// TIA Portal V17 export
// export: Created 2023-02-14T02:49:49.5801565Z, ExportSetting WithDefaults, DisplayName Totally Integrated Automation Portal, DisplayVersion V17, DisplayName TIA Portal Openness, DisplayVersion V17, DisplayName TIA Portal Teamcenter Gateway, DisplayVersion V17, DisplayName TIA Portal Version Control Interface, DisplayVersion V17, DisplayName SINAMICS Startdrive Advanced, DisplayVersion V17, DisplayName SINAMICS Startdrive G130, G150, S120, S150, SINAMICS MV, S210, DisplayVersion V17, DisplayName SINAMICS Startdrive G110M, G120, G120C, G120D, G120P, G115D, DisplayVersion V17, DisplayName STEP 7 Professional, DisplayVersion V17, DisplayName STEP 7 Safety, DisplayVersion V17, DisplayName WinCC Professional, DisplayVersion V17
FUNCTION "Preparation" : Void   // FC6, LAD
{ S7_Optimized_Access := 'TRUE' }
VERSION : 0.1
// stored: AutoNumber true, IsIECCheckEnabled false, SetENOAutomatically false, UDAEnableTagReadback false
   VAR_TEMP   // added for the SCL form of the ladder/FBD networks
      _w1 : Bool;
      _w2 : Bool;
      _w3 : Bool;
      _w4 : Bool;
      _w5 : Bool;
   END_VAR
BEGIN

REGION Network 1: Analog IO
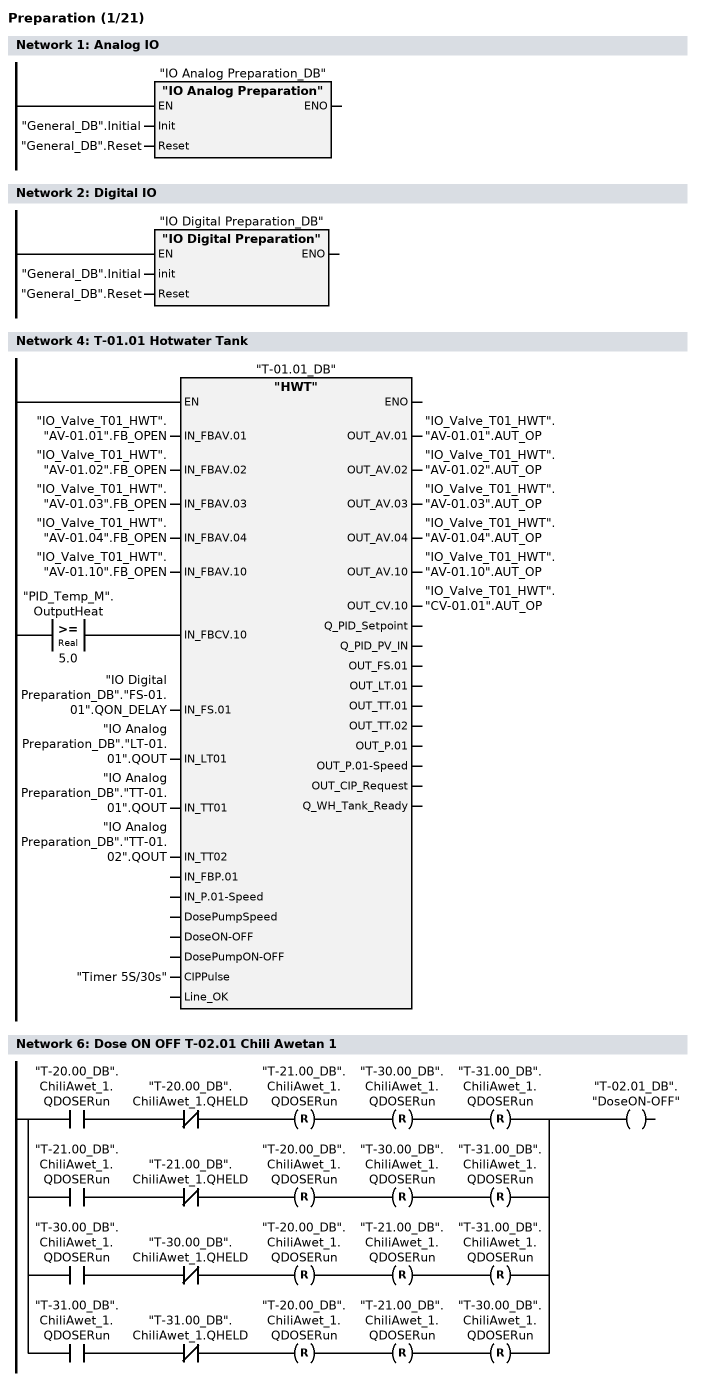
   RUNG wire#powerrail
      "IO Analog Preparation_DB"(Init := "General_DB".Initial, Reset := "General_DB".Reset)
   END_RUNG
   // the same network as SCL:
   "IO Analog Preparation_DB"(Init := "General_DB".Initial, Reset := "General_DB".Reset);   // "IO Analog Preparation"
END_REGION

REGION Network 2: Digital IO
   RUNG wire#powerrail
      "IO Digital Preparation_DB"(init := "General_DB".Initial, Reset := "General_DB".Reset)
   END_RUNG
   // the same network as SCL:
   "IO Digital Preparation_DB"(init := "General_DB".Initial, Reset := "General_DB".Reset);   // "IO Digital Preparation"
END_REGION

REGION Network 4: T-01.01 Hotwater Tank
   RUNG wire#powerrail
      "T-01.01_DB"("IN_FBCV.10" := wire#w1, "IN_FBAV.01" := "IO_Valve_T01_HWT"."AV-01.01".FB_OPEN, "IN_FBAV.02" := "IO_Valve_T01_HWT"."AV-01.02".FB_OPEN, "IN_FBAV.03" := "IO_Valve_T01_HWT"."AV-01.03".FB_OPEN, "IN_FBAV.04" := "IO_Valve_T01_HWT"."AV-01.04".FB_OPEN, "IN_FBAV.10" := "IO_Valve_T01_HWT"."AV-01.10".FB_OPEN, "IN_FS.01" := "IO Digital Preparation_DB"."FS-01.01".QON_DELAY, IN_LT01 := "IO Analog Preparation_DB"."LT-01.01".QOUT, IN_TT01 := "IO Analog Preparation_DB"."TT-01.01".QOUT, IN_TT02 := "IO Analog Preparation_DB"."TT-01.02".QOUT, "IN_FBP.01" :=, "IN_P.01-Speed" :=, DosePumpSpeed :=, "DoseON-OFF" :=, "DosePumpON-OFF" :=, CIPPulse := "Timer 5S/30s", Line_OK :=, "OUT_AV.01" => "IO_Valve_T01_HWT"."AV-01.01".AUT_OP, "OUT_AV.02" => "IO_Valve_T01_HWT"."AV-01.02".AUT_OP, "OUT_AV.03" => "IO_Valve_T01_HWT"."AV-01.03".AUT_OP, "OUT_AV.04" => "IO_Valve_T01_HWT"."AV-01.04".AUT_OP, "OUT_AV.10" => "IO_Valve_T01_HWT"."AV-01.10".AUT_OP, "OUT_CV.10" => "IO_Valve_T01_HWT"."CV-01.01".AUT_OP, Q_PID_Setpoint =>, Q_PID_PV_IN =>, "OUT_FS.01" =>, "OUT_LT.01" =>, "OUT_TT.01" =>, "OUT_TT.02" =>, "OUT_P.01" =>, "OUT_P.01-Speed" =>, OUT_CIP_Request =>, Q_WH_Tank_Ready =>)
   END_RUNG
   RUNG wire#powerrail
      { S7_Templates := "SrcType := Real" } GE_Contact(in1 := "PID_Temp_M".OutputHeat, in2 := 5.0)
   END_RUNG wire#w1
   // the same network as SCL:
   "T-01.01_DB"("IN_FBAV.01" := "IO_Valve_T01_HWT"."AV-01.01".FB_OPEN,   // "HWT"
                "IN_FBAV.02" := "IO_Valve_T01_HWT"."AV-01.02".FB_OPEN,
                "IN_FBAV.03" := "IO_Valve_T01_HWT"."AV-01.03".FB_OPEN,
                "IN_FBAV.04" := "IO_Valve_T01_HWT"."AV-01.04".FB_OPEN,
                "IN_FBAV.10" := "IO_Valve_T01_HWT"."AV-01.10".FB_OPEN,
                "IN_FBCV.10" := "PID_Temp_M".OutputHeat >= 5.0,
                "IN_FS.01" := "IO Digital Preparation_DB"."FS-01.01".QON_DELAY,
                IN_LT01 := "IO Analog Preparation_DB"."LT-01.01".QOUT,
                IN_TT01 := "IO Analog Preparation_DB"."TT-01.01".QOUT,
                IN_TT02 := "IO Analog Preparation_DB"."TT-01.02".QOUT,
                CIPPulse := "Timer 5S/30s",
                "OUT_AV.01" => "IO_Valve_T01_HWT"."AV-01.01".AUT_OP,
                "OUT_AV.02" => "IO_Valve_T01_HWT"."AV-01.02".AUT_OP,
                "OUT_AV.03" => "IO_Valve_T01_HWT"."AV-01.03".AUT_OP,
                "OUT_AV.04" => "IO_Valve_T01_HWT"."AV-01.04".AUT_OP,
                "OUT_AV.10" => "IO_Valve_T01_HWT"."AV-01.10".AUT_OP,
                "OUT_CV.10" => "IO_Valve_T01_HWT"."CV-01.01".AUT_OP);
END_REGION

REGION Network 6: Dose ON OFF T-02.01 Chili Awetan 1
   RUNG wire#powerrail
      Contact( "T-20.00_DB".ChiliAwet_1.QDOSERun )
      I_Contact( "T-20.00_DB".ChiliAwet_1.QHELD )
      R_Coil( "T-21.00_DB".ChiliAwet_1.QDOSERun )
      R_Coil( "T-30.00_DB".ChiliAwet_1.QDOSERun )
      R_Coil( "T-31.00_DB".ChiliAwet_1.QDOSERun )
      wire#w1
      Coil( "T-02.01_DB"."DoseON-OFF" )
   END_RUNG
   RUNG wire#powerrail
      Contact( "T-21.00_DB".ChiliAwet_1.QDOSERun )
      I_Contact( "T-21.00_DB".ChiliAwet_1.QHELD )
      R_Coil( "T-20.00_DB".ChiliAwet_1.QDOSERun )
      R_Coil( "T-30.00_DB".ChiliAwet_1.QDOSERun )
      R_Coil( "T-31.00_DB".ChiliAwet_1.QDOSERun )
   END_RUNG wire#w1
   RUNG wire#powerrail
      Contact( "T-30.00_DB".ChiliAwet_1.QDOSERun )
      I_Contact( "T-30.00_DB".ChiliAwet_1.QHELD )
      R_Coil( "T-20.00_DB".ChiliAwet_1.QDOSERun )
      R_Coil( "T-21.00_DB".ChiliAwet_1.QDOSERun )
      R_Coil( "T-31.00_DB".ChiliAwet_1.QDOSERun )
   END_RUNG wire#w1
   RUNG wire#powerrail
      Contact( "T-31.00_DB".ChiliAwet_1.QDOSERun )
      I_Contact( "T-31.00_DB".ChiliAwet_1.QHELD )
      R_Coil( "T-20.00_DB".ChiliAwet_1.QDOSERun )
      R_Coil( "T-21.00_DB".ChiliAwet_1.QDOSERun )
      R_Coil( "T-30.00_DB".ChiliAwet_1.QDOSERun )
   END_RUNG wire#w1
   // the same network as SCL:
   #_w1 := "T-20.00_DB".ChiliAwet_1.QDOSERun AND NOT "T-20.00_DB".ChiliAwet_1.QHELD;
   IF #_w1 THEN
       "T-21.00_DB".ChiliAwet_1.QDOSERun := FALSE;
       "T-30.00_DB".ChiliAwet_1.QDOSERun := FALSE;
       "T-31.00_DB".ChiliAwet_1.QDOSERun := FALSE;
   END_IF;
   #_w2 := "T-21.00_DB".ChiliAwet_1.QDOSERun AND NOT "T-21.00_DB".ChiliAwet_1.QHELD;
   IF #_w2 THEN
       "T-20.00_DB".ChiliAwet_1.QDOSERun := FALSE;
       "T-30.00_DB".ChiliAwet_1.QDOSERun := FALSE;
       "T-31.00_DB".ChiliAwet_1.QDOSERun := FALSE;
   END_IF;
   #_w3 := "T-30.00_DB".ChiliAwet_1.QDOSERun AND NOT "T-30.00_DB".ChiliAwet_1.QHELD;
   IF #_w3 THEN
       "T-20.00_DB".ChiliAwet_1.QDOSERun := FALSE;
       "T-21.00_DB".ChiliAwet_1.QDOSERun := FALSE;
       "T-31.00_DB".ChiliAwet_1.QDOSERun := FALSE;
   END_IF;
   #_w4 := "T-31.00_DB".ChiliAwet_1.QDOSERun AND NOT "T-31.00_DB".ChiliAwet_1.QHELD;
   IF #_w4 THEN
       "T-20.00_DB".ChiliAwet_1.QDOSERun := FALSE;
       "T-21.00_DB".ChiliAwet_1.QDOSERun := FALSE;
       "T-30.00_DB".ChiliAwet_1.QDOSERun := FALSE;
   END_IF;
   "T-02.01_DB"."DoseON-OFF" := #_w1 OR #_w2 OR #_w3 OR #_w4;
END_REGION

REGION Network 7: Dose Pump ON OFF T-02.01 Chili Awetan 1
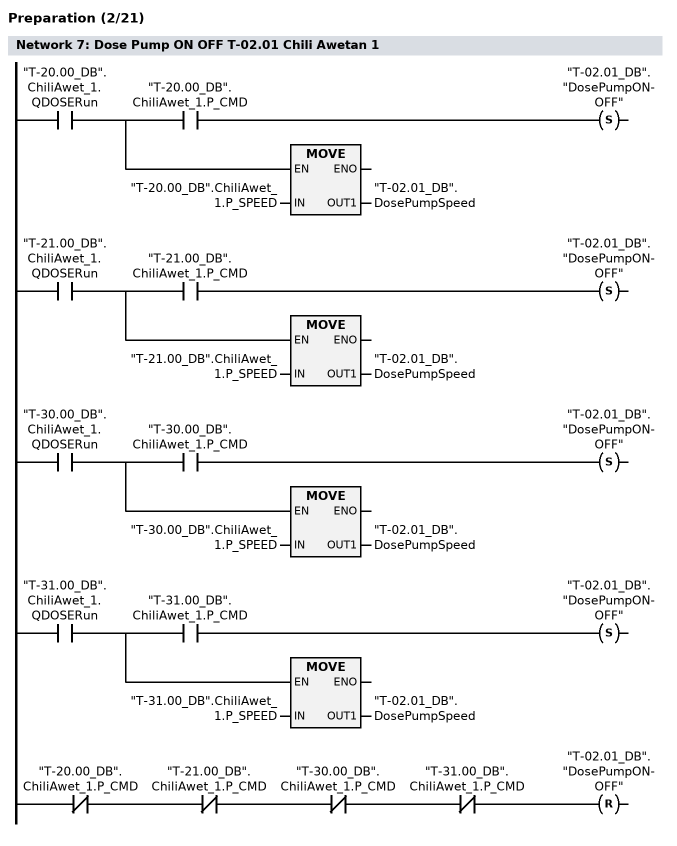
   RUNG wire#powerrail
      Contact( "T-20.00_DB".ChiliAwet_1.QDOSERun )
      wire#w1
      Contact( "T-20.00_DB".ChiliAwet_1.P_CMD )
      S_Coil( "T-02.01_DB"."DosePumpON-OFF" )
   END_RUNG
   RUNG wire#w1
      Move(in := "T-20.00_DB".ChiliAwet_1.P_SPEED, out1 => "T-02.01_DB".DosePumpSpeed)
   END_RUNG
   RUNG wire#powerrail
      Contact( "T-21.00_DB".ChiliAwet_1.QDOSERun )
      wire#w2
      Contact( "T-21.00_DB".ChiliAwet_1.P_CMD )
      S_Coil( "T-02.01_DB"."DosePumpON-OFF" )
   END_RUNG
   RUNG wire#w2
      Move(in := "T-21.00_DB".ChiliAwet_1.P_SPEED, out1 => "T-02.01_DB".DosePumpSpeed)
   END_RUNG
   RUNG wire#powerrail
      Contact( "T-30.00_DB".ChiliAwet_1.QDOSERun )
      wire#w3
      Contact( "T-30.00_DB".ChiliAwet_1.P_CMD )
      S_Coil( "T-02.01_DB"."DosePumpON-OFF" )
   END_RUNG
   RUNG wire#w3
      Move(in := "T-30.00_DB".ChiliAwet_1.P_SPEED, out1 => "T-02.01_DB".DosePumpSpeed)
   END_RUNG
   RUNG wire#powerrail
      Contact( "T-31.00_DB".ChiliAwet_1.QDOSERun )
      wire#w4
      Contact( "T-31.00_DB".ChiliAwet_1.P_CMD )
      S_Coil( "T-02.01_DB"."DosePumpON-OFF" )
   END_RUNG
   RUNG wire#w4
      Move(in := "T-31.00_DB".ChiliAwet_1.P_SPEED, out1 => "T-02.01_DB".DosePumpSpeed)
   END_RUNG
   RUNG wire#powerrail
      I_Contact( "T-20.00_DB".ChiliAwet_1.P_CMD )
      I_Contact( "T-21.00_DB".ChiliAwet_1.P_CMD )
      I_Contact( "T-30.00_DB".ChiliAwet_1.P_CMD )
      I_Contact( "T-31.00_DB".ChiliAwet_1.P_CMD )
      R_Coil( "T-02.01_DB"."DosePumpON-OFF" )
   END_RUNG
   // the same network as SCL:
   IF "T-20.00_DB".ChiliAwet_1.QDOSERun AND "T-20.00_DB".ChiliAwet_1.P_CMD THEN
       "T-02.01_DB"."DosePumpON-OFF" := TRUE;
   END_IF;
   IF "T-20.00_DB".ChiliAwet_1.QDOSERun THEN
       "T-02.01_DB".DosePumpSpeed := "T-20.00_DB".ChiliAwet_1.P_SPEED;
   END_IF;
   IF "T-21.00_DB".ChiliAwet_1.QDOSERun AND "T-21.00_DB".ChiliAwet_1.P_CMD THEN
       "T-02.01_DB"."DosePumpON-OFF" := TRUE;
   END_IF;
   IF "T-21.00_DB".ChiliAwet_1.QDOSERun THEN
       "T-02.01_DB".DosePumpSpeed := "T-21.00_DB".ChiliAwet_1.P_SPEED;
   END_IF;
   IF "T-30.00_DB".ChiliAwet_1.QDOSERun AND "T-30.00_DB".ChiliAwet_1.P_CMD THEN
       "T-02.01_DB"."DosePumpON-OFF" := TRUE;
   END_IF;
   IF "T-30.00_DB".ChiliAwet_1.QDOSERun THEN
       "T-02.01_DB".DosePumpSpeed := "T-30.00_DB".ChiliAwet_1.P_SPEED;
   END_IF;
   IF "T-31.00_DB".ChiliAwet_1.QDOSERun AND "T-31.00_DB".ChiliAwet_1.P_CMD THEN
       "T-02.01_DB"."DosePumpON-OFF" := TRUE;
   END_IF;
   IF "T-31.00_DB".ChiliAwet_1.QDOSERun THEN
       "T-02.01_DB".DosePumpSpeed := "T-31.00_DB".ChiliAwet_1.P_SPEED;
   END_IF;
   IF NOT "T-20.00_DB".ChiliAwet_1.P_CMD AND NOT "T-21.00_DB".ChiliAwet_1.P_CMD AND NOT "T-30.00_DB".ChiliAwet_1.P_CMD AND NOT "T-31.00_DB".ChiliAwet_1.P_CMD THEN
       "T-02.01_DB"."DosePumpON-OFF" := FALSE;
   END_IF;
END_REGION

REGION Network 8: T-02.01 Buffer Tank Chili Awetan
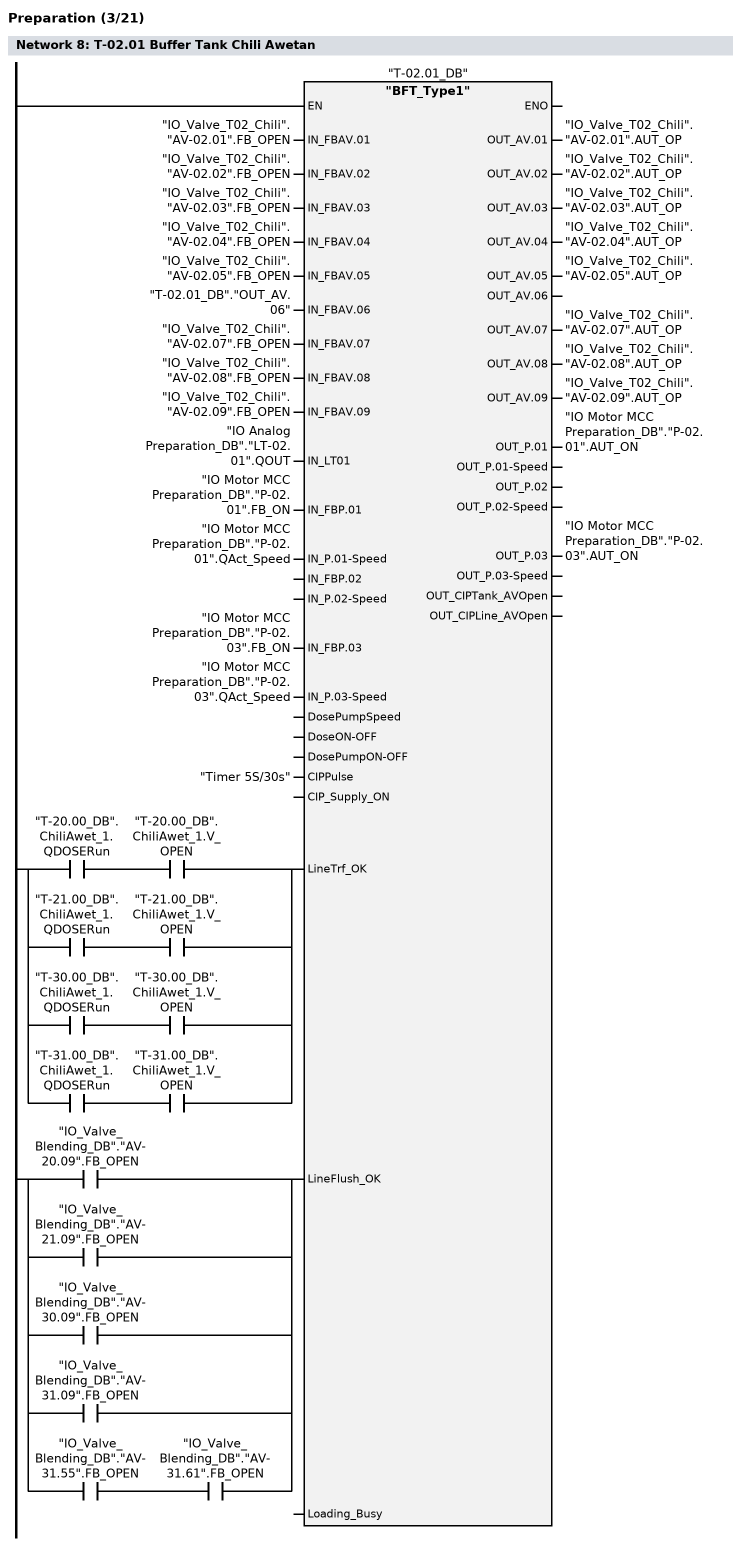
   RUNG wire#powerrail
      "T-02.01_DB"(LineTrf_OK := wire#w1, LineFlush_OK := wire#w2, "IN_FBAV.01" := "IO_Valve_T02_Chili"."AV-02.01".FB_OPEN, "IN_FBAV.02" := "IO_Valve_T02_Chili"."AV-02.02".FB_OPEN, "IN_FBAV.03" := "IO_Valve_T02_Chili"."AV-02.03".FB_OPEN, "IN_FBAV.04" := "IO_Valve_T02_Chili"."AV-02.04".FB_OPEN, "IN_FBAV.05" := "IO_Valve_T02_Chili"."AV-02.05".FB_OPEN, "IN_FBAV.06" := "T-02.01_DB"."OUT_AV.06", "IN_FBAV.07" := "IO_Valve_T02_Chili"."AV-02.07".FB_OPEN, "IN_FBAV.08" := "IO_Valve_T02_Chili"."AV-02.08".FB_OPEN, "IN_FBAV.09" := "IO_Valve_T02_Chili"."AV-02.09".FB_OPEN, IN_LT01 := "IO Analog Preparation_DB"."LT-02.01".QOUT, "IN_FBP.01" := "IO Motor MCC Preparation_DB"."P-02.01".FB_ON, "IN_P.01-Speed" := "IO Motor MCC Preparation_DB"."P-02.01".QAct_Speed, "IN_FBP.02" :=, "IN_P.02-Speed" :=, "IN_FBP.03" := "IO Motor MCC Preparation_DB"."P-02.03".FB_ON, "IN_P.03-Speed" := "IO Motor MCC Preparation_DB"."P-02.03".QAct_Speed, DosePumpSpeed :=, "DoseON-OFF" :=, "DosePumpON-OFF" :=, CIPPulse := "Timer 5S/30s", CIP_Supply_ON :=, Loading_Busy :=, "OUT_AV.01" => "IO_Valve_T02_Chili"."AV-02.01".AUT_OP, "OUT_AV.02" => "IO_Valve_T02_Chili"."AV-02.02".AUT_OP, "OUT_AV.03" => "IO_Valve_T02_Chili"."AV-02.03".AUT_OP, "OUT_AV.04" => "IO_Valve_T02_Chili"."AV-02.04".AUT_OP, "OUT_AV.05" => "IO_Valve_T02_Chili"."AV-02.05".AUT_OP, "OUT_AV.06" =>, "OUT_AV.07" => "IO_Valve_T02_Chili"."AV-02.07".AUT_OP, "OUT_AV.08" => "IO_Valve_T02_Chili"."AV-02.08".AUT_OP, "OUT_AV.09" => "IO_Valve_T02_Chili"."AV-02.09".AUT_OP, "OUT_P.01" => "IO Motor MCC Preparation_DB"."P-02.01".AUT_ON, "OUT_P.01-Speed" =>, "OUT_P.02" =>, "OUT_P.02-Speed" =>, "OUT_P.03" => "IO Motor MCC Preparation_DB"."P-02.03".AUT_ON, "OUT_P.03-Speed" =>, OUT_CIPTank_AVOpen =>, OUT_CIPLine_AVOpen =>)
   END_RUNG
   RUNG wire#powerrail
      Contact( "T-20.00_DB".ChiliAwet_1.QDOSERun )
      Contact( "T-20.00_DB".ChiliAwet_1.V_OPEN )
   END_RUNG wire#w1
   RUNG wire#powerrail
      Contact( "T-21.00_DB".ChiliAwet_1.QDOSERun )
      Contact( "T-21.00_DB".ChiliAwet_1.V_OPEN )
   END_RUNG wire#w1
   RUNG wire#powerrail
      Contact( "T-30.00_DB".ChiliAwet_1.QDOSERun )
      Contact( "T-30.00_DB".ChiliAwet_1.V_OPEN )
   END_RUNG wire#w1
   RUNG wire#powerrail
      Contact( "T-31.00_DB".ChiliAwet_1.QDOSERun )
      Contact( "T-31.00_DB".ChiliAwet_1.V_OPEN )
   END_RUNG wire#w1
   RUNG wire#powerrail
      Contact( "IO_Valve_Blending_DB"."AV-20.09".FB_OPEN )
   END_RUNG wire#w2
   RUNG wire#powerrail
      Contact( "IO_Valve_Blending_DB"."AV-21.09".FB_OPEN )
   END_RUNG wire#w2
   RUNG wire#powerrail
      Contact( "IO_Valve_Blending_DB"."AV-30.09".FB_OPEN )
   END_RUNG wire#w2
   RUNG wire#powerrail
      Contact( "IO_Valve_Blending_DB"."AV-31.09".FB_OPEN )
   END_RUNG wire#w2
   RUNG wire#powerrail
      Contact( "IO_Valve_Blending_DB"."AV-31.55".FB_OPEN )
      Contact( "IO_Valve_Blending_DB"."AV-31.61".FB_OPEN )
   END_RUNG wire#w2
   // the same network as SCL:
   "T-02.01_DB"("IN_FBAV.01" := "IO_Valve_T02_Chili"."AV-02.01".FB_OPEN,   // "BFT_Type1"
                "IN_FBAV.02" := "IO_Valve_T02_Chili"."AV-02.02".FB_OPEN,
                "IN_FBAV.03" := "IO_Valve_T02_Chili"."AV-02.03".FB_OPEN,
                "IN_FBAV.04" := "IO_Valve_T02_Chili"."AV-02.04".FB_OPEN,
                "IN_FBAV.05" := "IO_Valve_T02_Chili"."AV-02.05".FB_OPEN,
                "IN_FBAV.06" := "T-02.01_DB"."OUT_AV.06",
                "IN_FBAV.07" := "IO_Valve_T02_Chili"."AV-02.07".FB_OPEN,
                "IN_FBAV.08" := "IO_Valve_T02_Chili"."AV-02.08".FB_OPEN,
                "IN_FBAV.09" := "IO_Valve_T02_Chili"."AV-02.09".FB_OPEN,
                IN_LT01 := "IO Analog Preparation_DB"."LT-02.01".QOUT,
                "IN_FBP.01" := "IO Motor MCC Preparation_DB"."P-02.01".FB_ON,
                "IN_P.01-Speed" := "IO Motor MCC Preparation_DB"."P-02.01".QAct_Speed,
                "IN_FBP.03" := "IO Motor MCC Preparation_DB"."P-02.03".FB_ON,
                "IN_P.03-Speed" := "IO Motor MCC Preparation_DB"."P-02.03".QAct_Speed,
                CIPPulse := "Timer 5S/30s",
                LineTrf_OK := ("T-20.00_DB".ChiliAwet_1.QDOSERun AND "T-20.00_DB".ChiliAwet_1.V_OPEN) OR ("T-21.00_DB".ChiliAwet_1.QDOSERun AND "T-21.00_DB".ChiliAwet_1.V_OPEN) OR ("T-30.00_DB".ChiliAwet_1.QDOSERun AND "T-30.00_DB".ChiliAwet_1.V_OPEN) OR ("T-31.00_DB".ChiliAwet_1.QDOSERun AND "T-31.00_DB".ChiliAwet_1.V_OPEN),
                LineFlush_OK := "IO_Valve_Blending_DB"."AV-20.09".FB_OPEN OR "IO_Valve_Blending_DB"."AV-21.09".FB_OPEN OR "IO_Valve_Blending_DB"."AV-30.09".FB_OPEN OR "IO_Valve_Blending_DB"."AV-31.09".FB_OPEN OR ("IO_Valve_Blending_DB"."AV-31.55".FB_OPEN AND "IO_Valve_Blending_DB"."AV-31.61".FB_OPEN),
                "OUT_AV.01" => "IO_Valve_T02_Chili"."AV-02.01".AUT_OP,
                "OUT_AV.02" => "IO_Valve_T02_Chili"."AV-02.02".AUT_OP,
                "OUT_AV.03" => "IO_Valve_T02_Chili"."AV-02.03".AUT_OP,
                "OUT_AV.04" => "IO_Valve_T02_Chili"."AV-02.04".AUT_OP,
                "OUT_AV.05" => "IO_Valve_T02_Chili"."AV-02.05".AUT_OP,
                "OUT_AV.07" => "IO_Valve_T02_Chili"."AV-02.07".AUT_OP,
                "OUT_AV.08" => "IO_Valve_T02_Chili"."AV-02.08".AUT_OP,
                "OUT_AV.09" => "IO_Valve_T02_Chili"."AV-02.09".AUT_OP,
                "OUT_P.01" => "IO Motor MCC Preparation_DB"."P-02.01".AUT_ON,
                "OUT_P.03" => "IO Motor MCC Preparation_DB"."P-02.03".AUT_ON);
END_REGION

REGION Network 10: Dose ON OFF T-03.01 Chili Awetan 2
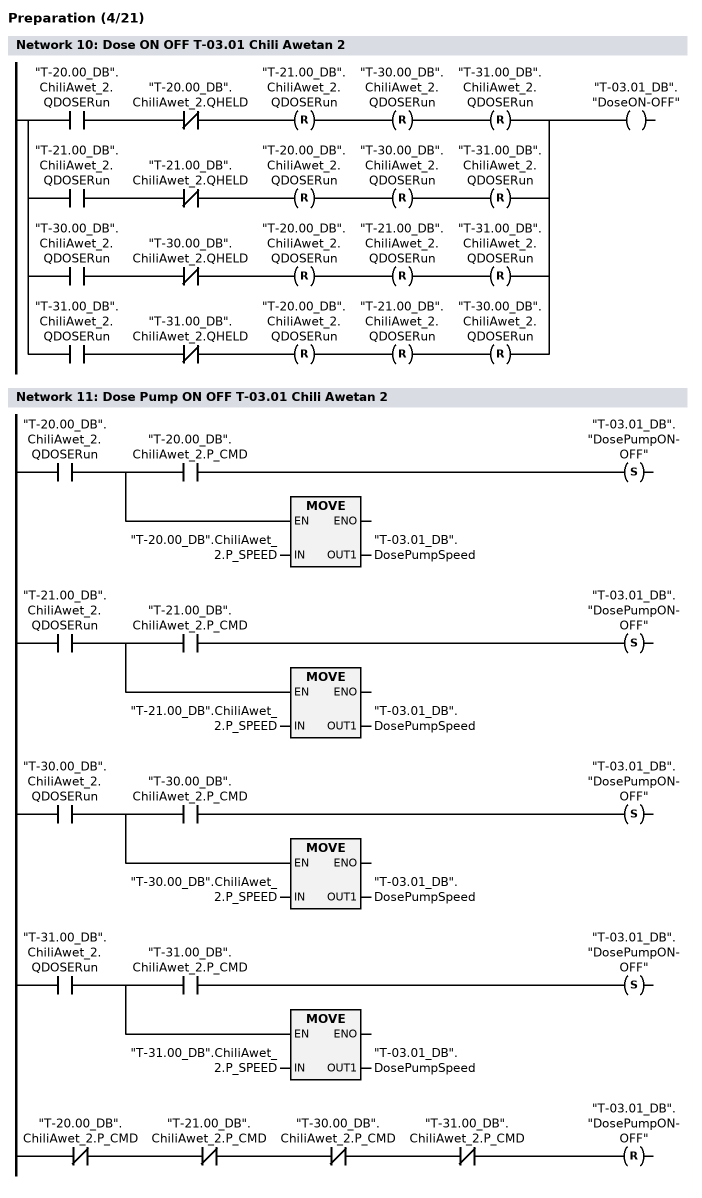
   RUNG wire#powerrail
      Contact( "T-20.00_DB".ChiliAwet_2.QDOSERun )
      I_Contact( "T-20.00_DB".ChiliAwet_2.QHELD )
      R_Coil( "T-21.00_DB".ChiliAwet_2.QDOSERun )
      R_Coil( "T-30.00_DB".ChiliAwet_2.QDOSERun )
      R_Coil( "T-31.00_DB".ChiliAwet_2.QDOSERun )
      wire#w1
      Coil( "T-03.01_DB"."DoseON-OFF" )
   END_RUNG
   RUNG wire#powerrail
      Contact( "T-21.00_DB".ChiliAwet_2.QDOSERun )
      I_Contact( "T-21.00_DB".ChiliAwet_2.QHELD )
      R_Coil( "T-20.00_DB".ChiliAwet_2.QDOSERun )
      R_Coil( "T-30.00_DB".ChiliAwet_2.QDOSERun )
      R_Coil( "T-31.00_DB".ChiliAwet_2.QDOSERun )
   END_RUNG wire#w1
   RUNG wire#powerrail
      Contact( "T-30.00_DB".ChiliAwet_2.QDOSERun )
      I_Contact( "T-30.00_DB".ChiliAwet_2.QHELD )
      R_Coil( "T-20.00_DB".ChiliAwet_2.QDOSERun )
      R_Coil( "T-21.00_DB".ChiliAwet_2.QDOSERun )
      R_Coil( "T-31.00_DB".ChiliAwet_2.QDOSERun )
   END_RUNG wire#w1
   RUNG wire#powerrail
      Contact( "T-31.00_DB".ChiliAwet_2.QDOSERun )
      I_Contact( "T-31.00_DB".ChiliAwet_2.QHELD )
      R_Coil( "T-20.00_DB".ChiliAwet_2.QDOSERun )
      R_Coil( "T-21.00_DB".ChiliAwet_2.QDOSERun )
      R_Coil( "T-30.00_DB".ChiliAwet_2.QDOSERun )
   END_RUNG wire#w1
   // the same network as SCL:
   #_w1 := "T-20.00_DB".ChiliAwet_2.QDOSERun AND NOT "T-20.00_DB".ChiliAwet_2.QHELD;
   IF #_w1 THEN
       "T-21.00_DB".ChiliAwet_2.QDOSERun := FALSE;
       "T-30.00_DB".ChiliAwet_2.QDOSERun := FALSE;
       "T-31.00_DB".ChiliAwet_2.QDOSERun := FALSE;
   END_IF;
   #_w2 := "T-21.00_DB".ChiliAwet_2.QDOSERun AND NOT "T-21.00_DB".ChiliAwet_2.QHELD;
   IF #_w2 THEN
       "T-20.00_DB".ChiliAwet_2.QDOSERun := FALSE;
       "T-30.00_DB".ChiliAwet_2.QDOSERun := FALSE;
       "T-31.00_DB".ChiliAwet_2.QDOSERun := FALSE;
   END_IF;
   #_w3 := "T-30.00_DB".ChiliAwet_2.QDOSERun AND NOT "T-30.00_DB".ChiliAwet_2.QHELD;
   IF #_w3 THEN
       "T-20.00_DB".ChiliAwet_2.QDOSERun := FALSE;
       "T-21.00_DB".ChiliAwet_2.QDOSERun := FALSE;
       "T-31.00_DB".ChiliAwet_2.QDOSERun := FALSE;
   END_IF;
   #_w4 := "T-31.00_DB".ChiliAwet_2.QDOSERun AND NOT "T-31.00_DB".ChiliAwet_2.QHELD;
   IF #_w4 THEN
       "T-20.00_DB".ChiliAwet_2.QDOSERun := FALSE;
       "T-21.00_DB".ChiliAwet_2.QDOSERun := FALSE;
       "T-30.00_DB".ChiliAwet_2.QDOSERun := FALSE;
   END_IF;
   "T-03.01_DB"."DoseON-OFF" := #_w1 OR #_w2 OR #_w3 OR #_w4;
END_REGION

REGION Network 11: Dose Pump ON OFF T-03.01 Chili Awetan 2
   RUNG wire#powerrail
      Contact( "T-20.00_DB".ChiliAwet_2.QDOSERun )
      wire#w1
      Contact( "T-20.00_DB".ChiliAwet_2.P_CMD )
      S_Coil( "T-03.01_DB"."DosePumpON-OFF" )
   END_RUNG
   RUNG wire#w1
      Move(in := "T-20.00_DB".ChiliAwet_2.P_SPEED, out1 => "T-03.01_DB".DosePumpSpeed)
   END_RUNG
   RUNG wire#powerrail
      Contact( "T-21.00_DB".ChiliAwet_2.QDOSERun )
      wire#w2
      Contact( "T-21.00_DB".ChiliAwet_2.P_CMD )
      S_Coil( "T-03.01_DB"."DosePumpON-OFF" )
   END_RUNG
   RUNG wire#w2
      Move(in := "T-21.00_DB".ChiliAwet_2.P_SPEED, out1 => "T-03.01_DB".DosePumpSpeed)
   END_RUNG
   RUNG wire#powerrail
      Contact( "T-30.00_DB".ChiliAwet_2.QDOSERun )
      wire#w3
      Contact( "T-30.00_DB".ChiliAwet_2.P_CMD )
      S_Coil( "T-03.01_DB"."DosePumpON-OFF" )
   END_RUNG
   RUNG wire#w3
      Move(in := "T-30.00_DB".ChiliAwet_2.P_SPEED, out1 => "T-03.01_DB".DosePumpSpeed)
   END_RUNG
   RUNG wire#powerrail
      Contact( "T-31.00_DB".ChiliAwet_2.QDOSERun )
      wire#w4
      Contact( "T-31.00_DB".ChiliAwet_2.P_CMD )
      S_Coil( "T-03.01_DB"."DosePumpON-OFF" )
   END_RUNG
   RUNG wire#w4
      Move(in := "T-31.00_DB".ChiliAwet_2.P_SPEED, out1 => "T-03.01_DB".DosePumpSpeed)
   END_RUNG
   RUNG wire#powerrail
      I_Contact( "T-20.00_DB".ChiliAwet_2.P_CMD )
      I_Contact( "T-21.00_DB".ChiliAwet_2.P_CMD )
      I_Contact( "T-30.00_DB".ChiliAwet_2.P_CMD )
      I_Contact( "T-31.00_DB".ChiliAwet_2.P_CMD )
      R_Coil( "T-03.01_DB"."DosePumpON-OFF" )
   END_RUNG
   // the same network as SCL:
   IF "T-20.00_DB".ChiliAwet_2.QDOSERun AND "T-20.00_DB".ChiliAwet_2.P_CMD THEN
       "T-03.01_DB"."DosePumpON-OFF" := TRUE;
   END_IF;
   IF "T-20.00_DB".ChiliAwet_2.QDOSERun THEN
       "T-03.01_DB".DosePumpSpeed := "T-20.00_DB".ChiliAwet_2.P_SPEED;
   END_IF;
   IF "T-21.00_DB".ChiliAwet_2.QDOSERun AND "T-21.00_DB".ChiliAwet_2.P_CMD THEN
       "T-03.01_DB"."DosePumpON-OFF" := TRUE;
   END_IF;
   IF "T-21.00_DB".ChiliAwet_2.QDOSERun THEN
       "T-03.01_DB".DosePumpSpeed := "T-21.00_DB".ChiliAwet_2.P_SPEED;
   END_IF;
   IF "T-30.00_DB".ChiliAwet_2.QDOSERun AND "T-30.00_DB".ChiliAwet_2.P_CMD THEN
       "T-03.01_DB"."DosePumpON-OFF" := TRUE;
   END_IF;
   IF "T-30.00_DB".ChiliAwet_2.QDOSERun THEN
       "T-03.01_DB".DosePumpSpeed := "T-30.00_DB".ChiliAwet_2.P_SPEED;
   END_IF;
   IF "T-31.00_DB".ChiliAwet_2.QDOSERun AND "T-31.00_DB".ChiliAwet_2.P_CMD THEN
       "T-03.01_DB"."DosePumpON-OFF" := TRUE;
   END_IF;
   IF "T-31.00_DB".ChiliAwet_2.QDOSERun THEN
       "T-03.01_DB".DosePumpSpeed := "T-31.00_DB".ChiliAwet_2.P_SPEED;
   END_IF;
   IF NOT "T-20.00_DB".ChiliAwet_2.P_CMD AND NOT "T-21.00_DB".ChiliAwet_2.P_CMD AND NOT "T-30.00_DB".ChiliAwet_2.P_CMD AND NOT "T-31.00_DB".ChiliAwet_2.P_CMD THEN
       "T-03.01_DB"."DosePumpON-OFF" := FALSE;
   END_IF;
END_REGION

REGION Network 12: T-03.01 Buffer Tank Chili Awetan
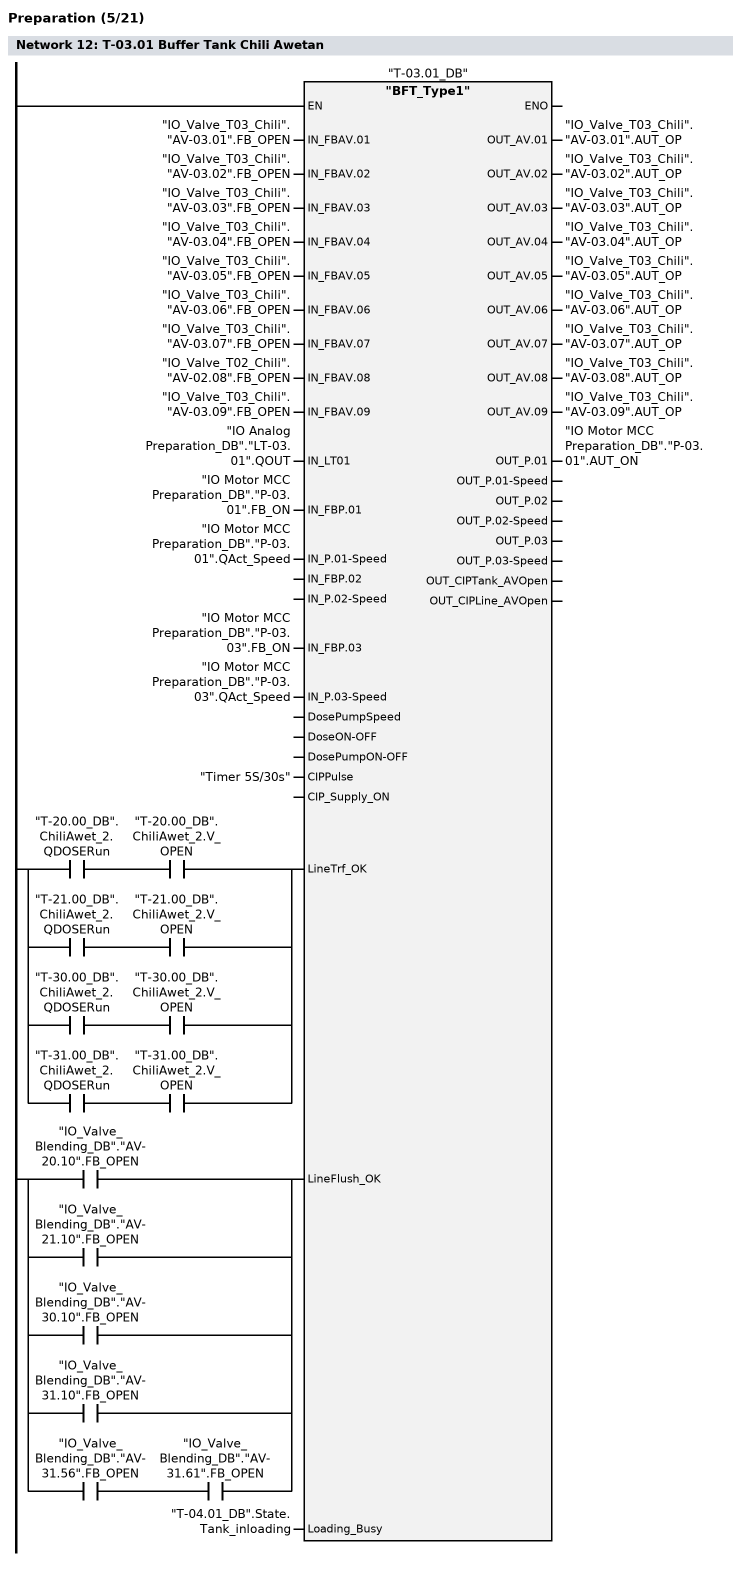
   RUNG wire#powerrail
      "T-03.01_DB"(LineTrf_OK := wire#w1, LineFlush_OK := wire#w2, "IN_FBAV.01" := "IO_Valve_T03_Chili"."AV-03.01".FB_OPEN, "IN_FBAV.02" := "IO_Valve_T03_Chili"."AV-03.02".FB_OPEN, "IN_FBAV.03" := "IO_Valve_T03_Chili"."AV-03.03".FB_OPEN, "IN_FBAV.04" := "IO_Valve_T03_Chili"."AV-03.04".FB_OPEN, "IN_FBAV.05" := "IO_Valve_T03_Chili"."AV-03.05".FB_OPEN, "IN_FBAV.06" := "IO_Valve_T03_Chili"."AV-03.06".FB_OPEN, "IN_FBAV.07" := "IO_Valve_T03_Chili"."AV-03.07".FB_OPEN, "IN_FBAV.08" := "IO_Valve_T02_Chili"."AV-02.08".FB_OPEN, "IN_FBAV.09" := "IO_Valve_T03_Chili"."AV-03.09".FB_OPEN, IN_LT01 := "IO Analog Preparation_DB"."LT-03.01".QOUT, "IN_FBP.01" := "IO Motor MCC Preparation_DB"."P-03.01".FB_ON, "IN_P.01-Speed" := "IO Motor MCC Preparation_DB"."P-03.01".QAct_Speed, "IN_FBP.02" :=, "IN_P.02-Speed" :=, "IN_FBP.03" := "IO Motor MCC Preparation_DB"."P-03.03".FB_ON, "IN_P.03-Speed" := "IO Motor MCC Preparation_DB"."P-03.03".QAct_Speed, DosePumpSpeed :=, "DoseON-OFF" :=, "DosePumpON-OFF" :=, CIPPulse := "Timer 5S/30s", CIP_Supply_ON :=, Loading_Busy := "T-04.01_DB".State.Tank_inloading, "OUT_AV.01" => "IO_Valve_T03_Chili"."AV-03.01".AUT_OP, "OUT_AV.02" => "IO_Valve_T03_Chili"."AV-03.02".AUT_OP, "OUT_AV.03" => "IO_Valve_T03_Chili"."AV-03.03".AUT_OP, "OUT_AV.04" => "IO_Valve_T03_Chili"."AV-03.04".AUT_OP, "OUT_AV.05" => "IO_Valve_T03_Chili"."AV-03.05".AUT_OP, "OUT_AV.06" => "IO_Valve_T03_Chili"."AV-03.06".AUT_OP, "OUT_AV.07" => "IO_Valve_T03_Chili"."AV-03.07".AUT_OP, "OUT_AV.08" => "IO_Valve_T03_Chili"."AV-03.08".AUT_OP, "OUT_AV.09" => "IO_Valve_T03_Chili"."AV-03.09".AUT_OP, "OUT_P.01" => "IO Motor MCC Preparation_DB"."P-03.01".AUT_ON, "OUT_P.01-Speed" =>, "OUT_P.02" =>, "OUT_P.02-Speed" =>, "OUT_P.03" =>, "OUT_P.03-Speed" =>, OUT_CIPTank_AVOpen =>, OUT_CIPLine_AVOpen =>)
   END_RUNG
   RUNG wire#powerrail
      Contact( "T-20.00_DB".ChiliAwet_2.QDOSERun )
      Contact( "T-20.00_DB".ChiliAwet_2.V_OPEN )
   END_RUNG wire#w1
   RUNG wire#powerrail
      Contact( "T-21.00_DB".ChiliAwet_2.QDOSERun )
      Contact( "T-21.00_DB".ChiliAwet_2.V_OPEN )
   END_RUNG wire#w1
   RUNG wire#powerrail
      Contact( "T-30.00_DB".ChiliAwet_2.QDOSERun )
      Contact( "T-30.00_DB".ChiliAwet_2.V_OPEN )
   END_RUNG wire#w1
   RUNG wire#powerrail
      Contact( "T-31.00_DB".ChiliAwet_2.QDOSERun )
      Contact( "T-31.00_DB".ChiliAwet_2.V_OPEN )
   END_RUNG wire#w1
   RUNG wire#powerrail
      Contact( "IO_Valve_Blending_DB"."AV-20.10".FB_OPEN )
   END_RUNG wire#w2
   RUNG wire#powerrail
      Contact( "IO_Valve_Blending_DB"."AV-21.10".FB_OPEN )
   END_RUNG wire#w2
   RUNG wire#powerrail
      Contact( "IO_Valve_Blending_DB"."AV-30.10".FB_OPEN )
   END_RUNG wire#w2
   RUNG wire#powerrail
      Contact( "IO_Valve_Blending_DB"."AV-31.10".FB_OPEN )
   END_RUNG wire#w2
   RUNG wire#powerrail
      Contact( "IO_Valve_Blending_DB"."AV-31.56".FB_OPEN )
      Contact( "IO_Valve_Blending_DB"."AV-31.61".FB_OPEN )
   END_RUNG wire#w2
   // the same network as SCL:
   "T-03.01_DB"("IN_FBAV.01" := "IO_Valve_T03_Chili"."AV-03.01".FB_OPEN,   // "BFT_Type1"
                "IN_FBAV.02" := "IO_Valve_T03_Chili"."AV-03.02".FB_OPEN,
                "IN_FBAV.03" := "IO_Valve_T03_Chili"."AV-03.03".FB_OPEN,
                "IN_FBAV.04" := "IO_Valve_T03_Chili"."AV-03.04".FB_OPEN,
                "IN_FBAV.05" := "IO_Valve_T03_Chili"."AV-03.05".FB_OPEN,
                "IN_FBAV.06" := "IO_Valve_T03_Chili"."AV-03.06".FB_OPEN,
                "IN_FBAV.07" := "IO_Valve_T03_Chili"."AV-03.07".FB_OPEN,
                "IN_FBAV.08" := "IO_Valve_T02_Chili"."AV-02.08".FB_OPEN,
                "IN_FBAV.09" := "IO_Valve_T03_Chili"."AV-03.09".FB_OPEN,
                IN_LT01 := "IO Analog Preparation_DB"."LT-03.01".QOUT,
                "IN_FBP.01" := "IO Motor MCC Preparation_DB"."P-03.01".FB_ON,
                "IN_P.01-Speed" := "IO Motor MCC Preparation_DB"."P-03.01".QAct_Speed,
                "IN_FBP.03" := "IO Motor MCC Preparation_DB"."P-03.03".FB_ON,
                "IN_P.03-Speed" := "IO Motor MCC Preparation_DB"."P-03.03".QAct_Speed,
                CIPPulse := "Timer 5S/30s",
                LineTrf_OK := ("T-20.00_DB".ChiliAwet_2.QDOSERun AND "T-20.00_DB".ChiliAwet_2.V_OPEN) OR ("T-21.00_DB".ChiliAwet_2.QDOSERun AND "T-21.00_DB".ChiliAwet_2.V_OPEN) OR ("T-30.00_DB".ChiliAwet_2.QDOSERun AND "T-30.00_DB".ChiliAwet_2.V_OPEN) OR ("T-31.00_DB".ChiliAwet_2.QDOSERun AND "T-31.00_DB".ChiliAwet_2.V_OPEN),
                LineFlush_OK := "IO_Valve_Blending_DB"."AV-20.10".FB_OPEN OR "IO_Valve_Blending_DB"."AV-21.10".FB_OPEN OR "IO_Valve_Blending_DB"."AV-30.10".FB_OPEN OR "IO_Valve_Blending_DB"."AV-31.10".FB_OPEN OR ("IO_Valve_Blending_DB"."AV-31.56".FB_OPEN AND "IO_Valve_Blending_DB"."AV-31.61".FB_OPEN),
                Loading_Busy := "T-04.01_DB".State.Tank_inloading,
                "OUT_AV.01" => "IO_Valve_T03_Chili"."AV-03.01".AUT_OP,
                "OUT_AV.02" => "IO_Valve_T03_Chili"."AV-03.02".AUT_OP,
                "OUT_AV.03" => "IO_Valve_T03_Chili"."AV-03.03".AUT_OP,
                "OUT_AV.04" => "IO_Valve_T03_Chili"."AV-03.04".AUT_OP,
                "OUT_AV.05" => "IO_Valve_T03_Chili"."AV-03.05".AUT_OP,
                "OUT_AV.06" => "IO_Valve_T03_Chili"."AV-03.06".AUT_OP,
                "OUT_AV.07" => "IO_Valve_T03_Chili"."AV-03.07".AUT_OP,
                "OUT_AV.08" => "IO_Valve_T03_Chili"."AV-03.08".AUT_OP,
                "OUT_AV.09" => "IO_Valve_T03_Chili"."AV-03.09".AUT_OP,
                "OUT_P.01" => "IO Motor MCC Preparation_DB"."P-03.01".AUT_ON);
END_REGION

REGION Network 14: Dose ON OFF T-04.01 Chili Awetan 3
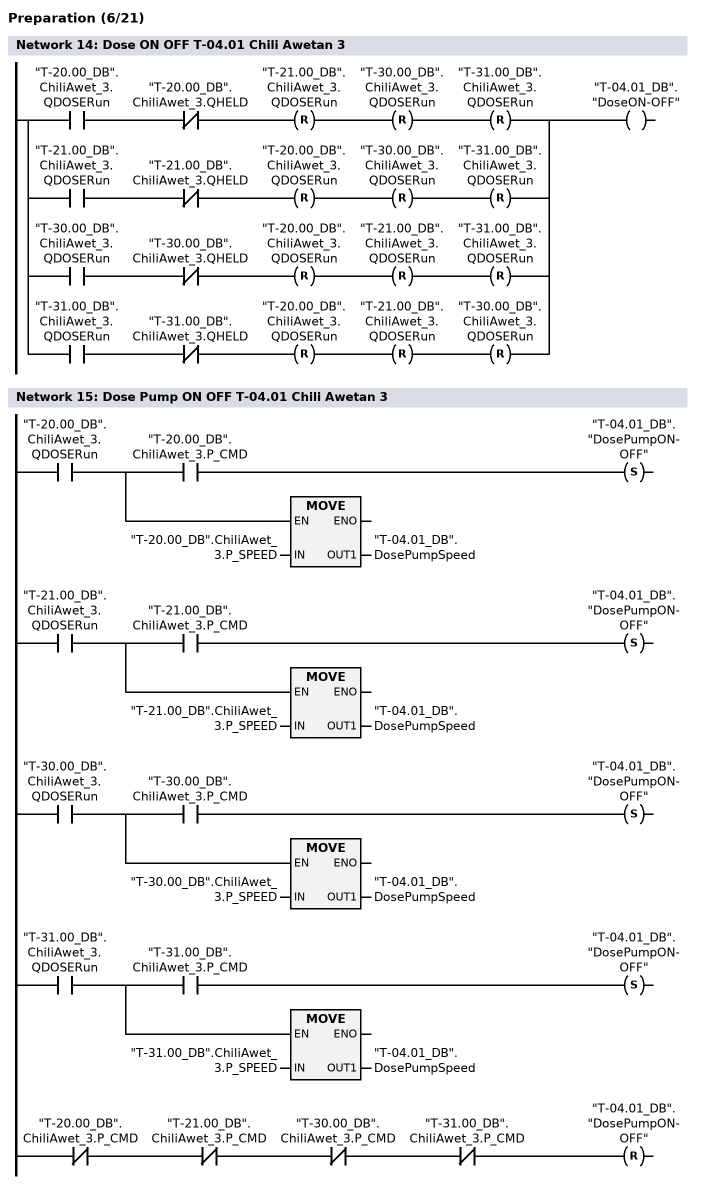
   RUNG wire#powerrail
      Contact( "T-20.00_DB".ChiliAwet_3.QDOSERun )
      I_Contact( "T-20.00_DB".ChiliAwet_3.QHELD )
      R_Coil( "T-21.00_DB".ChiliAwet_3.QDOSERun )
      R_Coil( "T-30.00_DB".ChiliAwet_3.QDOSERun )
      R_Coil( "T-31.00_DB".ChiliAwet_3.QDOSERun )
      wire#w1
      Coil( "T-04.01_DB"."DoseON-OFF" )
   END_RUNG
   RUNG wire#powerrail
      Contact( "T-21.00_DB".ChiliAwet_3.QDOSERun )
      I_Contact( "T-21.00_DB".ChiliAwet_3.QHELD )
      R_Coil( "T-20.00_DB".ChiliAwet_3.QDOSERun )
      R_Coil( "T-30.00_DB".ChiliAwet_3.QDOSERun )
      R_Coil( "T-31.00_DB".ChiliAwet_3.QDOSERun )
   END_RUNG wire#w1
   RUNG wire#powerrail
      Contact( "T-30.00_DB".ChiliAwet_3.QDOSERun )
      I_Contact( "T-30.00_DB".ChiliAwet_3.QHELD )
      R_Coil( "T-20.00_DB".ChiliAwet_3.QDOSERun )
      R_Coil( "T-21.00_DB".ChiliAwet_3.QDOSERun )
      R_Coil( "T-31.00_DB".ChiliAwet_3.QDOSERun )
   END_RUNG wire#w1
   RUNG wire#powerrail
      Contact( "T-31.00_DB".ChiliAwet_3.QDOSERun )
      I_Contact( "T-31.00_DB".ChiliAwet_3.QHELD )
      R_Coil( "T-20.00_DB".ChiliAwet_3.QDOSERun )
      R_Coil( "T-21.00_DB".ChiliAwet_3.QDOSERun )
      R_Coil( "T-30.00_DB".ChiliAwet_3.QDOSERun )
   END_RUNG wire#w1
   // the same network as SCL:
   #_w1 := "T-20.00_DB".ChiliAwet_3.QDOSERun AND NOT "T-20.00_DB".ChiliAwet_3.QHELD;
   IF #_w1 THEN
       "T-21.00_DB".ChiliAwet_3.QDOSERun := FALSE;
       "T-30.00_DB".ChiliAwet_3.QDOSERun := FALSE;
       "T-31.00_DB".ChiliAwet_3.QDOSERun := FALSE;
   END_IF;
   #_w2 := "T-21.00_DB".ChiliAwet_3.QDOSERun AND NOT "T-21.00_DB".ChiliAwet_3.QHELD;
   IF #_w2 THEN
       "T-20.00_DB".ChiliAwet_3.QDOSERun := FALSE;
       "T-30.00_DB".ChiliAwet_3.QDOSERun := FALSE;
       "T-31.00_DB".ChiliAwet_3.QDOSERun := FALSE;
   END_IF;
   #_w3 := "T-30.00_DB".ChiliAwet_3.QDOSERun AND NOT "T-30.00_DB".ChiliAwet_3.QHELD;
   IF #_w3 THEN
       "T-20.00_DB".ChiliAwet_3.QDOSERun := FALSE;
       "T-21.00_DB".ChiliAwet_3.QDOSERun := FALSE;
       "T-31.00_DB".ChiliAwet_3.QDOSERun := FALSE;
   END_IF;
   #_w4 := "T-31.00_DB".ChiliAwet_3.QDOSERun AND NOT "T-31.00_DB".ChiliAwet_3.QHELD;
   IF #_w4 THEN
       "T-20.00_DB".ChiliAwet_3.QDOSERun := FALSE;
       "T-21.00_DB".ChiliAwet_3.QDOSERun := FALSE;
       "T-30.00_DB".ChiliAwet_3.QDOSERun := FALSE;
   END_IF;
   "T-04.01_DB"."DoseON-OFF" := #_w1 OR #_w2 OR #_w3 OR #_w4;
END_REGION

REGION Network 15: Dose Pump ON OFF T-04.01 Chili Awetan 3
   RUNG wire#powerrail
      Contact( "T-20.00_DB".ChiliAwet_3.QDOSERun )
      wire#w1
      Contact( "T-20.00_DB".ChiliAwet_3.P_CMD )
      S_Coil( "T-04.01_DB"."DosePumpON-OFF" )
   END_RUNG
   RUNG wire#w1
      Move(in := "T-20.00_DB".ChiliAwet_3.P_SPEED, out1 => "T-04.01_DB".DosePumpSpeed)
   END_RUNG
   RUNG wire#powerrail
      Contact( "T-21.00_DB".ChiliAwet_3.QDOSERun )
      wire#w2
      Contact( "T-21.00_DB".ChiliAwet_3.P_CMD )
      S_Coil( "T-04.01_DB"."DosePumpON-OFF" )
   END_RUNG
   RUNG wire#w2
      Move(in := "T-21.00_DB".ChiliAwet_3.P_SPEED, out1 => "T-04.01_DB".DosePumpSpeed)
   END_RUNG
   RUNG wire#powerrail
      Contact( "T-30.00_DB".ChiliAwet_3.QDOSERun )
      wire#w3
      Contact( "T-30.00_DB".ChiliAwet_3.P_CMD )
      S_Coil( "T-04.01_DB"."DosePumpON-OFF" )
   END_RUNG
   RUNG wire#w3
      Move(in := "T-30.00_DB".ChiliAwet_3.P_SPEED, out1 => "T-04.01_DB".DosePumpSpeed)
   END_RUNG
   RUNG wire#powerrail
      Contact( "T-31.00_DB".ChiliAwet_3.QDOSERun )
      wire#w4
      Contact( "T-31.00_DB".ChiliAwet_3.P_CMD )
      S_Coil( "T-04.01_DB"."DosePumpON-OFF" )
   END_RUNG
   RUNG wire#w4
      Move(in := "T-31.00_DB".ChiliAwet_3.P_SPEED, out1 => "T-04.01_DB".DosePumpSpeed)
   END_RUNG
   RUNG wire#powerrail
      I_Contact( "T-20.00_DB".ChiliAwet_3.P_CMD )
      I_Contact( "T-21.00_DB".ChiliAwet_3.P_CMD )
      I_Contact( "T-30.00_DB".ChiliAwet_3.P_CMD )
      I_Contact( "T-31.00_DB".ChiliAwet_3.P_CMD )
      R_Coil( "T-04.01_DB"."DosePumpON-OFF" )
   END_RUNG
   // the same network as SCL:
   IF "T-20.00_DB".ChiliAwet_3.QDOSERun AND "T-20.00_DB".ChiliAwet_3.P_CMD THEN
       "T-04.01_DB"."DosePumpON-OFF" := TRUE;
   END_IF;
   IF "T-20.00_DB".ChiliAwet_3.QDOSERun THEN
       "T-04.01_DB".DosePumpSpeed := "T-20.00_DB".ChiliAwet_3.P_SPEED;
   END_IF;
   IF "T-21.00_DB".ChiliAwet_3.QDOSERun AND "T-21.00_DB".ChiliAwet_3.P_CMD THEN
       "T-04.01_DB"."DosePumpON-OFF" := TRUE;
   END_IF;
   IF "T-21.00_DB".ChiliAwet_3.QDOSERun THEN
       "T-04.01_DB".DosePumpSpeed := "T-21.00_DB".ChiliAwet_3.P_SPEED;
   END_IF;
   IF "T-30.00_DB".ChiliAwet_3.QDOSERun AND "T-30.00_DB".ChiliAwet_3.P_CMD THEN
       "T-04.01_DB"."DosePumpON-OFF" := TRUE;
   END_IF;
   IF "T-30.00_DB".ChiliAwet_3.QDOSERun THEN
       "T-04.01_DB".DosePumpSpeed := "T-30.00_DB".ChiliAwet_3.P_SPEED;
   END_IF;
   IF "T-31.00_DB".ChiliAwet_3.QDOSERun AND "T-31.00_DB".ChiliAwet_3.P_CMD THEN
       "T-04.01_DB"."DosePumpON-OFF" := TRUE;
   END_IF;
   IF "T-31.00_DB".ChiliAwet_3.QDOSERun THEN
       "T-04.01_DB".DosePumpSpeed := "T-31.00_DB".ChiliAwet_3.P_SPEED;
   END_IF;
   IF NOT "T-20.00_DB".ChiliAwet_3.P_CMD AND NOT "T-21.00_DB".ChiliAwet_3.P_CMD AND NOT "T-30.00_DB".ChiliAwet_3.P_CMD AND NOT "T-31.00_DB".ChiliAwet_3.P_CMD THEN
       "T-04.01_DB"."DosePumpON-OFF" := FALSE;
   END_IF;
END_REGION

REGION Network 16: T-04.01 Buffer Tank Chili Awetan
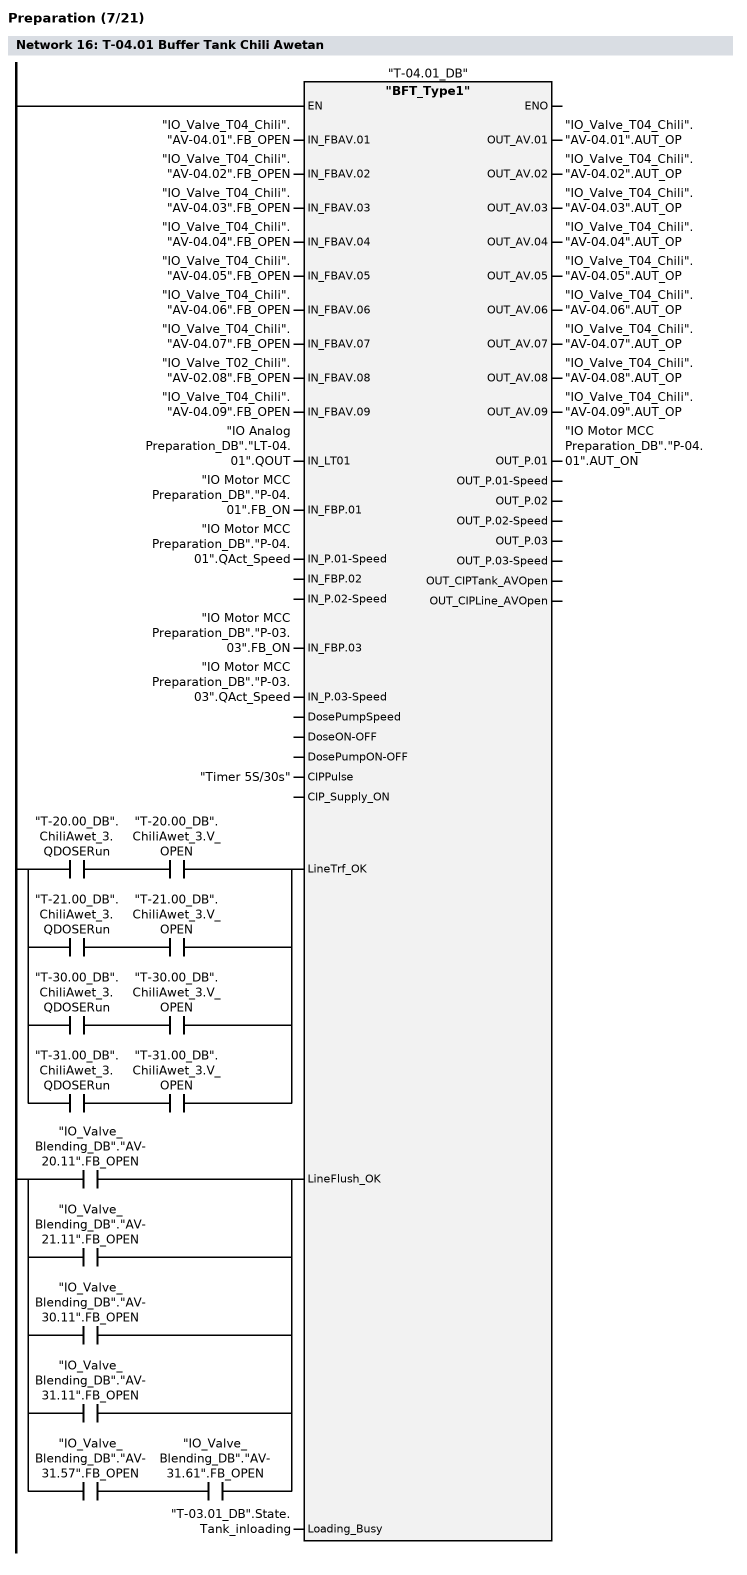
   RUNG wire#powerrail
      "T-04.01_DB"(LineTrf_OK := wire#w1, LineFlush_OK := wire#w2, "IN_FBAV.01" := "IO_Valve_T04_Chili"."AV-04.01".FB_OPEN, "IN_FBAV.02" := "IO_Valve_T04_Chili"."AV-04.02".FB_OPEN, "IN_FBAV.03" := "IO_Valve_T04_Chili"."AV-04.03".FB_OPEN, "IN_FBAV.04" := "IO_Valve_T04_Chili"."AV-04.04".FB_OPEN, "IN_FBAV.05" := "IO_Valve_T04_Chili"."AV-04.05".FB_OPEN, "IN_FBAV.06" := "IO_Valve_T04_Chili"."AV-04.06".FB_OPEN, "IN_FBAV.07" := "IO_Valve_T04_Chili"."AV-04.07".FB_OPEN, "IN_FBAV.08" := "IO_Valve_T02_Chili"."AV-02.08".FB_OPEN, "IN_FBAV.09" := "IO_Valve_T04_Chili"."AV-04.09".FB_OPEN, IN_LT01 := "IO Analog Preparation_DB"."LT-04.01".QOUT, "IN_FBP.01" := "IO Motor MCC Preparation_DB"."P-04.01".FB_ON, "IN_P.01-Speed" := "IO Motor MCC Preparation_DB"."P-04.01".QAct_Speed, "IN_FBP.02" :=, "IN_P.02-Speed" :=, "IN_FBP.03" := "IO Motor MCC Preparation_DB"."P-03.03".FB_ON, "IN_P.03-Speed" := "IO Motor MCC Preparation_DB"."P-03.03".QAct_Speed, DosePumpSpeed :=, "DoseON-OFF" :=, "DosePumpON-OFF" :=, CIPPulse := "Timer 5S/30s", CIP_Supply_ON :=, Loading_Busy := "T-03.01_DB".State.Tank_inloading, "OUT_AV.01" => "IO_Valve_T04_Chili"."AV-04.01".AUT_OP, "OUT_AV.02" => "IO_Valve_T04_Chili"."AV-04.02".AUT_OP, "OUT_AV.03" => "IO_Valve_T04_Chili"."AV-04.03".AUT_OP, "OUT_AV.04" => "IO_Valve_T04_Chili"."AV-04.04".AUT_OP, "OUT_AV.05" => "IO_Valve_T04_Chili"."AV-04.05".AUT_OP, "OUT_AV.06" => "IO_Valve_T04_Chili"."AV-04.06".AUT_OP, "OUT_AV.07" => "IO_Valve_T04_Chili"."AV-04.07".AUT_OP, "OUT_AV.08" => "IO_Valve_T04_Chili"."AV-04.08".AUT_OP, "OUT_AV.09" => "IO_Valve_T04_Chili"."AV-04.09".AUT_OP, "OUT_P.01" => "IO Motor MCC Preparation_DB"."P-04.01".AUT_ON, "OUT_P.01-Speed" =>, "OUT_P.02" =>, "OUT_P.02-Speed" =>, "OUT_P.03" =>, "OUT_P.03-Speed" =>, OUT_CIPTank_AVOpen =>, OUT_CIPLine_AVOpen =>)
   END_RUNG
   RUNG wire#powerrail
      Contact( "T-20.00_DB".ChiliAwet_3.QDOSERun )
      Contact( "T-20.00_DB".ChiliAwet_3.V_OPEN )
   END_RUNG wire#w1
   RUNG wire#powerrail
      Contact( "T-21.00_DB".ChiliAwet_3.QDOSERun )
      Contact( "T-21.00_DB".ChiliAwet_3.V_OPEN )
   END_RUNG wire#w1
   RUNG wire#powerrail
      Contact( "T-30.00_DB".ChiliAwet_3.QDOSERun )
      Contact( "T-30.00_DB".ChiliAwet_3.V_OPEN )
   END_RUNG wire#w1
   RUNG wire#powerrail
      Contact( "T-31.00_DB".ChiliAwet_3.QDOSERun )
      Contact( "T-31.00_DB".ChiliAwet_3.V_OPEN )
   END_RUNG wire#w1
   RUNG wire#powerrail
      Contact( "IO_Valve_Blending_DB"."AV-20.11".FB_OPEN )
   END_RUNG wire#w2
   RUNG wire#powerrail
      Contact( "IO_Valve_Blending_DB"."AV-21.11".FB_OPEN )
   END_RUNG wire#w2
   RUNG wire#powerrail
      Contact( "IO_Valve_Blending_DB"."AV-30.11".FB_OPEN )
   END_RUNG wire#w2
   RUNG wire#powerrail
      Contact( "IO_Valve_Blending_DB"."AV-31.11".FB_OPEN )
   END_RUNG wire#w2
   RUNG wire#powerrail
      Contact( "IO_Valve_Blending_DB"."AV-31.57".FB_OPEN )
      Contact( "IO_Valve_Blending_DB"."AV-31.61".FB_OPEN )
   END_RUNG wire#w2
   // the same network as SCL:
   "T-04.01_DB"("IN_FBAV.01" := "IO_Valve_T04_Chili"."AV-04.01".FB_OPEN,   // "BFT_Type1"
                "IN_FBAV.02" := "IO_Valve_T04_Chili"."AV-04.02".FB_OPEN,
                "IN_FBAV.03" := "IO_Valve_T04_Chili"."AV-04.03".FB_OPEN,
                "IN_FBAV.04" := "IO_Valve_T04_Chili"."AV-04.04".FB_OPEN,
                "IN_FBAV.05" := "IO_Valve_T04_Chili"."AV-04.05".FB_OPEN,
                "IN_FBAV.06" := "IO_Valve_T04_Chili"."AV-04.06".FB_OPEN,
                "IN_FBAV.07" := "IO_Valve_T04_Chili"."AV-04.07".FB_OPEN,
                "IN_FBAV.08" := "IO_Valve_T02_Chili"."AV-02.08".FB_OPEN,
                "IN_FBAV.09" := "IO_Valve_T04_Chili"."AV-04.09".FB_OPEN,
                IN_LT01 := "IO Analog Preparation_DB"."LT-04.01".QOUT,
                "IN_FBP.01" := "IO Motor MCC Preparation_DB"."P-04.01".FB_ON,
                "IN_P.01-Speed" := "IO Motor MCC Preparation_DB"."P-04.01".QAct_Speed,
                "IN_FBP.03" := "IO Motor MCC Preparation_DB"."P-03.03".FB_ON,
                "IN_P.03-Speed" := "IO Motor MCC Preparation_DB"."P-03.03".QAct_Speed,
                CIPPulse := "Timer 5S/30s",
                LineTrf_OK := ("T-20.00_DB".ChiliAwet_3.QDOSERun AND "T-20.00_DB".ChiliAwet_3.V_OPEN) OR ("T-21.00_DB".ChiliAwet_3.QDOSERun AND "T-21.00_DB".ChiliAwet_3.V_OPEN) OR ("T-30.00_DB".ChiliAwet_3.QDOSERun AND "T-30.00_DB".ChiliAwet_3.V_OPEN) OR ("T-31.00_DB".ChiliAwet_3.QDOSERun AND "T-31.00_DB".ChiliAwet_3.V_OPEN),
                LineFlush_OK := "IO_Valve_Blending_DB"."AV-20.11".FB_OPEN OR "IO_Valve_Blending_DB"."AV-21.11".FB_OPEN OR "IO_Valve_Blending_DB"."AV-30.11".FB_OPEN OR "IO_Valve_Blending_DB"."AV-31.11".FB_OPEN OR ("IO_Valve_Blending_DB"."AV-31.57".FB_OPEN AND "IO_Valve_Blending_DB"."AV-31.61".FB_OPEN),
                Loading_Busy := "T-03.01_DB".State.Tank_inloading,
                "OUT_AV.01" => "IO_Valve_T04_Chili"."AV-04.01".AUT_OP,
                "OUT_AV.02" => "IO_Valve_T04_Chili"."AV-04.02".AUT_OP,
                "OUT_AV.03" => "IO_Valve_T04_Chili"."AV-04.03".AUT_OP,
                "OUT_AV.04" => "IO_Valve_T04_Chili"."AV-04.04".AUT_OP,
                "OUT_AV.05" => "IO_Valve_T04_Chili"."AV-04.05".AUT_OP,
                "OUT_AV.06" => "IO_Valve_T04_Chili"."AV-04.06".AUT_OP,
                "OUT_AV.07" => "IO_Valve_T04_Chili"."AV-04.07".AUT_OP,
                "OUT_AV.08" => "IO_Valve_T04_Chili"."AV-04.08".AUT_OP,
                "OUT_AV.09" => "IO_Valve_T04_Chili"."AV-04.09".AUT_OP,
                "OUT_P.01" => "IO Motor MCC Preparation_DB"."P-04.01".AUT_ON);
END_REGION

REGION Network 17: Inload Pump T-03 and T-04 ( P-03.03 )
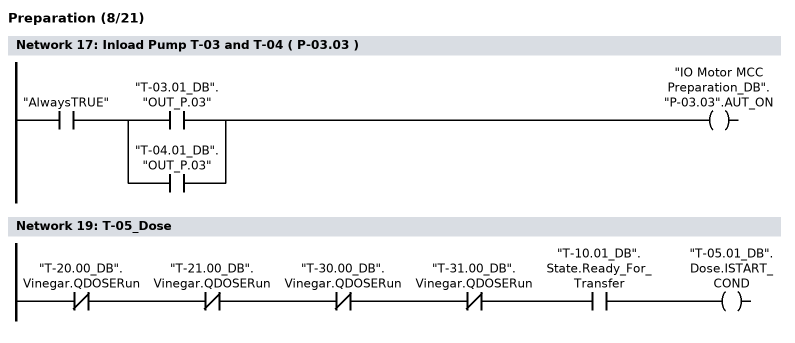
   RUNG wire#powerrail
      Contact( "AlwaysTRUE" )
      wire#w1
      Contact( "T-03.01_DB"."OUT_P.03" )
      wire#w2
      Coil( "IO Motor MCC Preparation_DB"."P-03.03".AUT_ON )
   END_RUNG
   RUNG wire#w1
      Contact( "T-04.01_DB"."OUT_P.03" )
   END_RUNG wire#w2
   // the same network as SCL:
   "IO Motor MCC Preparation_DB"."P-03.03".AUT_ON := "AlwaysTRUE" AND ("T-03.01_DB"."OUT_P.03" OR "T-04.01_DB"."OUT_P.03");
END_REGION

REGION Network 19: T-05_Dose
   RUNG wire#powerrail
      I_Contact( "T-20.00_DB".Vinegar.QDOSERun )
      I_Contact( "T-21.00_DB".Vinegar.QDOSERun )
      I_Contact( "T-30.00_DB".Vinegar.QDOSERun )
      I_Contact( "T-31.00_DB".Vinegar.QDOSERun )
      Contact( "T-10.01_DB".State.Ready_For_Transfer )
      Coil( "T-05.01_DB".Dose.ISTART_COND )
   END_RUNG
   // the same network as SCL:
   "T-05.01_DB".Dose.ISTART_COND := NOT "T-20.00_DB".Vinegar.QDOSERun AND NOT "T-21.00_DB".Vinegar.QDOSERun AND NOT "T-30.00_DB".Vinegar.QDOSERun AND NOT "T-31.00_DB".Vinegar.QDOSERun AND "T-10.01_DB".State.Ready_For_Transfer;
END_REGION

REGION Network 20: T-05.01 Buffer Tank Tomato
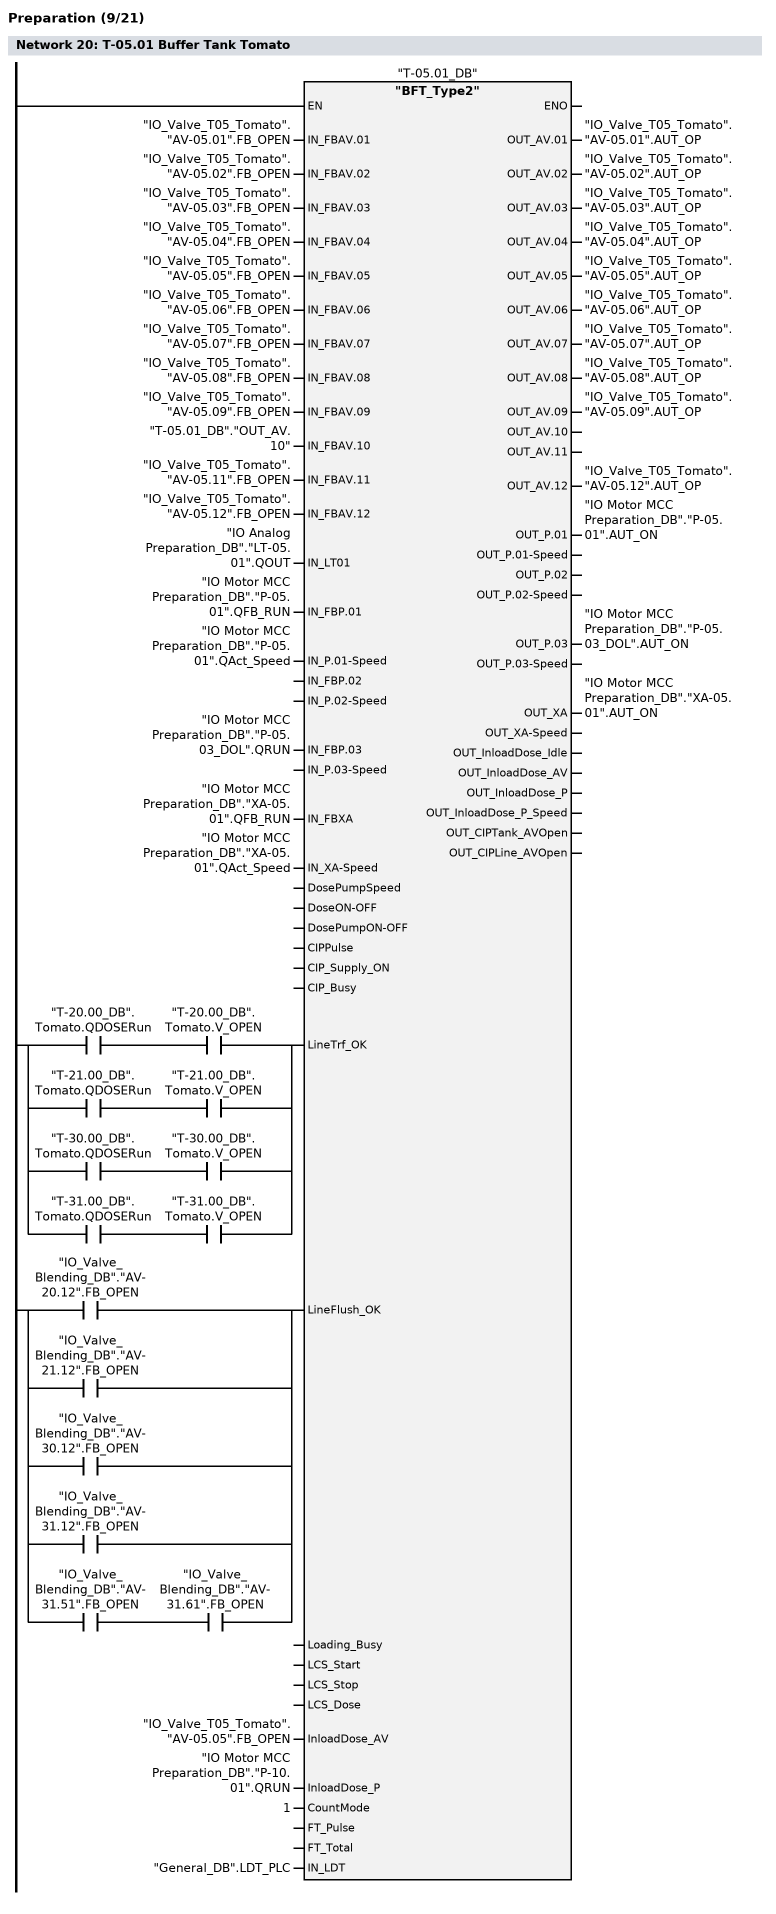
   RUNG wire#powerrail
      "T-05.01_DB"(LineTrf_OK := wire#w1, LineFlush_OK := wire#w2, "IN_FBAV.01" := "IO_Valve_T05_Tomato"."AV-05.01".FB_OPEN, "IN_FBAV.02" := "IO_Valve_T05_Tomato"."AV-05.02".FB_OPEN, "IN_FBAV.03" := "IO_Valve_T05_Tomato"."AV-05.03".FB_OPEN, "IN_FBAV.04" := "IO_Valve_T05_Tomato"."AV-05.04".FB_OPEN, "IN_FBAV.05" := "IO_Valve_T05_Tomato"."AV-05.05".FB_OPEN, "IN_FBAV.06" := "IO_Valve_T05_Tomato"."AV-05.06".FB_OPEN, "IN_FBAV.07" := "IO_Valve_T05_Tomato"."AV-05.07".FB_OPEN, "IN_FBAV.08" := "IO_Valve_T05_Tomato"."AV-05.08".FB_OPEN, "IN_FBAV.09" := "IO_Valve_T05_Tomato"."AV-05.09".FB_OPEN, "IN_FBAV.10" := "T-05.01_DB"."OUT_AV.10", "IN_FBAV.11" := "IO_Valve_T05_Tomato"."AV-05.11".FB_OPEN, "IN_FBAV.12" := "IO_Valve_T05_Tomato"."AV-05.12".FB_OPEN, IN_LT01 := "IO Analog Preparation_DB"."LT-05.01".QOUT, "IN_FBP.01" := "IO Motor MCC Preparation_DB"."P-05.01".QFB_RUN, "IN_P.01-Speed" := "IO Motor MCC Preparation_DB"."P-05.01".QAct_Speed, "IN_FBP.02" :=, "IN_P.02-Speed" :=, "IN_FBP.03" := "IO Motor MCC Preparation_DB"."P-05.03_DOL".QRUN, "IN_P.03-Speed" :=, IN_FBXA := "IO Motor MCC Preparation_DB"."XA-05.01".QFB_RUN, "IN_XA-Speed" := "IO Motor MCC Preparation_DB"."XA-05.01".QAct_Speed, DosePumpSpeed :=, "DoseON-OFF" :=, "DosePumpON-OFF" :=, CIPPulse :=, CIP_Supply_ON :=, CIP_Busy :=, Loading_Busy :=, LCS_Start :=, LCS_Stop :=, LCS_Dose :=, InloadDose_AV := "IO_Valve_T05_Tomato"."AV-05.05".FB_OPEN, InloadDose_P := "IO Motor MCC Preparation_DB"."P-10.01".QRUN, CountMode := 1, FT_Pulse :=, FT_Total :=, IN_LDT := "General_DB".LDT_PLC, "OUT_AV.01" => "IO_Valve_T05_Tomato"."AV-05.01".AUT_OP, "OUT_AV.02" => "IO_Valve_T05_Tomato"."AV-05.02".AUT_OP, "OUT_AV.03" => "IO_Valve_T05_Tomato"."AV-05.03".AUT_OP, "OUT_AV.04" => "IO_Valve_T05_Tomato"."AV-05.04".AUT_OP, "OUT_AV.05" => "IO_Valve_T05_Tomato"."AV-05.05".AUT_OP, "OUT_AV.06" => "IO_Valve_T05_Tomato"."AV-05.06".AUT_OP, "OUT_AV.07" => "IO_Valve_T05_Tomato"."AV-05.07".AUT_OP, "OUT_AV.08" => "IO_Valve_T05_Tomato"."AV-05.08".AUT_OP, "OUT_AV.09" => "IO_Valve_T05_Tomato"."AV-05.09".AUT_OP, "OUT_AV.10" =>, "OUT_AV.11" =>, "OUT_AV.12" => "IO_Valve_T05_Tomato"."AV-05.12".AUT_OP, "OUT_P.01" => "IO Motor MCC Preparation_DB"."P-05.01".AUT_ON, "OUT_P.01-Speed" =>, "OUT_P.02" =>, "OUT_P.02-Speed" =>, "OUT_P.03" => "IO Motor MCC Preparation_DB"."P-05.03_DOL".AUT_ON, "OUT_P.03-Speed" =>, OUT_XA => "IO Motor MCC Preparation_DB"."XA-05.01".AUT_ON, "OUT_XA-Speed" =>, OUT_InloadDose_Idle =>, OUT_InloadDose_AV =>, OUT_InloadDose_P =>, OUT_InloadDose_P_Speed =>, OUT_CIPTank_AVOpen =>, OUT_CIPLine_AVOpen =>)
   END_RUNG
   RUNG wire#powerrail
      Contact( "T-20.00_DB".Tomato.QDOSERun )
      Contact( "T-20.00_DB".Tomato.V_OPEN )
   END_RUNG wire#w1
   RUNG wire#powerrail
      Contact( "T-21.00_DB".Tomato.QDOSERun )
      Contact( "T-21.00_DB".Tomato.V_OPEN )
   END_RUNG wire#w1
   RUNG wire#powerrail
      Contact( "T-30.00_DB".Tomato.QDOSERun )
      Contact( "T-30.00_DB".Tomato.V_OPEN )
   END_RUNG wire#w1
   RUNG wire#powerrail
      Contact( "T-31.00_DB".Tomato.QDOSERun )
      Contact( "T-31.00_DB".Tomato.V_OPEN )
   END_RUNG wire#w1
   RUNG wire#powerrail
      Contact( "IO_Valve_Blending_DB"."AV-20.12".FB_OPEN )
   END_RUNG wire#w2
   RUNG wire#powerrail
      Contact( "IO_Valve_Blending_DB"."AV-21.12".FB_OPEN )
   END_RUNG wire#w2
   RUNG wire#powerrail
      Contact( "IO_Valve_Blending_DB"."AV-30.12".FB_OPEN )
   END_RUNG wire#w2
   RUNG wire#powerrail
      Contact( "IO_Valve_Blending_DB"."AV-31.12".FB_OPEN )
   END_RUNG wire#w2
   RUNG wire#powerrail
      Contact( "IO_Valve_Blending_DB"."AV-31.51".FB_OPEN )
      Contact( "IO_Valve_Blending_DB"."AV-31.61".FB_OPEN )
   END_RUNG wire#w2
   // the same network as SCL:
   "T-05.01_DB"("IN_FBAV.01" := "IO_Valve_T05_Tomato"."AV-05.01".FB_OPEN,   // "BFT_Type2"
                "IN_FBAV.02" := "IO_Valve_T05_Tomato"."AV-05.02".FB_OPEN,
                "IN_FBAV.03" := "IO_Valve_T05_Tomato"."AV-05.03".FB_OPEN,
                "IN_FBAV.04" := "IO_Valve_T05_Tomato"."AV-05.04".FB_OPEN,
                "IN_FBAV.05" := "IO_Valve_T05_Tomato"."AV-05.05".FB_OPEN,
                "IN_FBAV.06" := "IO_Valve_T05_Tomato"."AV-05.06".FB_OPEN,
                "IN_FBAV.07" := "IO_Valve_T05_Tomato"."AV-05.07".FB_OPEN,
                "IN_FBAV.08" := "IO_Valve_T05_Tomato"."AV-05.08".FB_OPEN,
                "IN_FBAV.09" := "IO_Valve_T05_Tomato"."AV-05.09".FB_OPEN,
                "IN_FBAV.10" := "T-05.01_DB"."OUT_AV.10",
                "IN_FBAV.11" := "IO_Valve_T05_Tomato"."AV-05.11".FB_OPEN,
                "IN_FBAV.12" := "IO_Valve_T05_Tomato"."AV-05.12".FB_OPEN,
                IN_LT01 := "IO Analog Preparation_DB"."LT-05.01".QOUT,
                "IN_FBP.01" := "IO Motor MCC Preparation_DB"."P-05.01".QFB_RUN,
                "IN_P.01-Speed" := "IO Motor MCC Preparation_DB"."P-05.01".QAct_Speed,
                "IN_FBP.03" := "IO Motor MCC Preparation_DB"."P-05.03_DOL".QRUN,
                IN_FBXA := "IO Motor MCC Preparation_DB"."XA-05.01".QFB_RUN,
                "IN_XA-Speed" := "IO Motor MCC Preparation_DB"."XA-05.01".QAct_Speed,
                LineTrf_OK := ("T-20.00_DB".Tomato.QDOSERun AND "T-20.00_DB".Tomato.V_OPEN) OR ("T-21.00_DB".Tomato.QDOSERun AND "T-21.00_DB".Tomato.V_OPEN) OR ("T-30.00_DB".Tomato.QDOSERun AND "T-30.00_DB".Tomato.V_OPEN) OR ("T-31.00_DB".Tomato.QDOSERun AND "T-31.00_DB".Tomato.V_OPEN),
                LineFlush_OK := "IO_Valve_Blending_DB"."AV-20.12".FB_OPEN OR "IO_Valve_Blending_DB"."AV-21.12".FB_OPEN OR "IO_Valve_Blending_DB"."AV-30.12".FB_OPEN OR "IO_Valve_Blending_DB"."AV-31.12".FB_OPEN OR ("IO_Valve_Blending_DB"."AV-31.51".FB_OPEN AND "IO_Valve_Blending_DB"."AV-31.61".FB_OPEN),
                InloadDose_AV := "IO_Valve_T05_Tomato"."AV-05.05".FB_OPEN,
                InloadDose_P := "IO Motor MCC Preparation_DB"."P-10.01".QRUN,
                CountMode := 1,
                IN_LDT := "General_DB".LDT_PLC,
                "OUT_AV.01" => "IO_Valve_T05_Tomato"."AV-05.01".AUT_OP,
                "OUT_AV.02" => "IO_Valve_T05_Tomato"."AV-05.02".AUT_OP,
                "OUT_AV.03" => "IO_Valve_T05_Tomato"."AV-05.03".AUT_OP,
                "OUT_AV.04" => "IO_Valve_T05_Tomato"."AV-05.04".AUT_OP,
                "OUT_AV.05" => "IO_Valve_T05_Tomato"."AV-05.05".AUT_OP,
                "OUT_AV.06" => "IO_Valve_T05_Tomato"."AV-05.06".AUT_OP,
                "OUT_AV.07" => "IO_Valve_T05_Tomato"."AV-05.07".AUT_OP,
                "OUT_AV.08" => "IO_Valve_T05_Tomato"."AV-05.08".AUT_OP,
                "OUT_AV.09" => "IO_Valve_T05_Tomato"."AV-05.09".AUT_OP,
                "OUT_AV.12" => "IO_Valve_T05_Tomato"."AV-05.12".AUT_OP,
                "OUT_P.01" => "IO Motor MCC Preparation_DB"."P-05.01".AUT_ON,
                "OUT_P.03" => "IO Motor MCC Preparation_DB"."P-05.03_DOL".AUT_ON,
                OUT_XA => "IO Motor MCC Preparation_DB"."XA-05.01".AUT_ON);
END_REGION

REGION Network 22: Dose ON OFF T-06.01 Chili Fresh 1
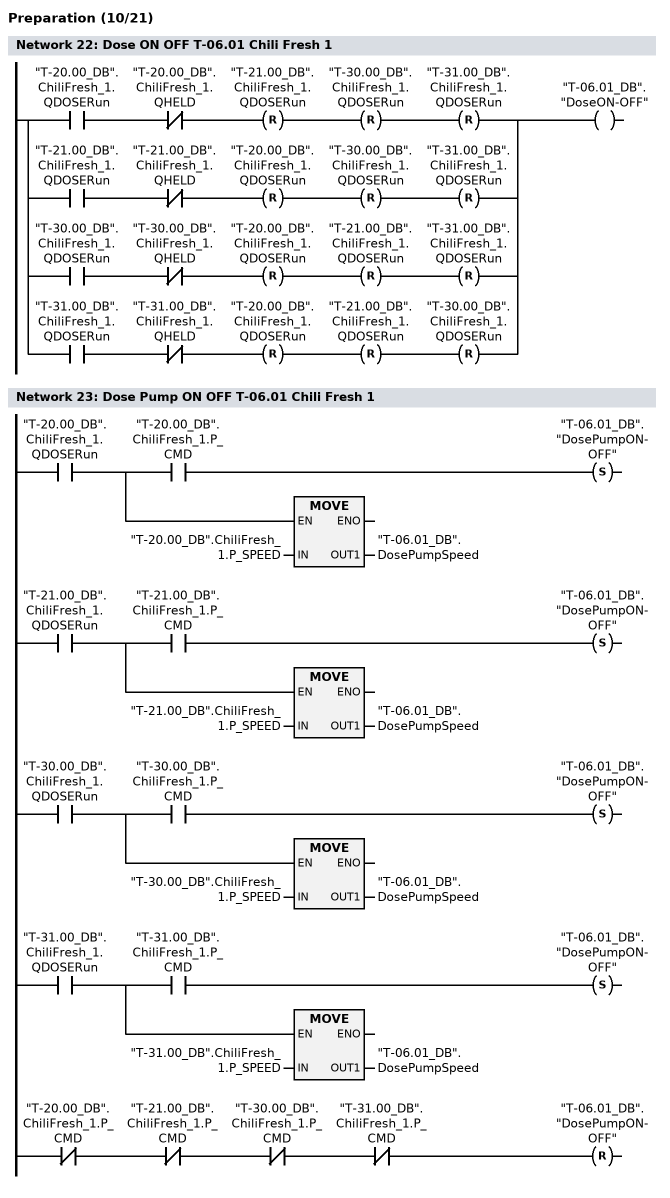
   RUNG wire#powerrail
      Contact( "T-20.00_DB".ChiliFresh_1.QDOSERun )
      I_Contact( "T-20.00_DB".ChiliFresh_1.QHELD )
      R_Coil( "T-21.00_DB".ChiliFresh_1.QDOSERun )
      R_Coil( "T-30.00_DB".ChiliFresh_1.QDOSERun )
      R_Coil( "T-31.00_DB".ChiliFresh_1.QDOSERun )
      wire#w1
      Coil( "T-06.01_DB"."DoseON-OFF" )
   END_RUNG
   RUNG wire#powerrail
      Contact( "T-21.00_DB".ChiliFresh_1.QDOSERun )
      I_Contact( "T-21.00_DB".ChiliFresh_1.QHELD )
      R_Coil( "T-20.00_DB".ChiliFresh_1.QDOSERun )
      R_Coil( "T-30.00_DB".ChiliFresh_1.QDOSERun )
      R_Coil( "T-31.00_DB".ChiliFresh_1.QDOSERun )
   END_RUNG wire#w1
   RUNG wire#powerrail
      Contact( "T-30.00_DB".ChiliFresh_1.QDOSERun )
      I_Contact( "T-30.00_DB".ChiliFresh_1.QHELD )
      R_Coil( "T-20.00_DB".ChiliFresh_1.QDOSERun )
      R_Coil( "T-21.00_DB".ChiliFresh_1.QDOSERun )
      R_Coil( "T-31.00_DB".ChiliFresh_1.QDOSERun )
   END_RUNG wire#w1
   RUNG wire#powerrail
      Contact( "T-31.00_DB".ChiliFresh_1.QDOSERun )
      I_Contact( "T-31.00_DB".ChiliFresh_1.QHELD )
      R_Coil( "T-20.00_DB".ChiliFresh_1.QDOSERun )
      R_Coil( "T-21.00_DB".ChiliFresh_1.QDOSERun )
      R_Coil( "T-30.00_DB".ChiliFresh_1.QDOSERun )
   END_RUNG wire#w1
   // the same network as SCL:
   #_w1 := "T-20.00_DB".ChiliFresh_1.QDOSERun AND NOT "T-20.00_DB".ChiliFresh_1.QHELD;
   IF #_w1 THEN
       "T-21.00_DB".ChiliFresh_1.QDOSERun := FALSE;
       "T-30.00_DB".ChiliFresh_1.QDOSERun := FALSE;
       "T-31.00_DB".ChiliFresh_1.QDOSERun := FALSE;
   END_IF;
   #_w2 := "T-21.00_DB".ChiliFresh_1.QDOSERun AND NOT "T-21.00_DB".ChiliFresh_1.QHELD;
   IF #_w2 THEN
       "T-20.00_DB".ChiliFresh_1.QDOSERun := FALSE;
       "T-30.00_DB".ChiliFresh_1.QDOSERun := FALSE;
       "T-31.00_DB".ChiliFresh_1.QDOSERun := FALSE;
   END_IF;
   #_w3 := "T-30.00_DB".ChiliFresh_1.QDOSERun AND NOT "T-30.00_DB".ChiliFresh_1.QHELD;
   IF #_w3 THEN
       "T-20.00_DB".ChiliFresh_1.QDOSERun := FALSE;
       "T-21.00_DB".ChiliFresh_1.QDOSERun := FALSE;
       "T-31.00_DB".ChiliFresh_1.QDOSERun := FALSE;
   END_IF;
   #_w4 := "T-31.00_DB".ChiliFresh_1.QDOSERun AND NOT "T-31.00_DB".ChiliFresh_1.QHELD;
   IF #_w4 THEN
       "T-20.00_DB".ChiliFresh_1.QDOSERun := FALSE;
       "T-21.00_DB".ChiliFresh_1.QDOSERun := FALSE;
       "T-30.00_DB".ChiliFresh_1.QDOSERun := FALSE;
   END_IF;
   "T-06.01_DB"."DoseON-OFF" := #_w1 OR #_w2 OR #_w3 OR #_w4;
END_REGION

REGION Network 23: Dose Pump ON OFF T-06.01 Chili Fresh 1
   RUNG wire#powerrail
      Contact( "T-20.00_DB".ChiliFresh_1.QDOSERun )
      wire#w1
      Contact( "T-20.00_DB".ChiliFresh_1.P_CMD )
      S_Coil( "T-06.01_DB"."DosePumpON-OFF" )
   END_RUNG
   RUNG wire#w1
      Move(in := "T-20.00_DB".ChiliFresh_1.P_SPEED, out1 => "T-06.01_DB".DosePumpSpeed)
   END_RUNG
   RUNG wire#powerrail
      Contact( "T-21.00_DB".ChiliFresh_1.QDOSERun )
      wire#w2
      Contact( "T-21.00_DB".ChiliFresh_1.P_CMD )
      S_Coil( "T-06.01_DB"."DosePumpON-OFF" )
   END_RUNG
   RUNG wire#w2
      Move(in := "T-21.00_DB".ChiliFresh_1.P_SPEED, out1 => "T-06.01_DB".DosePumpSpeed)
   END_RUNG
   RUNG wire#powerrail
      Contact( "T-30.00_DB".ChiliFresh_1.QDOSERun )
      wire#w3
      Contact( "T-30.00_DB".ChiliFresh_1.P_CMD )
      S_Coil( "T-06.01_DB"."DosePumpON-OFF" )
   END_RUNG
   RUNG wire#w3
      Move(in := "T-30.00_DB".ChiliFresh_1.P_SPEED, out1 => "T-06.01_DB".DosePumpSpeed)
   END_RUNG
   RUNG wire#powerrail
      Contact( "T-31.00_DB".ChiliFresh_1.QDOSERun )
      wire#w4
      Contact( "T-31.00_DB".ChiliFresh_1.P_CMD )
      S_Coil( "T-06.01_DB"."DosePumpON-OFF" )
   END_RUNG
   RUNG wire#w4
      Move(in := "T-31.00_DB".ChiliFresh_1.P_SPEED, out1 => "T-06.01_DB".DosePumpSpeed)
   END_RUNG
   RUNG wire#powerrail
      I_Contact( "T-20.00_DB".ChiliFresh_1.P_CMD )
      I_Contact( "T-21.00_DB".ChiliFresh_1.P_CMD )
      I_Contact( "T-30.00_DB".ChiliFresh_1.P_CMD )
      I_Contact( "T-31.00_DB".ChiliFresh_1.P_CMD )
      R_Coil( "T-06.01_DB"."DosePumpON-OFF" )
   END_RUNG
   // the same network as SCL:
   IF "T-20.00_DB".ChiliFresh_1.QDOSERun AND "T-20.00_DB".ChiliFresh_1.P_CMD THEN
       "T-06.01_DB"."DosePumpON-OFF" := TRUE;
   END_IF;
   IF "T-20.00_DB".ChiliFresh_1.QDOSERun THEN
       "T-06.01_DB".DosePumpSpeed := "T-20.00_DB".ChiliFresh_1.P_SPEED;
   END_IF;
   IF "T-21.00_DB".ChiliFresh_1.QDOSERun AND "T-21.00_DB".ChiliFresh_1.P_CMD THEN
       "T-06.01_DB"."DosePumpON-OFF" := TRUE;
   END_IF;
   IF "T-21.00_DB".ChiliFresh_1.QDOSERun THEN
       "T-06.01_DB".DosePumpSpeed := "T-21.00_DB".ChiliFresh_1.P_SPEED;
   END_IF;
   IF "T-30.00_DB".ChiliFresh_1.QDOSERun AND "T-30.00_DB".ChiliFresh_1.P_CMD THEN
       "T-06.01_DB"."DosePumpON-OFF" := TRUE;
   END_IF;
   IF "T-30.00_DB".ChiliFresh_1.QDOSERun THEN
       "T-06.01_DB".DosePumpSpeed := "T-30.00_DB".ChiliFresh_1.P_SPEED;
   END_IF;
   IF "T-31.00_DB".ChiliFresh_1.QDOSERun AND "T-31.00_DB".ChiliFresh_1.P_CMD THEN
       "T-06.01_DB"."DosePumpON-OFF" := TRUE;
   END_IF;
   IF "T-31.00_DB".ChiliFresh_1.QDOSERun THEN
       "T-06.01_DB".DosePumpSpeed := "T-31.00_DB".ChiliFresh_1.P_SPEED;
   END_IF;
   IF NOT "T-20.00_DB".ChiliFresh_1.P_CMD AND NOT "T-21.00_DB".ChiliFresh_1.P_CMD AND NOT "T-30.00_DB".ChiliFresh_1.P_CMD AND NOT "T-31.00_DB".ChiliFresh_1.P_CMD THEN
       "T-06.01_DB"."DosePumpON-OFF" := FALSE;
   END_IF;
END_REGION

REGION Network 24: T-06.01 Buffer Tank Chili Fresh
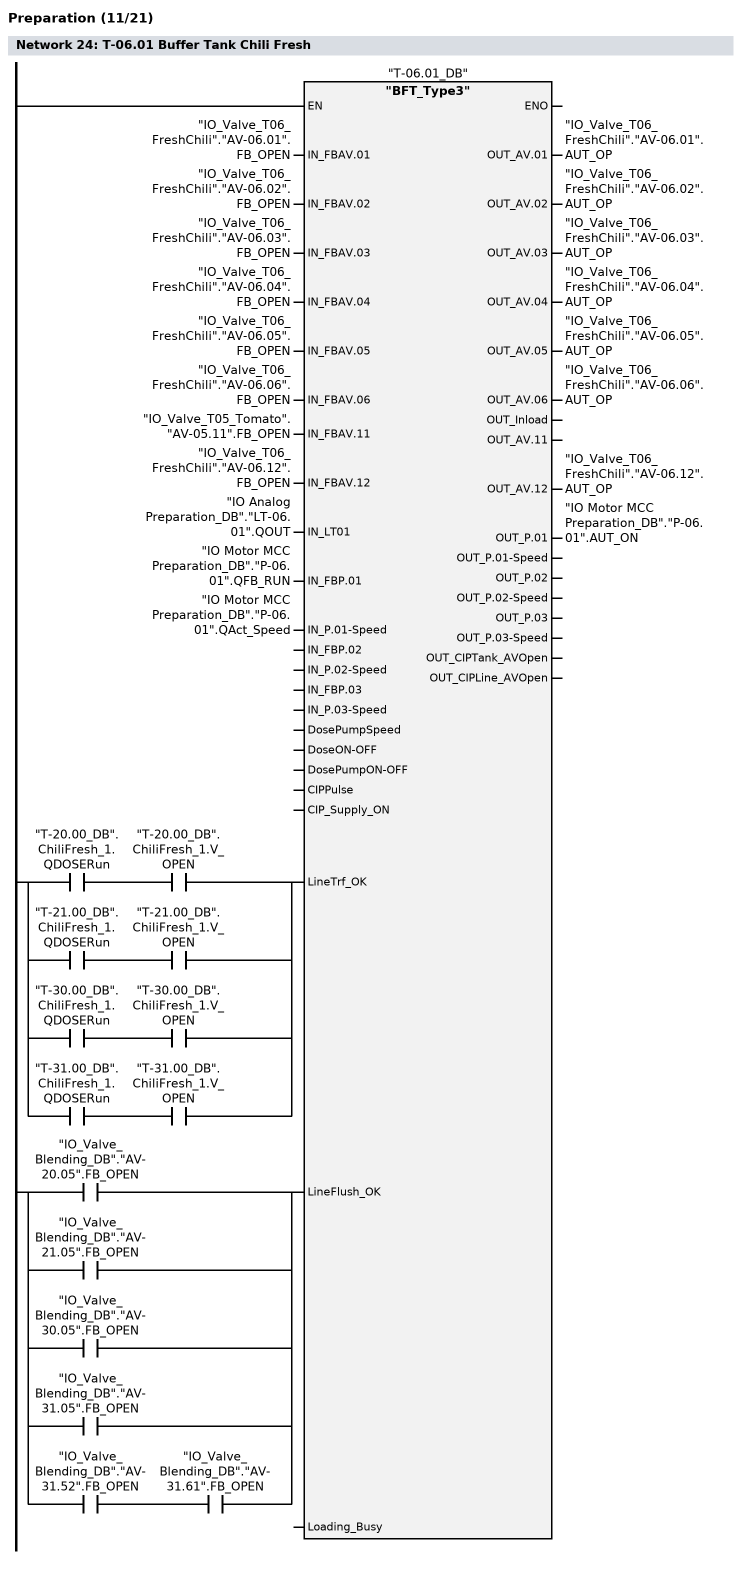
   RUNG wire#powerrail
      "T-06.01_DB"(LineTrf_OK := wire#w1, LineFlush_OK := wire#w2, "IN_FBAV.01" := "IO_Valve_T06_FreshChili"."AV-06.01".FB_OPEN, "IN_FBAV.02" := "IO_Valve_T06_FreshChili"."AV-06.02".FB_OPEN, "IN_FBAV.03" := "IO_Valve_T06_FreshChili"."AV-06.03".FB_OPEN, "IN_FBAV.04" := "IO_Valve_T06_FreshChili"."AV-06.04".FB_OPEN, "IN_FBAV.05" := "IO_Valve_T06_FreshChili"."AV-06.05".FB_OPEN, "IN_FBAV.06" := "IO_Valve_T06_FreshChili"."AV-06.06".FB_OPEN, "IN_FBAV.11" := "IO_Valve_T05_Tomato"."AV-05.11".FB_OPEN, "IN_FBAV.12" := "IO_Valve_T06_FreshChili"."AV-06.12".FB_OPEN, IN_LT01 := "IO Analog Preparation_DB"."LT-06.01".QOUT, "IN_FBP.01" := "IO Motor MCC Preparation_DB"."P-06.01".QFB_RUN, "IN_P.01-Speed" := "IO Motor MCC Preparation_DB"."P-06.01".QAct_Speed, "IN_FBP.02" :=, "IN_P.02-Speed" :=, "IN_FBP.03" :=, "IN_P.03-Speed" :=, DosePumpSpeed :=, "DoseON-OFF" :=, "DosePumpON-OFF" :=, CIPPulse :=, CIP_Supply_ON :=, Loading_Busy :=, "OUT_AV.01" => "IO_Valve_T06_FreshChili"."AV-06.01".AUT_OP, "OUT_AV.02" => "IO_Valve_T06_FreshChili"."AV-06.02".AUT_OP, "OUT_AV.03" => "IO_Valve_T06_FreshChili"."AV-06.03".AUT_OP, "OUT_AV.04" => "IO_Valve_T06_FreshChili"."AV-06.04".AUT_OP, "OUT_AV.05" => "IO_Valve_T06_FreshChili"."AV-06.05".AUT_OP, "OUT_AV.06" => "IO_Valve_T06_FreshChili"."AV-06.06".AUT_OP, OUT_Inload =>, "OUT_AV.11" =>, "OUT_AV.12" => "IO_Valve_T06_FreshChili"."AV-06.12".AUT_OP, "OUT_P.01" => "IO Motor MCC Preparation_DB"."P-06.01".AUT_ON, "OUT_P.01-Speed" =>, "OUT_P.02" =>, "OUT_P.02-Speed" =>, "OUT_P.03" =>, "OUT_P.03-Speed" =>, OUT_CIPTank_AVOpen =>, OUT_CIPLine_AVOpen =>)
   END_RUNG
   RUNG wire#powerrail
      Contact( "T-20.00_DB".ChiliFresh_1.QDOSERun )
      Contact( "T-20.00_DB".ChiliFresh_1.V_OPEN )
   END_RUNG wire#w1
   RUNG wire#powerrail
      Contact( "T-21.00_DB".ChiliFresh_1.QDOSERun )
      Contact( "T-21.00_DB".ChiliFresh_1.V_OPEN )
   END_RUNG wire#w1
   RUNG wire#powerrail
      Contact( "T-30.00_DB".ChiliFresh_1.QDOSERun )
      Contact( "T-30.00_DB".ChiliFresh_1.V_OPEN )
   END_RUNG wire#w1
   RUNG wire#powerrail
      Contact( "T-31.00_DB".ChiliFresh_1.QDOSERun )
      Contact( "T-31.00_DB".ChiliFresh_1.V_OPEN )
   END_RUNG wire#w1
   RUNG wire#powerrail
      Contact( "IO_Valve_Blending_DB"."AV-20.05".FB_OPEN )
   END_RUNG wire#w2
   RUNG wire#powerrail
      Contact( "IO_Valve_Blending_DB"."AV-21.05".FB_OPEN )
   END_RUNG wire#w2
   RUNG wire#powerrail
      Contact( "IO_Valve_Blending_DB"."AV-30.05".FB_OPEN )
   END_RUNG wire#w2
   RUNG wire#powerrail
      Contact( "IO_Valve_Blending_DB"."AV-31.05".FB_OPEN )
   END_RUNG wire#w2
   RUNG wire#powerrail
      Contact( "IO_Valve_Blending_DB"."AV-31.52".FB_OPEN )
      Contact( "IO_Valve_Blending_DB"."AV-31.61".FB_OPEN )
   END_RUNG wire#w2
   // the same network as SCL:
   "T-06.01_DB"("IN_FBAV.01" := "IO_Valve_T06_FreshChili"."AV-06.01".FB_OPEN,   // "BFT_Type3"
                "IN_FBAV.02" := "IO_Valve_T06_FreshChili"."AV-06.02".FB_OPEN,
                "IN_FBAV.03" := "IO_Valve_T06_FreshChili"."AV-06.03".FB_OPEN,
                "IN_FBAV.04" := "IO_Valve_T06_FreshChili"."AV-06.04".FB_OPEN,
                "IN_FBAV.05" := "IO_Valve_T06_FreshChili"."AV-06.05".FB_OPEN,
                "IN_FBAV.06" := "IO_Valve_T06_FreshChili"."AV-06.06".FB_OPEN,
                "IN_FBAV.11" := "IO_Valve_T05_Tomato"."AV-05.11".FB_OPEN,
                "IN_FBAV.12" := "IO_Valve_T06_FreshChili"."AV-06.12".FB_OPEN,
                IN_LT01 := "IO Analog Preparation_DB"."LT-06.01".QOUT,
                "IN_FBP.01" := "IO Motor MCC Preparation_DB"."P-06.01".QFB_RUN,
                "IN_P.01-Speed" := "IO Motor MCC Preparation_DB"."P-06.01".QAct_Speed,
                LineTrf_OK := ("T-20.00_DB".ChiliFresh_1.QDOSERun AND "T-20.00_DB".ChiliFresh_1.V_OPEN) OR ("T-21.00_DB".ChiliFresh_1.QDOSERun AND "T-21.00_DB".ChiliFresh_1.V_OPEN) OR ("T-30.00_DB".ChiliFresh_1.QDOSERun AND "T-30.00_DB".ChiliFresh_1.V_OPEN) OR ("T-31.00_DB".ChiliFresh_1.QDOSERun AND "T-31.00_DB".ChiliFresh_1.V_OPEN),
                LineFlush_OK := "IO_Valve_Blending_DB"."AV-20.05".FB_OPEN OR "IO_Valve_Blending_DB"."AV-21.05".FB_OPEN OR "IO_Valve_Blending_DB"."AV-30.05".FB_OPEN OR "IO_Valve_Blending_DB"."AV-31.05".FB_OPEN OR ("IO_Valve_Blending_DB"."AV-31.52".FB_OPEN AND "IO_Valve_Blending_DB"."AV-31.61".FB_OPEN),
                "OUT_AV.01" => "IO_Valve_T06_FreshChili"."AV-06.01".AUT_OP,
                "OUT_AV.02" => "IO_Valve_T06_FreshChili"."AV-06.02".AUT_OP,
                "OUT_AV.03" => "IO_Valve_T06_FreshChili"."AV-06.03".AUT_OP,
                "OUT_AV.04" => "IO_Valve_T06_FreshChili"."AV-06.04".AUT_OP,
                "OUT_AV.05" => "IO_Valve_T06_FreshChili"."AV-06.05".AUT_OP,
                "OUT_AV.06" => "IO_Valve_T06_FreshChili"."AV-06.06".AUT_OP,
                "OUT_AV.12" => "IO_Valve_T06_FreshChili"."AV-06.12".AUT_OP,
                "OUT_P.01" => "IO Motor MCC Preparation_DB"."P-06.01".AUT_ON);
END_REGION

REGION Network 26: Dose ON OFF T-07.01 Chili Fresh 2
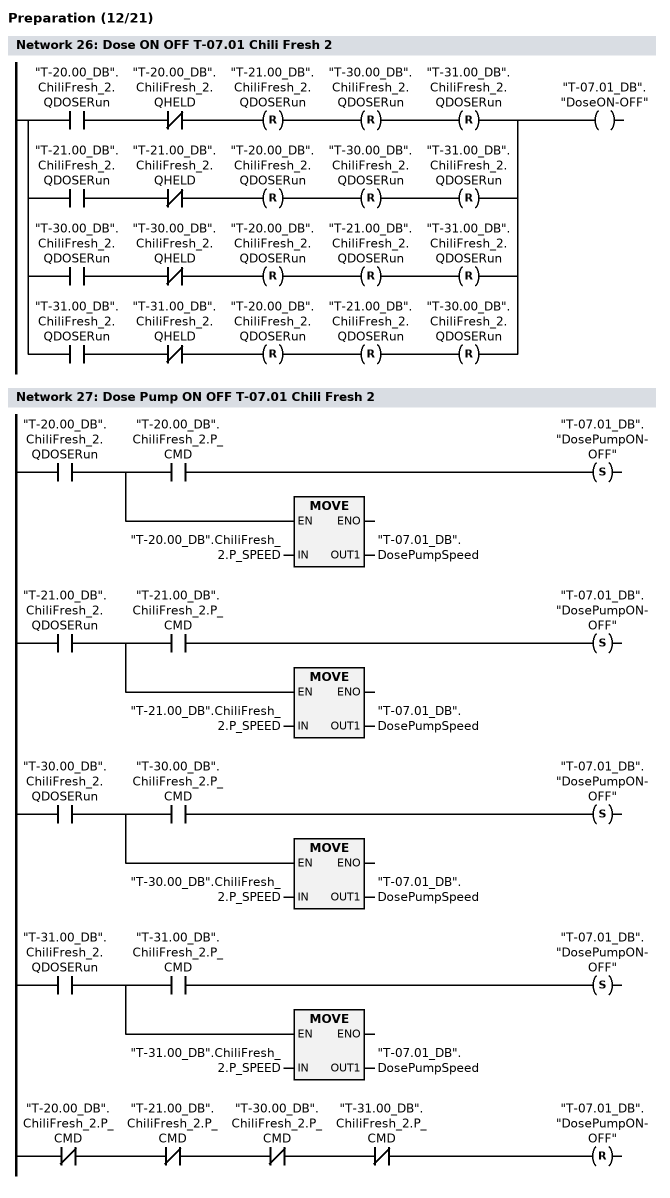
   RUNG wire#powerrail
      Contact( "T-20.00_DB".ChiliFresh_2.QDOSERun )
      I_Contact( "T-20.00_DB".ChiliFresh_2.QHELD )
      R_Coil( "T-21.00_DB".ChiliFresh_2.QDOSERun )
      R_Coil( "T-30.00_DB".ChiliFresh_2.QDOSERun )
      R_Coil( "T-31.00_DB".ChiliFresh_2.QDOSERun )
      wire#w1
      Coil( "T-07.01_DB"."DoseON-OFF" )
   END_RUNG
   RUNG wire#powerrail
      Contact( "T-21.00_DB".ChiliFresh_2.QDOSERun )
      I_Contact( "T-21.00_DB".ChiliFresh_2.QHELD )
      R_Coil( "T-20.00_DB".ChiliFresh_2.QDOSERun )
      R_Coil( "T-30.00_DB".ChiliFresh_2.QDOSERun )
      R_Coil( "T-31.00_DB".ChiliFresh_2.QDOSERun )
   END_RUNG wire#w1
   RUNG wire#powerrail
      Contact( "T-30.00_DB".ChiliFresh_2.QDOSERun )
      I_Contact( "T-30.00_DB".ChiliFresh_2.QHELD )
      R_Coil( "T-20.00_DB".ChiliFresh_2.QDOSERun )
      R_Coil( "T-21.00_DB".ChiliFresh_2.QDOSERun )
      R_Coil( "T-31.00_DB".ChiliFresh_2.QDOSERun )
   END_RUNG wire#w1
   RUNG wire#powerrail
      Contact( "T-31.00_DB".ChiliFresh_2.QDOSERun )
      I_Contact( "T-31.00_DB".ChiliFresh_2.QHELD )
      R_Coil( "T-20.00_DB".ChiliFresh_2.QDOSERun )
      R_Coil( "T-21.00_DB".ChiliFresh_2.QDOSERun )
      R_Coil( "T-30.00_DB".ChiliFresh_2.QDOSERun )
   END_RUNG wire#w1
   // the same network as SCL:
   #_w1 := "T-20.00_DB".ChiliFresh_2.QDOSERun AND NOT "T-20.00_DB".ChiliFresh_2.QHELD;
   IF #_w1 THEN
       "T-21.00_DB".ChiliFresh_2.QDOSERun := FALSE;
       "T-30.00_DB".ChiliFresh_2.QDOSERun := FALSE;
       "T-31.00_DB".ChiliFresh_2.QDOSERun := FALSE;
   END_IF;
   #_w2 := "T-21.00_DB".ChiliFresh_2.QDOSERun AND NOT "T-21.00_DB".ChiliFresh_2.QHELD;
   IF #_w2 THEN
       "T-20.00_DB".ChiliFresh_2.QDOSERun := FALSE;
       "T-30.00_DB".ChiliFresh_2.QDOSERun := FALSE;
       "T-31.00_DB".ChiliFresh_2.QDOSERun := FALSE;
   END_IF;
   #_w3 := "T-30.00_DB".ChiliFresh_2.QDOSERun AND NOT "T-30.00_DB".ChiliFresh_2.QHELD;
   IF #_w3 THEN
       "T-20.00_DB".ChiliFresh_2.QDOSERun := FALSE;
       "T-21.00_DB".ChiliFresh_2.QDOSERun := FALSE;
       "T-31.00_DB".ChiliFresh_2.QDOSERun := FALSE;
   END_IF;
   #_w4 := "T-31.00_DB".ChiliFresh_2.QDOSERun AND NOT "T-31.00_DB".ChiliFresh_2.QHELD;
   IF #_w4 THEN
       "T-20.00_DB".ChiliFresh_2.QDOSERun := FALSE;
       "T-21.00_DB".ChiliFresh_2.QDOSERun := FALSE;
       "T-30.00_DB".ChiliFresh_2.QDOSERun := FALSE;
   END_IF;
   "T-07.01_DB"."DoseON-OFF" := #_w1 OR #_w2 OR #_w3 OR #_w4;
END_REGION

REGION Network 27: Dose Pump ON OFF T-07.01 Chili Fresh 2
   RUNG wire#powerrail
      Contact( "T-20.00_DB".ChiliFresh_2.QDOSERun )
      wire#w1
      Contact( "T-20.00_DB".ChiliFresh_2.P_CMD )
      S_Coil( "T-07.01_DB"."DosePumpON-OFF" )
   END_RUNG
   RUNG wire#w1
      Move(in := "T-20.00_DB".ChiliFresh_2.P_SPEED, out1 => "T-07.01_DB".DosePumpSpeed)
   END_RUNG
   RUNG wire#powerrail
      Contact( "T-21.00_DB".ChiliFresh_2.QDOSERun )
      wire#w2
      Contact( "T-21.00_DB".ChiliFresh_2.P_CMD )
      S_Coil( "T-07.01_DB"."DosePumpON-OFF" )
   END_RUNG
   RUNG wire#w2
      Move(in := "T-21.00_DB".ChiliFresh_2.P_SPEED, out1 => "T-07.01_DB".DosePumpSpeed)
   END_RUNG
   RUNG wire#powerrail
      Contact( "T-30.00_DB".ChiliFresh_2.QDOSERun )
      wire#w3
      Contact( "T-30.00_DB".ChiliFresh_2.P_CMD )
      S_Coil( "T-07.01_DB"."DosePumpON-OFF" )
   END_RUNG
   RUNG wire#w3
      Move(in := "T-30.00_DB".ChiliFresh_2.P_SPEED, out1 => "T-07.01_DB".DosePumpSpeed)
   END_RUNG
   RUNG wire#powerrail
      Contact( "T-31.00_DB".ChiliFresh_2.QDOSERun )
      wire#w4
      Contact( "T-31.00_DB".ChiliFresh_2.P_CMD )
      S_Coil( "T-07.01_DB"."DosePumpON-OFF" )
   END_RUNG
   RUNG wire#w4
      Move(in := "T-31.00_DB".ChiliFresh_2.P_SPEED, out1 => "T-07.01_DB".DosePumpSpeed)
   END_RUNG
   RUNG wire#powerrail
      I_Contact( "T-20.00_DB".ChiliFresh_2.P_CMD )
      I_Contact( "T-21.00_DB".ChiliFresh_2.P_CMD )
      I_Contact( "T-30.00_DB".ChiliFresh_2.P_CMD )
      I_Contact( "T-31.00_DB".ChiliFresh_2.P_CMD )
      R_Coil( "T-07.01_DB"."DosePumpON-OFF" )
   END_RUNG
   // the same network as SCL:
   IF "T-20.00_DB".ChiliFresh_2.QDOSERun AND "T-20.00_DB".ChiliFresh_2.P_CMD THEN
       "T-07.01_DB"."DosePumpON-OFF" := TRUE;
   END_IF;
   IF "T-20.00_DB".ChiliFresh_2.QDOSERun THEN
       "T-07.01_DB".DosePumpSpeed := "T-20.00_DB".ChiliFresh_2.P_SPEED;
   END_IF;
   IF "T-21.00_DB".ChiliFresh_2.QDOSERun AND "T-21.00_DB".ChiliFresh_2.P_CMD THEN
       "T-07.01_DB"."DosePumpON-OFF" := TRUE;
   END_IF;
   IF "T-21.00_DB".ChiliFresh_2.QDOSERun THEN
       "T-07.01_DB".DosePumpSpeed := "T-21.00_DB".ChiliFresh_2.P_SPEED;
   END_IF;
   IF "T-30.00_DB".ChiliFresh_2.QDOSERun AND "T-30.00_DB".ChiliFresh_2.P_CMD THEN
       "T-07.01_DB"."DosePumpON-OFF" := TRUE;
   END_IF;
   IF "T-30.00_DB".ChiliFresh_2.QDOSERun THEN
       "T-07.01_DB".DosePumpSpeed := "T-30.00_DB".ChiliFresh_2.P_SPEED;
   END_IF;
   IF "T-31.00_DB".ChiliFresh_2.QDOSERun AND "T-31.00_DB".ChiliFresh_2.P_CMD THEN
       "T-07.01_DB"."DosePumpON-OFF" := TRUE;
   END_IF;
   IF "T-31.00_DB".ChiliFresh_2.QDOSERun THEN
       "T-07.01_DB".DosePumpSpeed := "T-31.00_DB".ChiliFresh_2.P_SPEED;
   END_IF;
   IF NOT "T-20.00_DB".ChiliFresh_2.P_CMD AND NOT "T-21.00_DB".ChiliFresh_2.P_CMD AND NOT "T-30.00_DB".ChiliFresh_2.P_CMD AND NOT "T-31.00_DB".ChiliFresh_2.P_CMD THEN
       "T-07.01_DB"."DosePumpON-OFF" := FALSE;
   END_IF;
END_REGION

REGION Network 28: T-07.01 Buffer Tank Chili Fresh
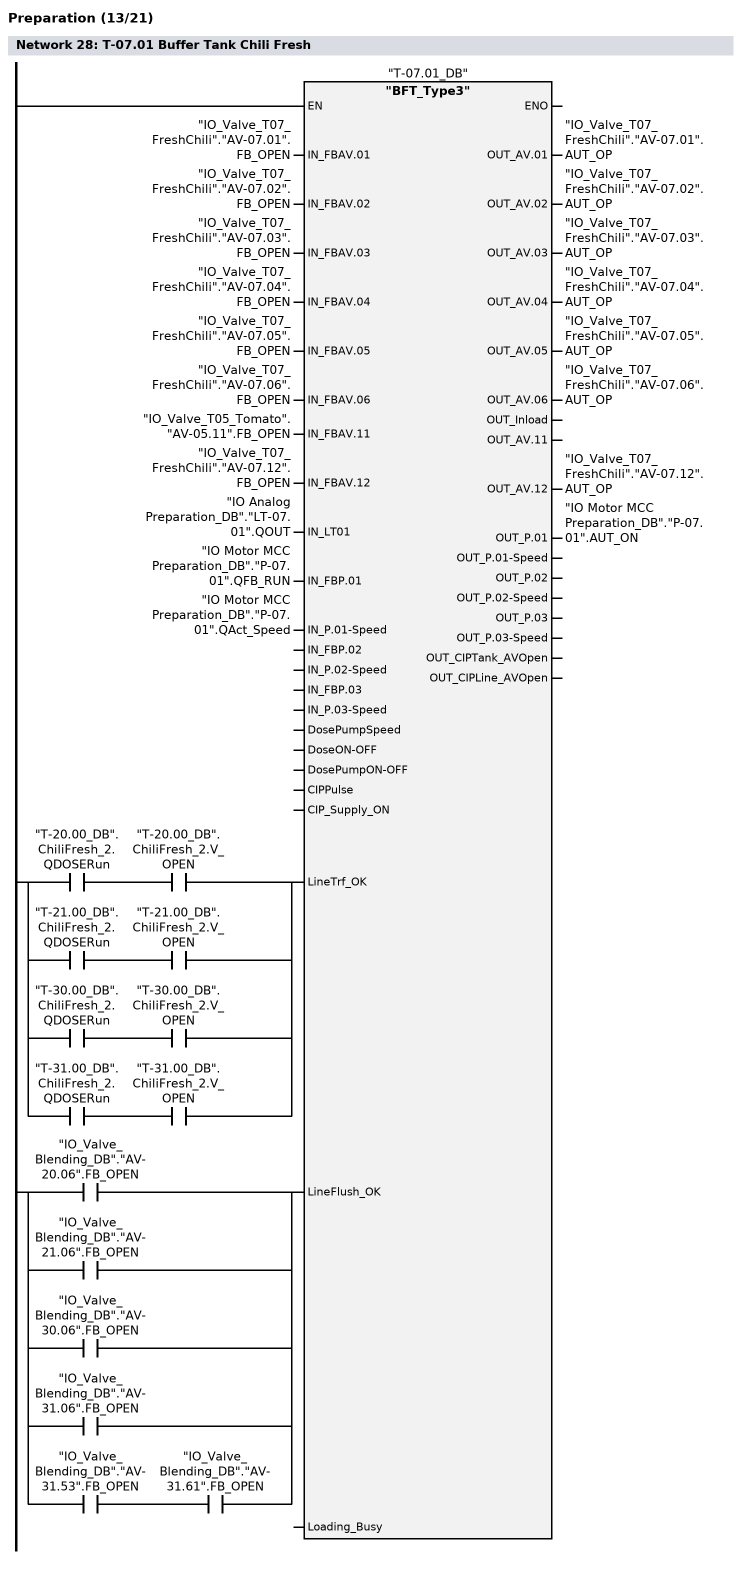
   RUNG wire#powerrail
      "T-07.01_DB"(LineTrf_OK := wire#w1, LineFlush_OK := wire#w2, "IN_FBAV.01" := "IO_Valve_T07_FreshChili"."AV-07.01".FB_OPEN, "IN_FBAV.02" := "IO_Valve_T07_FreshChili"."AV-07.02".FB_OPEN, "IN_FBAV.03" := "IO_Valve_T07_FreshChili"."AV-07.03".FB_OPEN, "IN_FBAV.04" := "IO_Valve_T07_FreshChili"."AV-07.04".FB_OPEN, "IN_FBAV.05" := "IO_Valve_T07_FreshChili"."AV-07.05".FB_OPEN, "IN_FBAV.06" := "IO_Valve_T07_FreshChili"."AV-07.06".FB_OPEN, "IN_FBAV.11" := "IO_Valve_T05_Tomato"."AV-05.11".FB_OPEN, "IN_FBAV.12" := "IO_Valve_T07_FreshChili"."AV-07.12".FB_OPEN, IN_LT01 := "IO Analog Preparation_DB"."LT-07.01".QOUT, "IN_FBP.01" := "IO Motor MCC Preparation_DB"."P-07.01".QFB_RUN, "IN_P.01-Speed" := "IO Motor MCC Preparation_DB"."P-07.01".QAct_Speed, "IN_FBP.02" :=, "IN_P.02-Speed" :=, "IN_FBP.03" :=, "IN_P.03-Speed" :=, DosePumpSpeed :=, "DoseON-OFF" :=, "DosePumpON-OFF" :=, CIPPulse :=, CIP_Supply_ON :=, Loading_Busy :=, "OUT_AV.01" => "IO_Valve_T07_FreshChili"."AV-07.01".AUT_OP, "OUT_AV.02" => "IO_Valve_T07_FreshChili"."AV-07.02".AUT_OP, "OUT_AV.03" => "IO_Valve_T07_FreshChili"."AV-07.03".AUT_OP, "OUT_AV.04" => "IO_Valve_T07_FreshChili"."AV-07.04".AUT_OP, "OUT_AV.05" => "IO_Valve_T07_FreshChili"."AV-07.05".AUT_OP, "OUT_AV.06" => "IO_Valve_T07_FreshChili"."AV-07.06".AUT_OP, OUT_Inload =>, "OUT_AV.11" =>, "OUT_AV.12" => "IO_Valve_T07_FreshChili"."AV-07.12".AUT_OP, "OUT_P.01" => "IO Motor MCC Preparation_DB"."P-07.01".AUT_ON, "OUT_P.01-Speed" =>, "OUT_P.02" =>, "OUT_P.02-Speed" =>, "OUT_P.03" =>, "OUT_P.03-Speed" =>, OUT_CIPTank_AVOpen =>, OUT_CIPLine_AVOpen =>)
   END_RUNG
   RUNG wire#powerrail
      Contact( "T-20.00_DB".ChiliFresh_2.QDOSERun )
      Contact( "T-20.00_DB".ChiliFresh_2.V_OPEN )
   END_RUNG wire#w1
   RUNG wire#powerrail
      Contact( "T-21.00_DB".ChiliFresh_2.QDOSERun )
      Contact( "T-21.00_DB".ChiliFresh_2.V_OPEN )
   END_RUNG wire#w1
   RUNG wire#powerrail
      Contact( "T-30.00_DB".ChiliFresh_2.QDOSERun )
      Contact( "T-30.00_DB".ChiliFresh_2.V_OPEN )
   END_RUNG wire#w1
   RUNG wire#powerrail
      Contact( "T-31.00_DB".ChiliFresh_2.QDOSERun )
      Contact( "T-31.00_DB".ChiliFresh_2.V_OPEN )
   END_RUNG wire#w1
   RUNG wire#powerrail
      Contact( "IO_Valve_Blending_DB"."AV-20.06".FB_OPEN )
   END_RUNG wire#w2
   RUNG wire#powerrail
      Contact( "IO_Valve_Blending_DB"."AV-21.06".FB_OPEN )
   END_RUNG wire#w2
   RUNG wire#powerrail
      Contact( "IO_Valve_Blending_DB"."AV-30.06".FB_OPEN )
   END_RUNG wire#w2
   RUNG wire#powerrail
      Contact( "IO_Valve_Blending_DB"."AV-31.06".FB_OPEN )
   END_RUNG wire#w2
   RUNG wire#powerrail
      Contact( "IO_Valve_Blending_DB"."AV-31.53".FB_OPEN )
      Contact( "IO_Valve_Blending_DB"."AV-31.61".FB_OPEN )
   END_RUNG wire#w2
   // the same network as SCL:
   "T-07.01_DB"("IN_FBAV.01" := "IO_Valve_T07_FreshChili"."AV-07.01".FB_OPEN,   // "BFT_Type3"
                "IN_FBAV.02" := "IO_Valve_T07_FreshChili"."AV-07.02".FB_OPEN,
                "IN_FBAV.03" := "IO_Valve_T07_FreshChili"."AV-07.03".FB_OPEN,
                "IN_FBAV.04" := "IO_Valve_T07_FreshChili"."AV-07.04".FB_OPEN,
                "IN_FBAV.05" := "IO_Valve_T07_FreshChili"."AV-07.05".FB_OPEN,
                "IN_FBAV.06" := "IO_Valve_T07_FreshChili"."AV-07.06".FB_OPEN,
                "IN_FBAV.11" := "IO_Valve_T05_Tomato"."AV-05.11".FB_OPEN,
                "IN_FBAV.12" := "IO_Valve_T07_FreshChili"."AV-07.12".FB_OPEN,
                IN_LT01 := "IO Analog Preparation_DB"."LT-07.01".QOUT,
                "IN_FBP.01" := "IO Motor MCC Preparation_DB"."P-07.01".QFB_RUN,
                "IN_P.01-Speed" := "IO Motor MCC Preparation_DB"."P-07.01".QAct_Speed,
                LineTrf_OK := ("T-20.00_DB".ChiliFresh_2.QDOSERun AND "T-20.00_DB".ChiliFresh_2.V_OPEN) OR ("T-21.00_DB".ChiliFresh_2.QDOSERun AND "T-21.00_DB".ChiliFresh_2.V_OPEN) OR ("T-30.00_DB".ChiliFresh_2.QDOSERun AND "T-30.00_DB".ChiliFresh_2.V_OPEN) OR ("T-31.00_DB".ChiliFresh_2.QDOSERun AND "T-31.00_DB".ChiliFresh_2.V_OPEN),
                LineFlush_OK := "IO_Valve_Blending_DB"."AV-20.06".FB_OPEN OR "IO_Valve_Blending_DB"."AV-21.06".FB_OPEN OR "IO_Valve_Blending_DB"."AV-30.06".FB_OPEN OR "IO_Valve_Blending_DB"."AV-31.06".FB_OPEN OR ("IO_Valve_Blending_DB"."AV-31.53".FB_OPEN AND "IO_Valve_Blending_DB"."AV-31.61".FB_OPEN),
                "OUT_AV.01" => "IO_Valve_T07_FreshChili"."AV-07.01".AUT_OP,
                "OUT_AV.02" => "IO_Valve_T07_FreshChili"."AV-07.02".AUT_OP,
                "OUT_AV.03" => "IO_Valve_T07_FreshChili"."AV-07.03".AUT_OP,
                "OUT_AV.04" => "IO_Valve_T07_FreshChili"."AV-07.04".AUT_OP,
                "OUT_AV.05" => "IO_Valve_T07_FreshChili"."AV-07.05".AUT_OP,
                "OUT_AV.06" => "IO_Valve_T07_FreshChili"."AV-07.06".AUT_OP,
                "OUT_AV.12" => "IO_Valve_T07_FreshChili"."AV-07.12".AUT_OP,
                "OUT_P.01" => "IO Motor MCC Preparation_DB"."P-07.01".AUT_ON);
END_REGION

REGION Network 30: Dose ON OFF T-08.01 Chili Fresh 3
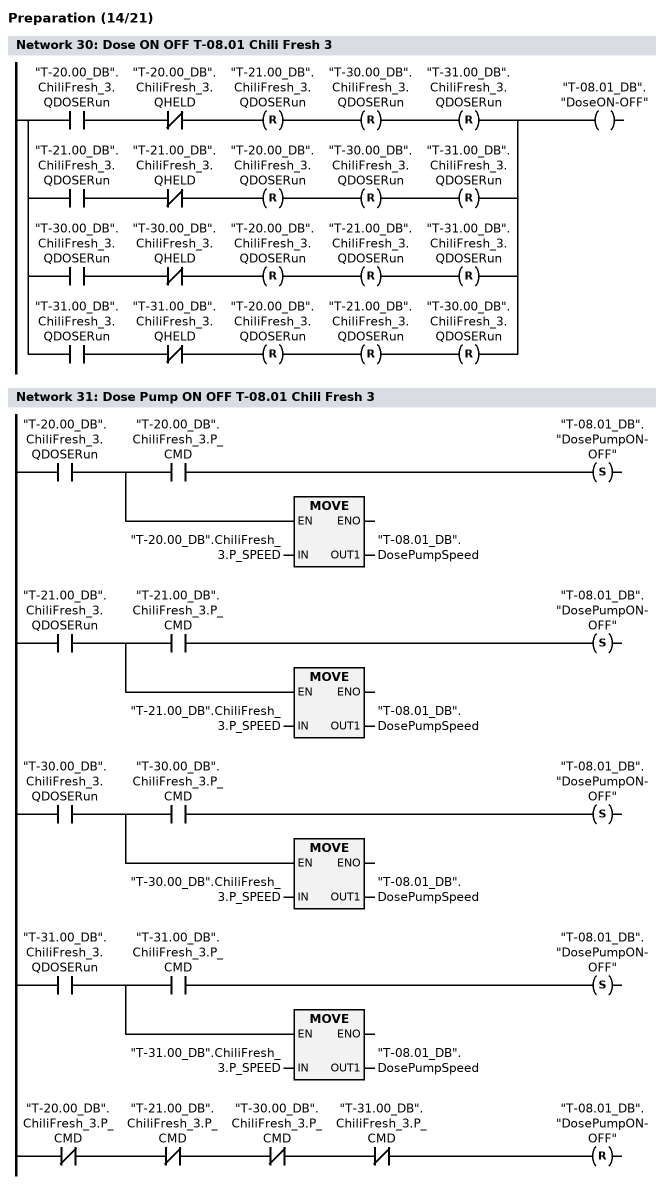
   RUNG wire#powerrail
      Contact( "T-20.00_DB".ChiliFresh_3.QDOSERun )
      I_Contact( "T-20.00_DB".ChiliFresh_3.QHELD )
      R_Coil( "T-21.00_DB".ChiliFresh_3.QDOSERun )
      R_Coil( "T-30.00_DB".ChiliFresh_3.QDOSERun )
      R_Coil( "T-31.00_DB".ChiliFresh_3.QDOSERun )
      wire#w1
      Coil( "T-08.01_DB"."DoseON-OFF" )
   END_RUNG
   RUNG wire#powerrail
      Contact( "T-21.00_DB".ChiliFresh_3.QDOSERun )
      I_Contact( "T-21.00_DB".ChiliFresh_3.QHELD )
      R_Coil( "T-20.00_DB".ChiliFresh_3.QDOSERun )
      R_Coil( "T-30.00_DB".ChiliFresh_3.QDOSERun )
      R_Coil( "T-31.00_DB".ChiliFresh_3.QDOSERun )
   END_RUNG wire#w1
   RUNG wire#powerrail
      Contact( "T-30.00_DB".ChiliFresh_3.QDOSERun )
      I_Contact( "T-30.00_DB".ChiliFresh_3.QHELD )
      R_Coil( "T-20.00_DB".ChiliFresh_3.QDOSERun )
      R_Coil( "T-21.00_DB".ChiliFresh_3.QDOSERun )
      R_Coil( "T-31.00_DB".ChiliFresh_3.QDOSERun )
   END_RUNG wire#w1
   RUNG wire#powerrail
      Contact( "T-31.00_DB".ChiliFresh_3.QDOSERun )
      I_Contact( "T-31.00_DB".ChiliFresh_3.QHELD )
      R_Coil( "T-20.00_DB".ChiliFresh_3.QDOSERun )
      R_Coil( "T-21.00_DB".ChiliFresh_3.QDOSERun )
      R_Coil( "T-30.00_DB".ChiliFresh_3.QDOSERun )
   END_RUNG wire#w1
   // the same network as SCL:
   #_w1 := "T-20.00_DB".ChiliFresh_3.QDOSERun AND NOT "T-20.00_DB".ChiliFresh_3.QHELD;
   IF #_w1 THEN
       "T-21.00_DB".ChiliFresh_3.QDOSERun := FALSE;
       "T-30.00_DB".ChiliFresh_3.QDOSERun := FALSE;
       "T-31.00_DB".ChiliFresh_3.QDOSERun := FALSE;
   END_IF;
   #_w2 := "T-21.00_DB".ChiliFresh_3.QDOSERun AND NOT "T-21.00_DB".ChiliFresh_3.QHELD;
   IF #_w2 THEN
       "T-20.00_DB".ChiliFresh_3.QDOSERun := FALSE;
       "T-30.00_DB".ChiliFresh_3.QDOSERun := FALSE;
       "T-31.00_DB".ChiliFresh_3.QDOSERun := FALSE;
   END_IF;
   #_w3 := "T-30.00_DB".ChiliFresh_3.QDOSERun AND NOT "T-30.00_DB".ChiliFresh_3.QHELD;
   IF #_w3 THEN
       "T-20.00_DB".ChiliFresh_3.QDOSERun := FALSE;
       "T-21.00_DB".ChiliFresh_3.QDOSERun := FALSE;
       "T-31.00_DB".ChiliFresh_3.QDOSERun := FALSE;
   END_IF;
   #_w4 := "T-31.00_DB".ChiliFresh_3.QDOSERun AND NOT "T-31.00_DB".ChiliFresh_3.QHELD;
   IF #_w4 THEN
       "T-20.00_DB".ChiliFresh_3.QDOSERun := FALSE;
       "T-21.00_DB".ChiliFresh_3.QDOSERun := FALSE;
       "T-30.00_DB".ChiliFresh_3.QDOSERun := FALSE;
   END_IF;
   "T-08.01_DB"."DoseON-OFF" := #_w1 OR #_w2 OR #_w3 OR #_w4;
END_REGION

REGION Network 31: Dose Pump ON OFF T-08.01 Chili Fresh 3
   RUNG wire#powerrail
      Contact( "T-20.00_DB".ChiliFresh_3.QDOSERun )
      wire#w1
      Contact( "T-20.00_DB".ChiliFresh_3.P_CMD )
      S_Coil( "T-08.01_DB"."DosePumpON-OFF" )
   END_RUNG
   RUNG wire#w1
      Move(in := "T-20.00_DB".ChiliFresh_3.P_SPEED, out1 => "T-08.01_DB".DosePumpSpeed)
   END_RUNG
   RUNG wire#powerrail
      Contact( "T-21.00_DB".ChiliFresh_3.QDOSERun )
      wire#w2
      Contact( "T-21.00_DB".ChiliFresh_3.P_CMD )
      S_Coil( "T-08.01_DB"."DosePumpON-OFF" )
   END_RUNG
   RUNG wire#w2
      Move(in := "T-21.00_DB".ChiliFresh_3.P_SPEED, out1 => "T-08.01_DB".DosePumpSpeed)
   END_RUNG
   RUNG wire#powerrail
      Contact( "T-30.00_DB".ChiliFresh_3.QDOSERun )
      wire#w3
      Contact( "T-30.00_DB".ChiliFresh_3.P_CMD )
      S_Coil( "T-08.01_DB"."DosePumpON-OFF" )
   END_RUNG
   RUNG wire#w3
      Move(in := "T-30.00_DB".ChiliFresh_3.P_SPEED, out1 => "T-08.01_DB".DosePumpSpeed)
   END_RUNG
   RUNG wire#powerrail
      Contact( "T-31.00_DB".ChiliFresh_3.QDOSERun )
      wire#w4
      Contact( "T-31.00_DB".ChiliFresh_3.P_CMD )
      S_Coil( "T-08.01_DB"."DosePumpON-OFF" )
   END_RUNG
   RUNG wire#w4
      Move(in := "T-31.00_DB".ChiliFresh_3.P_SPEED, out1 => "T-08.01_DB".DosePumpSpeed)
   END_RUNG
   RUNG wire#powerrail
      I_Contact( "T-20.00_DB".ChiliFresh_3.P_CMD )
      I_Contact( "T-21.00_DB".ChiliFresh_3.P_CMD )
      I_Contact( "T-30.00_DB".ChiliFresh_3.P_CMD )
      I_Contact( "T-31.00_DB".ChiliFresh_3.P_CMD )
      R_Coil( "T-08.01_DB"."DosePumpON-OFF" )
   END_RUNG
   // the same network as SCL:
   IF "T-20.00_DB".ChiliFresh_3.QDOSERun AND "T-20.00_DB".ChiliFresh_3.P_CMD THEN
       "T-08.01_DB"."DosePumpON-OFF" := TRUE;
   END_IF;
   IF "T-20.00_DB".ChiliFresh_3.QDOSERun THEN
       "T-08.01_DB".DosePumpSpeed := "T-20.00_DB".ChiliFresh_3.P_SPEED;
   END_IF;
   IF "T-21.00_DB".ChiliFresh_3.QDOSERun AND "T-21.00_DB".ChiliFresh_3.P_CMD THEN
       "T-08.01_DB"."DosePumpON-OFF" := TRUE;
   END_IF;
   IF "T-21.00_DB".ChiliFresh_3.QDOSERun THEN
       "T-08.01_DB".DosePumpSpeed := "T-21.00_DB".ChiliFresh_3.P_SPEED;
   END_IF;
   IF "T-30.00_DB".ChiliFresh_3.QDOSERun AND "T-30.00_DB".ChiliFresh_3.P_CMD THEN
       "T-08.01_DB"."DosePumpON-OFF" := TRUE;
   END_IF;
   IF "T-30.00_DB".ChiliFresh_3.QDOSERun THEN
       "T-08.01_DB".DosePumpSpeed := "T-30.00_DB".ChiliFresh_3.P_SPEED;
   END_IF;
   IF "T-31.00_DB".ChiliFresh_3.QDOSERun AND "T-31.00_DB".ChiliFresh_3.P_CMD THEN
       "T-08.01_DB"."DosePumpON-OFF" := TRUE;
   END_IF;
   IF "T-31.00_DB".ChiliFresh_3.QDOSERun THEN
       "T-08.01_DB".DosePumpSpeed := "T-31.00_DB".ChiliFresh_3.P_SPEED;
   END_IF;
   IF NOT "T-20.00_DB".ChiliFresh_3.P_CMD AND NOT "T-21.00_DB".ChiliFresh_3.P_CMD AND NOT "T-30.00_DB".ChiliFresh_3.P_CMD AND NOT "T-31.00_DB".ChiliFresh_3.P_CMD THEN
       "T-08.01_DB"."DosePumpON-OFF" := FALSE;
   END_IF;
END_REGION

REGION Network 32: T-08.01 Buffer Tank Chili Fresh
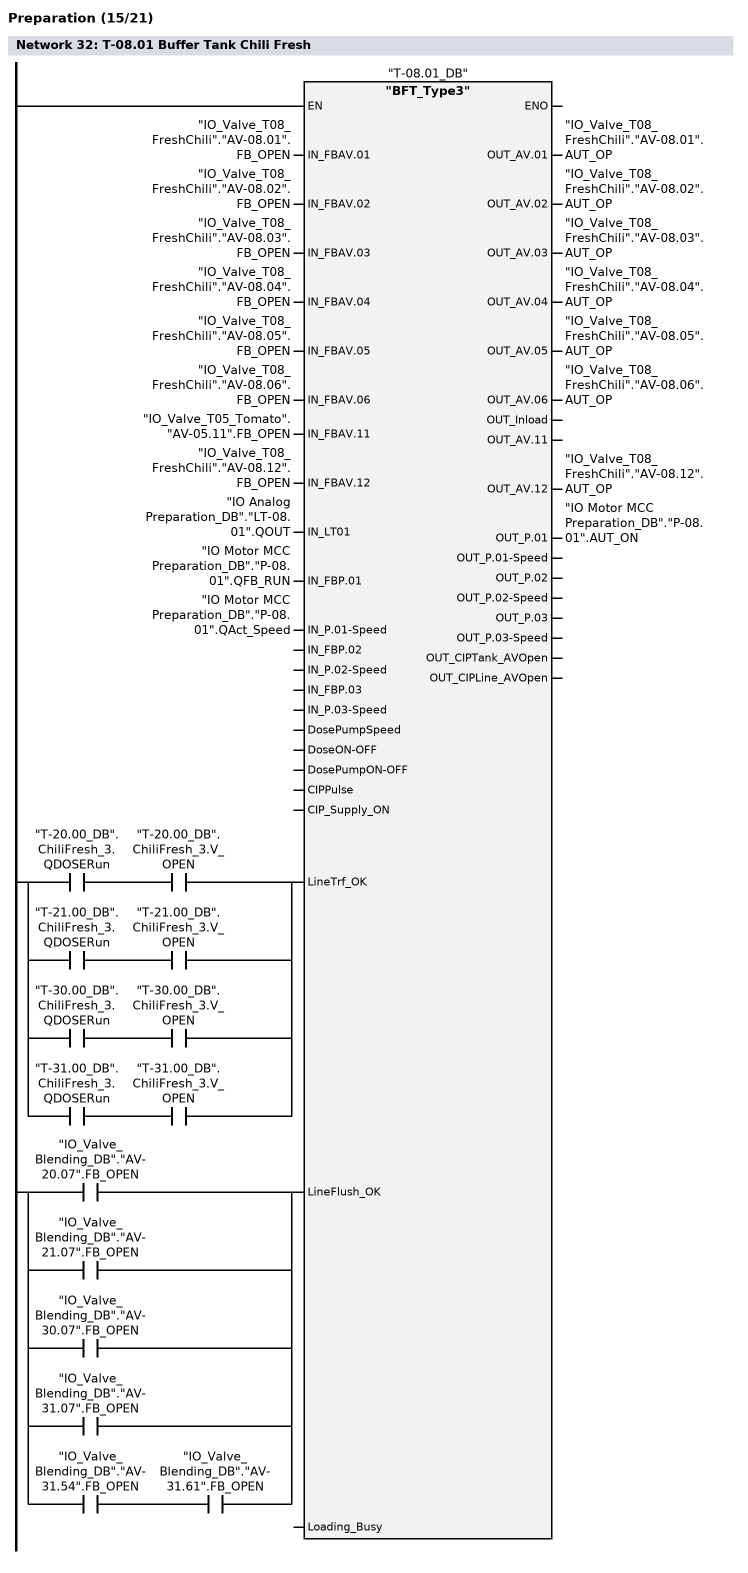
   RUNG wire#powerrail
      "T-08.01_DB"(LineTrf_OK := wire#w1, LineFlush_OK := wire#w2, "IN_FBAV.01" := "IO_Valve_T08_FreshChili"."AV-08.01".FB_OPEN, "IN_FBAV.02" := "IO_Valve_T08_FreshChili"."AV-08.02".FB_OPEN, "IN_FBAV.03" := "IO_Valve_T08_FreshChili"."AV-08.03".FB_OPEN, "IN_FBAV.04" := "IO_Valve_T08_FreshChili"."AV-08.04".FB_OPEN, "IN_FBAV.05" := "IO_Valve_T08_FreshChili"."AV-08.05".FB_OPEN, "IN_FBAV.06" := "IO_Valve_T08_FreshChili"."AV-08.06".FB_OPEN, "IN_FBAV.11" := "IO_Valve_T05_Tomato"."AV-05.11".FB_OPEN, "IN_FBAV.12" := "IO_Valve_T08_FreshChili"."AV-08.12".FB_OPEN, IN_LT01 := "IO Analog Preparation_DB"."LT-08.01".QOUT, "IN_FBP.01" := "IO Motor MCC Preparation_DB"."P-08.01".QFB_RUN, "IN_P.01-Speed" := "IO Motor MCC Preparation_DB"."P-08.01".QAct_Speed, "IN_FBP.02" :=, "IN_P.02-Speed" :=, "IN_FBP.03" :=, "IN_P.03-Speed" :=, DosePumpSpeed :=, "DoseON-OFF" :=, "DosePumpON-OFF" :=, CIPPulse :=, CIP_Supply_ON :=, Loading_Busy :=, "OUT_AV.01" => "IO_Valve_T08_FreshChili"."AV-08.01".AUT_OP, "OUT_AV.02" => "IO_Valve_T08_FreshChili"."AV-08.02".AUT_OP, "OUT_AV.03" => "IO_Valve_T08_FreshChili"."AV-08.03".AUT_OP, "OUT_AV.04" => "IO_Valve_T08_FreshChili"."AV-08.04".AUT_OP, "OUT_AV.05" => "IO_Valve_T08_FreshChili"."AV-08.05".AUT_OP, "OUT_AV.06" => "IO_Valve_T08_FreshChili"."AV-08.06".AUT_OP, OUT_Inload =>, "OUT_AV.11" =>, "OUT_AV.12" => "IO_Valve_T08_FreshChili"."AV-08.12".AUT_OP, "OUT_P.01" => "IO Motor MCC Preparation_DB"."P-08.01".AUT_ON, "OUT_P.01-Speed" =>, "OUT_P.02" =>, "OUT_P.02-Speed" =>, "OUT_P.03" =>, "OUT_P.03-Speed" =>, OUT_CIPTank_AVOpen =>, OUT_CIPLine_AVOpen =>)
   END_RUNG
   RUNG wire#powerrail
      Contact( "T-20.00_DB".ChiliFresh_3.QDOSERun )
      Contact( "T-20.00_DB".ChiliFresh_3.V_OPEN )
   END_RUNG wire#w1
   RUNG wire#powerrail
      Contact( "T-21.00_DB".ChiliFresh_3.QDOSERun )
      Contact( "T-21.00_DB".ChiliFresh_3.V_OPEN )
   END_RUNG wire#w1
   RUNG wire#powerrail
      Contact( "T-30.00_DB".ChiliFresh_3.QDOSERun )
      Contact( "T-30.00_DB".ChiliFresh_3.V_OPEN )
   END_RUNG wire#w1
   RUNG wire#powerrail
      Contact( "T-31.00_DB".ChiliFresh_3.QDOSERun )
      Contact( "T-31.00_DB".ChiliFresh_3.V_OPEN )
   END_RUNG wire#w1
   RUNG wire#powerrail
      Contact( "IO_Valve_Blending_DB"."AV-20.07".FB_OPEN )
   END_RUNG wire#w2
   RUNG wire#powerrail
      Contact( "IO_Valve_Blending_DB"."AV-21.07".FB_OPEN )
   END_RUNG wire#w2
   RUNG wire#powerrail
      Contact( "IO_Valve_Blending_DB"."AV-30.07".FB_OPEN )
   END_RUNG wire#w2
   RUNG wire#powerrail
      Contact( "IO_Valve_Blending_DB"."AV-31.07".FB_OPEN )
   END_RUNG wire#w2
   RUNG wire#powerrail
      Contact( "IO_Valve_Blending_DB"."AV-31.54".FB_OPEN )
      Contact( "IO_Valve_Blending_DB"."AV-31.61".FB_OPEN )
   END_RUNG wire#w2
   // the same network as SCL:
   "T-08.01_DB"("IN_FBAV.01" := "IO_Valve_T08_FreshChili"."AV-08.01".FB_OPEN,   // "BFT_Type3"
                "IN_FBAV.02" := "IO_Valve_T08_FreshChili"."AV-08.02".FB_OPEN,
                "IN_FBAV.03" := "IO_Valve_T08_FreshChili"."AV-08.03".FB_OPEN,
                "IN_FBAV.04" := "IO_Valve_T08_FreshChili"."AV-08.04".FB_OPEN,
                "IN_FBAV.05" := "IO_Valve_T08_FreshChili"."AV-08.05".FB_OPEN,
                "IN_FBAV.06" := "IO_Valve_T08_FreshChili"."AV-08.06".FB_OPEN,
                "IN_FBAV.11" := "IO_Valve_T05_Tomato"."AV-05.11".FB_OPEN,
                "IN_FBAV.12" := "IO_Valve_T08_FreshChili"."AV-08.12".FB_OPEN,
                IN_LT01 := "IO Analog Preparation_DB"."LT-08.01".QOUT,
                "IN_FBP.01" := "IO Motor MCC Preparation_DB"."P-08.01".QFB_RUN,
                "IN_P.01-Speed" := "IO Motor MCC Preparation_DB"."P-08.01".QAct_Speed,
                LineTrf_OK := ("T-20.00_DB".ChiliFresh_3.QDOSERun AND "T-20.00_DB".ChiliFresh_3.V_OPEN) OR ("T-21.00_DB".ChiliFresh_3.QDOSERun AND "T-21.00_DB".ChiliFresh_3.V_OPEN) OR ("T-30.00_DB".ChiliFresh_3.QDOSERun AND "T-30.00_DB".ChiliFresh_3.V_OPEN) OR ("T-31.00_DB".ChiliFresh_3.QDOSERun AND "T-31.00_DB".ChiliFresh_3.V_OPEN),
                LineFlush_OK := "IO_Valve_Blending_DB"."AV-20.07".FB_OPEN OR "IO_Valve_Blending_DB"."AV-21.07".FB_OPEN OR "IO_Valve_Blending_DB"."AV-30.07".FB_OPEN OR "IO_Valve_Blending_DB"."AV-31.07".FB_OPEN OR ("IO_Valve_Blending_DB"."AV-31.54".FB_OPEN AND "IO_Valve_Blending_DB"."AV-31.61".FB_OPEN),
                "OUT_AV.01" => "IO_Valve_T08_FreshChili"."AV-08.01".AUT_OP,
                "OUT_AV.02" => "IO_Valve_T08_FreshChili"."AV-08.02".AUT_OP,
                "OUT_AV.03" => "IO_Valve_T08_FreshChili"."AV-08.03".AUT_OP,
                "OUT_AV.04" => "IO_Valve_T08_FreshChili"."AV-08.04".AUT_OP,
                "OUT_AV.05" => "IO_Valve_T08_FreshChili"."AV-08.05".AUT_OP,
                "OUT_AV.06" => "IO_Valve_T08_FreshChili"."AV-08.06".AUT_OP,
                "OUT_AV.12" => "IO_Valve_T08_FreshChili"."AV-08.12".AUT_OP,
                "OUT_P.01" => "IO Motor MCC Preparation_DB"."P-08.01".AUT_ON);
END_REGION

REGION Network 34: Dose ON OFF T-09.01 Garlic
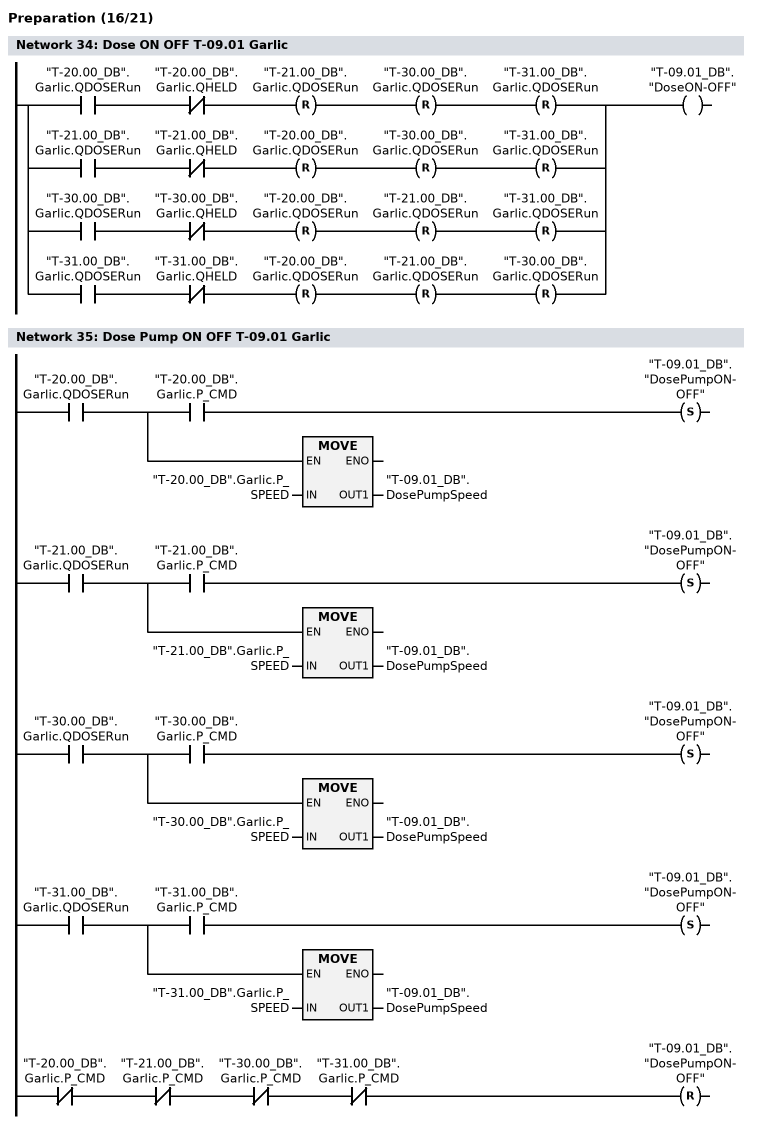
   RUNG wire#powerrail
      Contact( "T-20.00_DB".Garlic.QDOSERun )
      I_Contact( "T-20.00_DB".Garlic.QHELD )
      R_Coil( "T-21.00_DB".Garlic.QDOSERun )
      R_Coil( "T-30.00_DB".Garlic.QDOSERun )
      R_Coil( "T-31.00_DB".Garlic.QDOSERun )
      wire#w1
      Coil( "T-09.01_DB"."DoseON-OFF" )
   END_RUNG
   RUNG wire#powerrail
      Contact( "T-21.00_DB".Garlic.QDOSERun )
      I_Contact( "T-21.00_DB".Garlic.QHELD )
      R_Coil( "T-20.00_DB".Garlic.QDOSERun )
      R_Coil( "T-30.00_DB".Garlic.QDOSERun )
      R_Coil( "T-31.00_DB".Garlic.QDOSERun )
   END_RUNG wire#w1
   RUNG wire#powerrail
      Contact( "T-30.00_DB".Garlic.QDOSERun )
      I_Contact( "T-30.00_DB".Garlic.QHELD )
      R_Coil( "T-20.00_DB".Garlic.QDOSERun )
      R_Coil( "T-21.00_DB".Garlic.QDOSERun )
      R_Coil( "T-31.00_DB".Garlic.QDOSERun )
   END_RUNG wire#w1
   RUNG wire#powerrail
      Contact( "T-31.00_DB".Garlic.QDOSERun )
      I_Contact( "T-31.00_DB".Garlic.QHELD )
      R_Coil( "T-20.00_DB".Garlic.QDOSERun )
      R_Coil( "T-21.00_DB".Garlic.QDOSERun )
      R_Coil( "T-30.00_DB".Garlic.QDOSERun )
   END_RUNG wire#w1
   // the same network as SCL:
   #_w1 := "T-20.00_DB".Garlic.QDOSERun AND NOT "T-20.00_DB".Garlic.QHELD;
   IF #_w1 THEN
       "T-21.00_DB".Garlic.QDOSERun := FALSE;
       "T-30.00_DB".Garlic.QDOSERun := FALSE;
       "T-31.00_DB".Garlic.QDOSERun := FALSE;
   END_IF;
   #_w2 := "T-21.00_DB".Garlic.QDOSERun AND NOT "T-21.00_DB".Garlic.QHELD;
   IF #_w2 THEN
       "T-20.00_DB".Garlic.QDOSERun := FALSE;
       "T-30.00_DB".Garlic.QDOSERun := FALSE;
       "T-31.00_DB".Garlic.QDOSERun := FALSE;
   END_IF;
   #_w3 := "T-30.00_DB".Garlic.QDOSERun AND NOT "T-30.00_DB".Garlic.QHELD;
   IF #_w3 THEN
       "T-20.00_DB".Garlic.QDOSERun := FALSE;
       "T-21.00_DB".Garlic.QDOSERun := FALSE;
       "T-31.00_DB".Garlic.QDOSERun := FALSE;
   END_IF;
   #_w4 := "T-31.00_DB".Garlic.QDOSERun AND NOT "T-31.00_DB".Garlic.QHELD;
   IF #_w4 THEN
       "T-20.00_DB".Garlic.QDOSERun := FALSE;
       "T-21.00_DB".Garlic.QDOSERun := FALSE;
       "T-30.00_DB".Garlic.QDOSERun := FALSE;
   END_IF;
   "T-09.01_DB"."DoseON-OFF" := #_w1 OR #_w2 OR #_w3 OR #_w4;
END_REGION

REGION Network 35: Dose Pump ON OFF T-09.01 Garlic
   RUNG wire#powerrail
      Contact( "T-20.00_DB".Garlic.QDOSERun )
      wire#w1
      Contact( "T-20.00_DB".Garlic.P_CMD )
      S_Coil( "T-09.01_DB"."DosePumpON-OFF" )
   END_RUNG
   RUNG wire#w1
      Move(in := "T-20.00_DB".Garlic.P_SPEED, out1 => "T-09.01_DB".DosePumpSpeed)
   END_RUNG
   RUNG wire#powerrail
      Contact( "T-21.00_DB".Garlic.QDOSERun )
      wire#w2
      Contact( "T-21.00_DB".Garlic.P_CMD )
      S_Coil( "T-09.01_DB"."DosePumpON-OFF" )
   END_RUNG
   RUNG wire#w2
      Move(in := "T-21.00_DB".Garlic.P_SPEED, out1 => "T-09.01_DB".DosePumpSpeed)
   END_RUNG
   RUNG wire#powerrail
      Contact( "T-30.00_DB".Garlic.QDOSERun )
      wire#w3
      Contact( "T-30.00_DB".Garlic.P_CMD )
      S_Coil( "T-09.01_DB"."DosePumpON-OFF" )
   END_RUNG
   RUNG wire#w3
      Move(in := "T-30.00_DB".Garlic.P_SPEED, out1 => "T-09.01_DB".DosePumpSpeed)
   END_RUNG
   RUNG wire#powerrail
      Contact( "T-31.00_DB".Garlic.QDOSERun )
      wire#w4
      Contact( "T-31.00_DB".Garlic.P_CMD )
      S_Coil( "T-09.01_DB"."DosePumpON-OFF" )
   END_RUNG
   RUNG wire#w4
      Move(in := "T-31.00_DB".Garlic.P_SPEED, out1 => "T-09.01_DB".DosePumpSpeed)
   END_RUNG
   RUNG wire#powerrail
      I_Contact( "T-20.00_DB".Garlic.P_CMD )
      I_Contact( "T-21.00_DB".Garlic.P_CMD )
      I_Contact( "T-30.00_DB".Garlic.P_CMD )
      I_Contact( "T-31.00_DB".Garlic.P_CMD )
      R_Coil( "T-09.01_DB"."DosePumpON-OFF" )
   END_RUNG
   // the same network as SCL:
   IF "T-20.00_DB".Garlic.QDOSERun AND "T-20.00_DB".Garlic.P_CMD THEN
       "T-09.01_DB"."DosePumpON-OFF" := TRUE;
   END_IF;
   IF "T-20.00_DB".Garlic.QDOSERun THEN "T-09.01_DB".DosePumpSpeed := "T-20.00_DB".Garlic.P_SPEED; END_IF;
   IF "T-21.00_DB".Garlic.QDOSERun AND "T-21.00_DB".Garlic.P_CMD THEN
       "T-09.01_DB"."DosePumpON-OFF" := TRUE;
   END_IF;
   IF "T-21.00_DB".Garlic.QDOSERun THEN "T-09.01_DB".DosePumpSpeed := "T-21.00_DB".Garlic.P_SPEED; END_IF;
   IF "T-30.00_DB".Garlic.QDOSERun AND "T-30.00_DB".Garlic.P_CMD THEN
       "T-09.01_DB"."DosePumpON-OFF" := TRUE;
   END_IF;
   IF "T-30.00_DB".Garlic.QDOSERun THEN "T-09.01_DB".DosePumpSpeed := "T-30.00_DB".Garlic.P_SPEED; END_IF;
   IF "T-31.00_DB".Garlic.QDOSERun AND "T-31.00_DB".Garlic.P_CMD THEN
       "T-09.01_DB"."DosePumpON-OFF" := TRUE;
   END_IF;
   IF "T-31.00_DB".Garlic.QDOSERun THEN "T-09.01_DB".DosePumpSpeed := "T-31.00_DB".Garlic.P_SPEED; END_IF;
   IF NOT "T-20.00_DB".Garlic.P_CMD AND NOT "T-21.00_DB".Garlic.P_CMD AND NOT "T-30.00_DB".Garlic.P_CMD AND NOT "T-31.00_DB".Garlic.P_CMD THEN
       "T-09.01_DB"."DosePumpON-OFF" := FALSE;
   END_IF;
END_REGION

REGION Network 36: T-09.01 Buffer Tank Garlic
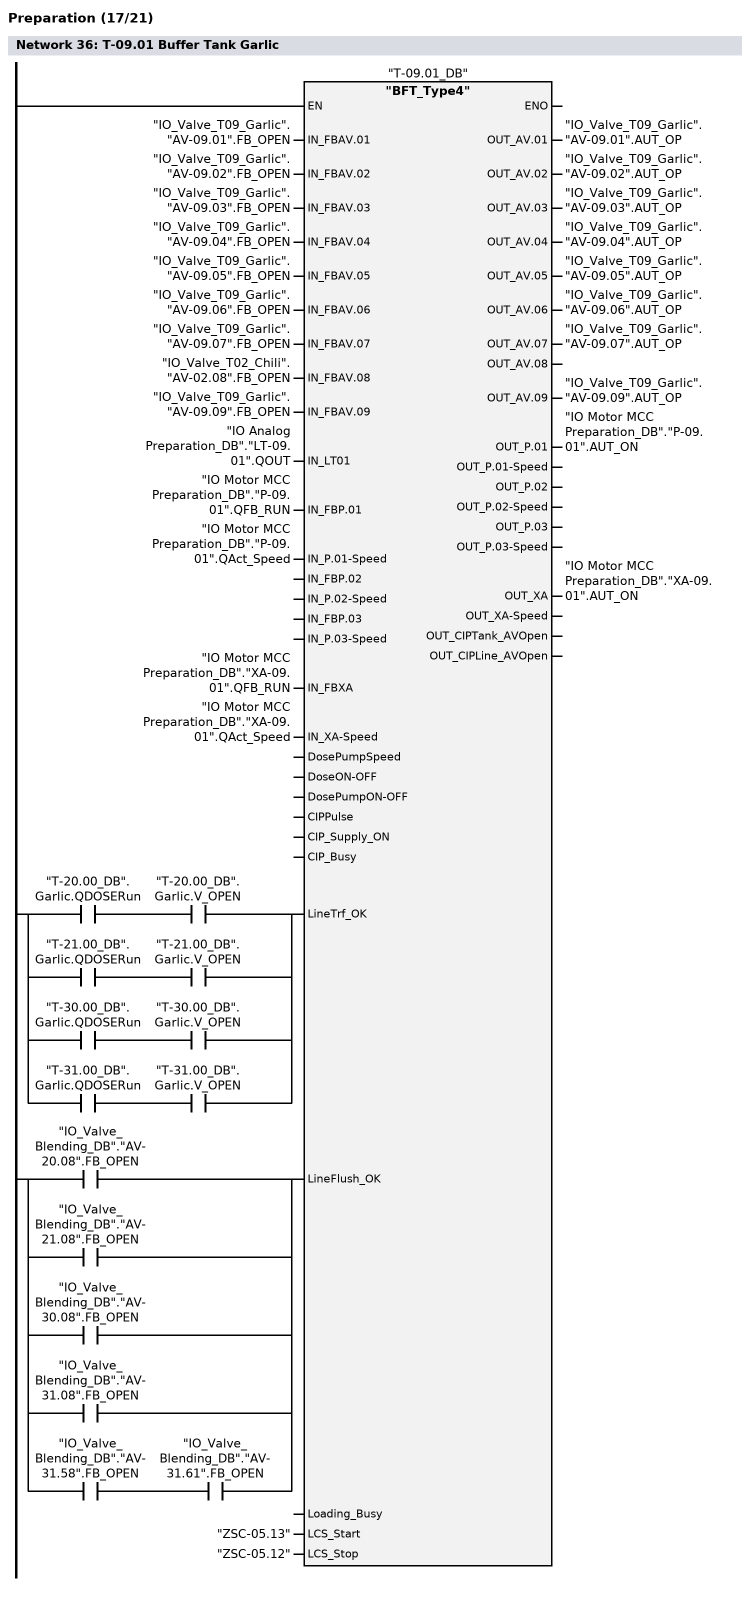
   RUNG wire#powerrail
      "T-09.01_DB"(LineTrf_OK := wire#w1, LineFlush_OK := wire#w2, "IN_FBAV.01" := "IO_Valve_T09_Garlic"."AV-09.01".FB_OPEN, "IN_FBAV.02" := "IO_Valve_T09_Garlic"."AV-09.02".FB_OPEN, "IN_FBAV.03" := "IO_Valve_T09_Garlic"."AV-09.03".FB_OPEN, "IN_FBAV.04" := "IO_Valve_T09_Garlic"."AV-09.04".FB_OPEN, "IN_FBAV.05" := "IO_Valve_T09_Garlic"."AV-09.05".FB_OPEN, "IN_FBAV.06" := "IO_Valve_T09_Garlic"."AV-09.06".FB_OPEN, "IN_FBAV.07" := "IO_Valve_T09_Garlic"."AV-09.07".FB_OPEN, "IN_FBAV.08" := "IO_Valve_T02_Chili"."AV-02.08".FB_OPEN, "IN_FBAV.09" := "IO_Valve_T09_Garlic"."AV-09.09".FB_OPEN, IN_LT01 := "IO Analog Preparation_DB"."LT-09.01".QOUT, "IN_FBP.01" := "IO Motor MCC Preparation_DB"."P-09.01".QFB_RUN, "IN_P.01-Speed" := "IO Motor MCC Preparation_DB"."P-09.01".QAct_Speed, "IN_FBP.02" :=, "IN_P.02-Speed" :=, "IN_FBP.03" :=, "IN_P.03-Speed" :=, IN_FBXA := "IO Motor MCC Preparation_DB"."XA-09.01".QFB_RUN, "IN_XA-Speed" := "IO Motor MCC Preparation_DB"."XA-09.01".QAct_Speed, DosePumpSpeed :=, "DoseON-OFF" :=, "DosePumpON-OFF" :=, CIPPulse :=, CIP_Supply_ON :=, CIP_Busy :=, Loading_Busy :=, LCS_Start := "ZSC-05.13", LCS_Stop := "ZSC-05.12", "OUT_AV.01" => "IO_Valve_T09_Garlic"."AV-09.01".AUT_OP, "OUT_AV.02" => "IO_Valve_T09_Garlic"."AV-09.02".AUT_OP, "OUT_AV.03" => "IO_Valve_T09_Garlic"."AV-09.03".AUT_OP, "OUT_AV.04" => "IO_Valve_T09_Garlic"."AV-09.04".AUT_OP, "OUT_AV.05" => "IO_Valve_T09_Garlic"."AV-09.05".AUT_OP, "OUT_AV.06" => "IO_Valve_T09_Garlic"."AV-09.06".AUT_OP, "OUT_AV.07" => "IO_Valve_T09_Garlic"."AV-09.07".AUT_OP, "OUT_AV.08" =>, "OUT_AV.09" => "IO_Valve_T09_Garlic"."AV-09.09".AUT_OP, "OUT_P.01" => "IO Motor MCC Preparation_DB"."P-09.01".AUT_ON, "OUT_P.01-Speed" =>, "OUT_P.02" =>, "OUT_P.02-Speed" =>, "OUT_P.03" =>, "OUT_P.03-Speed" =>, OUT_XA => "IO Motor MCC Preparation_DB"."XA-09.01".AUT_ON, "OUT_XA-Speed" =>, OUT_CIPTank_AVOpen =>, OUT_CIPLine_AVOpen =>)
   END_RUNG
   RUNG wire#powerrail
      Contact( "T-20.00_DB".Garlic.QDOSERun )
      Contact( "T-20.00_DB".Garlic.V_OPEN )
   END_RUNG wire#w1
   RUNG wire#powerrail
      Contact( "T-21.00_DB".Garlic.QDOSERun )
      Contact( "T-21.00_DB".Garlic.V_OPEN )
   END_RUNG wire#w1
   RUNG wire#powerrail
      Contact( "T-30.00_DB".Garlic.QDOSERun )
      Contact( "T-30.00_DB".Garlic.V_OPEN )
   END_RUNG wire#w1
   RUNG wire#powerrail
      Contact( "T-31.00_DB".Garlic.QDOSERun )
      Contact( "T-31.00_DB".Garlic.V_OPEN )
   END_RUNG wire#w1
   RUNG wire#powerrail
      Contact( "IO_Valve_Blending_DB"."AV-20.08".FB_OPEN )
   END_RUNG wire#w2
   RUNG wire#powerrail
      Contact( "IO_Valve_Blending_DB"."AV-21.08".FB_OPEN )
   END_RUNG wire#w2
   RUNG wire#powerrail
      Contact( "IO_Valve_Blending_DB"."AV-30.08".FB_OPEN )
   END_RUNG wire#w2
   RUNG wire#powerrail
      Contact( "IO_Valve_Blending_DB"."AV-31.08".FB_OPEN )
   END_RUNG wire#w2
   RUNG wire#powerrail
      Contact( "IO_Valve_Blending_DB"."AV-31.58".FB_OPEN )
      Contact( "IO_Valve_Blending_DB"."AV-31.61".FB_OPEN )
   END_RUNG wire#w2
   // the same network as SCL:
   "T-09.01_DB"("IN_FBAV.01" := "IO_Valve_T09_Garlic"."AV-09.01".FB_OPEN,   // "BFT_Type4"
                "IN_FBAV.02" := "IO_Valve_T09_Garlic"."AV-09.02".FB_OPEN,
                "IN_FBAV.03" := "IO_Valve_T09_Garlic"."AV-09.03".FB_OPEN,
                "IN_FBAV.04" := "IO_Valve_T09_Garlic"."AV-09.04".FB_OPEN,
                "IN_FBAV.05" := "IO_Valve_T09_Garlic"."AV-09.05".FB_OPEN,
                "IN_FBAV.06" := "IO_Valve_T09_Garlic"."AV-09.06".FB_OPEN,
                "IN_FBAV.07" := "IO_Valve_T09_Garlic"."AV-09.07".FB_OPEN,
                "IN_FBAV.08" := "IO_Valve_T02_Chili"."AV-02.08".FB_OPEN,
                "IN_FBAV.09" := "IO_Valve_T09_Garlic"."AV-09.09".FB_OPEN,
                IN_LT01 := "IO Analog Preparation_DB"."LT-09.01".QOUT,
                "IN_FBP.01" := "IO Motor MCC Preparation_DB"."P-09.01".QFB_RUN,
                "IN_P.01-Speed" := "IO Motor MCC Preparation_DB"."P-09.01".QAct_Speed,
                IN_FBXA := "IO Motor MCC Preparation_DB"."XA-09.01".QFB_RUN,
                "IN_XA-Speed" := "IO Motor MCC Preparation_DB"."XA-09.01".QAct_Speed,
                LineTrf_OK := ("T-20.00_DB".Garlic.QDOSERun AND "T-20.00_DB".Garlic.V_OPEN) OR ("T-21.00_DB".Garlic.QDOSERun AND "T-21.00_DB".Garlic.V_OPEN) OR ("T-30.00_DB".Garlic.QDOSERun AND "T-30.00_DB".Garlic.V_OPEN) OR ("T-31.00_DB".Garlic.QDOSERun AND "T-31.00_DB".Garlic.V_OPEN),
                LineFlush_OK := "IO_Valve_Blending_DB"."AV-20.08".FB_OPEN OR "IO_Valve_Blending_DB"."AV-21.08".FB_OPEN OR "IO_Valve_Blending_DB"."AV-30.08".FB_OPEN OR "IO_Valve_Blending_DB"."AV-31.08".FB_OPEN OR ("IO_Valve_Blending_DB"."AV-31.58".FB_OPEN AND "IO_Valve_Blending_DB"."AV-31.61".FB_OPEN),
                LCS_Start := "ZSC-05.13",
                LCS_Stop := "ZSC-05.12",
                "OUT_AV.01" => "IO_Valve_T09_Garlic"."AV-09.01".AUT_OP,
                "OUT_AV.02" => "IO_Valve_T09_Garlic"."AV-09.02".AUT_OP,
                "OUT_AV.03" => "IO_Valve_T09_Garlic"."AV-09.03".AUT_OP,
                "OUT_AV.04" => "IO_Valve_T09_Garlic"."AV-09.04".AUT_OP,
                "OUT_AV.05" => "IO_Valve_T09_Garlic"."AV-09.05".AUT_OP,
                "OUT_AV.06" => "IO_Valve_T09_Garlic"."AV-09.06".AUT_OP,
                "OUT_AV.07" => "IO_Valve_T09_Garlic"."AV-09.07".AUT_OP,
                "OUT_AV.09" => "IO_Valve_T09_Garlic"."AV-09.09".AUT_OP,
                "OUT_P.01" => "IO Motor MCC Preparation_DB"."P-09.01".AUT_ON,
                OUT_XA => "IO Motor MCC Preparation_DB"."XA-09.01".AUT_ON);
END_REGION

REGION Network 38: Dose ON OFF T-10.01 Vinegar
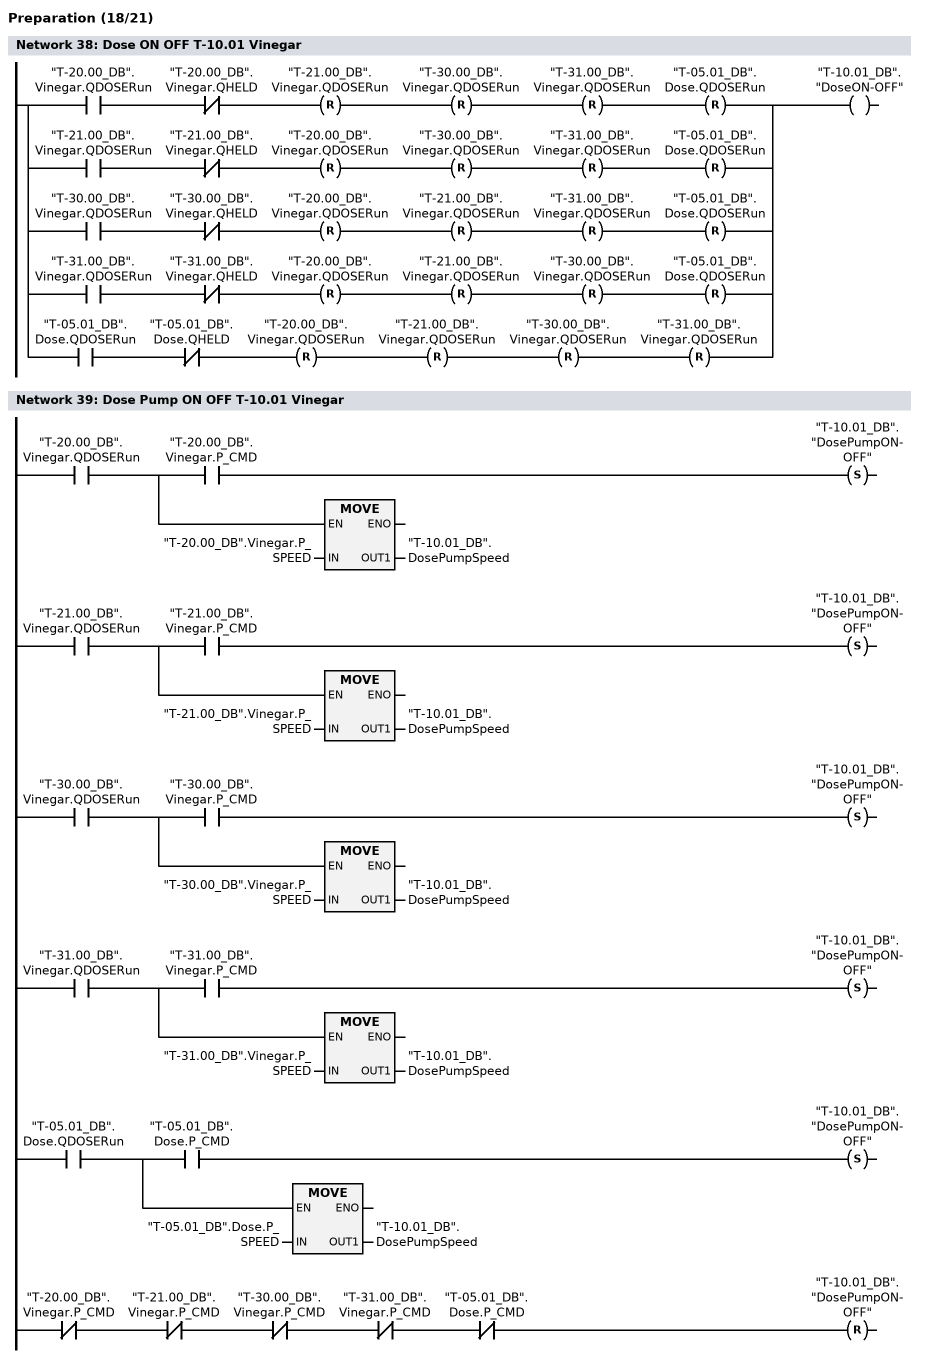
   RUNG wire#powerrail
      Contact( "T-20.00_DB".Vinegar.QDOSERun )
      I_Contact( "T-20.00_DB".Vinegar.QHELD )
      R_Coil( "T-21.00_DB".Vinegar.QDOSERun )
      R_Coil( "T-30.00_DB".Vinegar.QDOSERun )
      R_Coil( "T-31.00_DB".Vinegar.QDOSERun )
      R_Coil( "T-05.01_DB".Dose.QDOSERun )
      wire#w1
      Coil( "T-10.01_DB"."DoseON-OFF" )
   END_RUNG
   RUNG wire#powerrail
      Contact( "T-21.00_DB".Vinegar.QDOSERun )
      I_Contact( "T-21.00_DB".Vinegar.QHELD )
      R_Coil( "T-20.00_DB".Vinegar.QDOSERun )
      R_Coil( "T-30.00_DB".Vinegar.QDOSERun )
      R_Coil( "T-31.00_DB".Vinegar.QDOSERun )
      R_Coil( "T-05.01_DB".Dose.QDOSERun )
   END_RUNG wire#w1
   RUNG wire#powerrail
      Contact( "T-30.00_DB".Vinegar.QDOSERun )
      I_Contact( "T-30.00_DB".Vinegar.QHELD )
      R_Coil( "T-20.00_DB".Vinegar.QDOSERun )
      R_Coil( "T-21.00_DB".Vinegar.QDOSERun )
      R_Coil( "T-31.00_DB".Vinegar.QDOSERun )
      R_Coil( "T-05.01_DB".Dose.QDOSERun )
   END_RUNG wire#w1
   RUNG wire#powerrail
      Contact( "T-31.00_DB".Vinegar.QDOSERun )
      I_Contact( "T-31.00_DB".Vinegar.QHELD )
      R_Coil( "T-20.00_DB".Vinegar.QDOSERun )
      R_Coil( "T-21.00_DB".Vinegar.QDOSERun )
      R_Coil( "T-30.00_DB".Vinegar.QDOSERun )
      R_Coil( "T-05.01_DB".Dose.QDOSERun )
   END_RUNG wire#w1
   RUNG wire#powerrail
      Contact( "T-05.01_DB".Dose.QDOSERun )
      I_Contact( "T-05.01_DB".Dose.QHELD )
      R_Coil( "T-20.00_DB".Vinegar.QDOSERun )
      R_Coil( "T-21.00_DB".Vinegar.QDOSERun )
      R_Coil( "T-30.00_DB".Vinegar.QDOSERun )
      R_Coil( "T-31.00_DB".Vinegar.QDOSERun )
   END_RUNG wire#w1
   // the same network as SCL:
   #_w1 := "T-20.00_DB".Vinegar.QDOSERun AND NOT "T-20.00_DB".Vinegar.QHELD;
   IF #_w1 THEN
       "T-21.00_DB".Vinegar.QDOSERun := FALSE;
       "T-30.00_DB".Vinegar.QDOSERun := FALSE;
       "T-31.00_DB".Vinegar.QDOSERun := FALSE;
       "T-05.01_DB".Dose.QDOSERun := FALSE;
   END_IF;
   #_w2 := "T-21.00_DB".Vinegar.QDOSERun AND NOT "T-21.00_DB".Vinegar.QHELD;
   IF #_w2 THEN
       "T-20.00_DB".Vinegar.QDOSERun := FALSE;
       "T-30.00_DB".Vinegar.QDOSERun := FALSE;
       "T-31.00_DB".Vinegar.QDOSERun := FALSE;
       "T-05.01_DB".Dose.QDOSERun := FALSE;
   END_IF;
   #_w3 := "T-30.00_DB".Vinegar.QDOSERun AND NOT "T-30.00_DB".Vinegar.QHELD;
   IF #_w3 THEN
       "T-20.00_DB".Vinegar.QDOSERun := FALSE;
       "T-21.00_DB".Vinegar.QDOSERun := FALSE;
       "T-31.00_DB".Vinegar.QDOSERun := FALSE;
       "T-05.01_DB".Dose.QDOSERun := FALSE;
   END_IF;
   #_w4 := "T-31.00_DB".Vinegar.QDOSERun AND NOT "T-31.00_DB".Vinegar.QHELD;
   IF #_w4 THEN
       "T-20.00_DB".Vinegar.QDOSERun := FALSE;
       "T-21.00_DB".Vinegar.QDOSERun := FALSE;
       "T-30.00_DB".Vinegar.QDOSERun := FALSE;
       "T-05.01_DB".Dose.QDOSERun := FALSE;
   END_IF;
   #_w5 := "T-05.01_DB".Dose.QDOSERun AND NOT "T-05.01_DB".Dose.QHELD;
   IF #_w5 THEN
       "T-20.00_DB".Vinegar.QDOSERun := FALSE;
       "T-21.00_DB".Vinegar.QDOSERun := FALSE;
       "T-30.00_DB".Vinegar.QDOSERun := FALSE;
       "T-31.00_DB".Vinegar.QDOSERun := FALSE;
   END_IF;
   "T-10.01_DB"."DoseON-OFF" := #_w1 OR #_w2 OR #_w3 OR #_w4 OR #_w5;
END_REGION

REGION Network 39: Dose Pump ON OFF T-10.01 Vinegar
   RUNG wire#powerrail
      Contact( "T-20.00_DB".Vinegar.QDOSERun )
      wire#w1
      Contact( "T-20.00_DB".Vinegar.P_CMD )
      S_Coil( "T-10.01_DB"."DosePumpON-OFF" )
   END_RUNG
   RUNG wire#w1
      Move(in := "T-20.00_DB".Vinegar.P_SPEED, out1 => "T-10.01_DB".DosePumpSpeed)
   END_RUNG
   RUNG wire#powerrail
      Contact( "T-21.00_DB".Vinegar.QDOSERun )
      wire#w2
      Contact( "T-21.00_DB".Vinegar.P_CMD )
      S_Coil( "T-10.01_DB"."DosePumpON-OFF" )
   END_RUNG
   RUNG wire#w2
      Move(in := "T-21.00_DB".Vinegar.P_SPEED, out1 => "T-10.01_DB".DosePumpSpeed)
   END_RUNG
   RUNG wire#powerrail
      Contact( "T-30.00_DB".Vinegar.QDOSERun )
      wire#w3
      Contact( "T-30.00_DB".Vinegar.P_CMD )
      S_Coil( "T-10.01_DB"."DosePumpON-OFF" )
   END_RUNG
   RUNG wire#w3
      Move(in := "T-30.00_DB".Vinegar.P_SPEED, out1 => "T-10.01_DB".DosePumpSpeed)
   END_RUNG
   RUNG wire#powerrail
      Contact( "T-31.00_DB".Vinegar.QDOSERun )
      wire#w4
      Contact( "T-31.00_DB".Vinegar.P_CMD )
      S_Coil( "T-10.01_DB"."DosePumpON-OFF" )
   END_RUNG
   RUNG wire#w4
      Move(in := "T-31.00_DB".Vinegar.P_SPEED, out1 => "T-10.01_DB".DosePumpSpeed)
   END_RUNG
   RUNG wire#powerrail
      Contact( "T-05.01_DB".Dose.QDOSERun )
      wire#w5
      Contact( "T-05.01_DB".Dose.P_CMD )
      S_Coil( "T-10.01_DB"."DosePumpON-OFF" )
   END_RUNG
   RUNG wire#w5
      Move(in := "T-05.01_DB".Dose.P_SPEED, out1 => "T-10.01_DB".DosePumpSpeed)
   END_RUNG
   RUNG wire#powerrail
      I_Contact( "T-20.00_DB".Vinegar.P_CMD )
      I_Contact( "T-21.00_DB".Vinegar.P_CMD )
      I_Contact( "T-30.00_DB".Vinegar.P_CMD )
      I_Contact( "T-31.00_DB".Vinegar.P_CMD )
      I_Contact( "T-05.01_DB".Dose.P_CMD )
      R_Coil( "T-10.01_DB"."DosePumpON-OFF" )
   END_RUNG
   // the same network as SCL:
   IF "T-20.00_DB".Vinegar.QDOSERun AND "T-20.00_DB".Vinegar.P_CMD THEN
       "T-10.01_DB"."DosePumpON-OFF" := TRUE;
   END_IF;
   IF "T-20.00_DB".Vinegar.QDOSERun THEN "T-10.01_DB".DosePumpSpeed := "T-20.00_DB".Vinegar.P_SPEED; END_IF;
   IF "T-21.00_DB".Vinegar.QDOSERun AND "T-21.00_DB".Vinegar.P_CMD THEN
       "T-10.01_DB"."DosePumpON-OFF" := TRUE;
   END_IF;
   IF "T-21.00_DB".Vinegar.QDOSERun THEN "T-10.01_DB".DosePumpSpeed := "T-21.00_DB".Vinegar.P_SPEED; END_IF;
   IF "T-30.00_DB".Vinegar.QDOSERun AND "T-30.00_DB".Vinegar.P_CMD THEN
       "T-10.01_DB"."DosePumpON-OFF" := TRUE;
   END_IF;
   IF "T-30.00_DB".Vinegar.QDOSERun THEN "T-10.01_DB".DosePumpSpeed := "T-30.00_DB".Vinegar.P_SPEED; END_IF;
   IF "T-31.00_DB".Vinegar.QDOSERun AND "T-31.00_DB".Vinegar.P_CMD THEN
       "T-10.01_DB"."DosePumpON-OFF" := TRUE;
   END_IF;
   IF "T-31.00_DB".Vinegar.QDOSERun THEN "T-10.01_DB".DosePumpSpeed := "T-31.00_DB".Vinegar.P_SPEED; END_IF;
   IF "T-05.01_DB".Dose.QDOSERun AND "T-05.01_DB".Dose.P_CMD THEN
       "T-10.01_DB"."DosePumpON-OFF" := TRUE;
   END_IF;
   IF "T-05.01_DB".Dose.QDOSERun THEN "T-10.01_DB".DosePumpSpeed := "T-05.01_DB".Dose.P_SPEED; END_IF;
   IF NOT "T-20.00_DB".Vinegar.P_CMD AND NOT "T-21.00_DB".Vinegar.P_CMD AND NOT "T-30.00_DB".Vinegar.P_CMD AND NOT "T-31.00_DB".Vinegar.P_CMD AND NOT "T-05.01_DB".Dose.P_CMD THEN
       "T-10.01_DB"."DosePumpON-OFF" := FALSE;
   END_IF;
END_REGION

REGION Network 40: T-10.01 Buffer Tank Vinegar
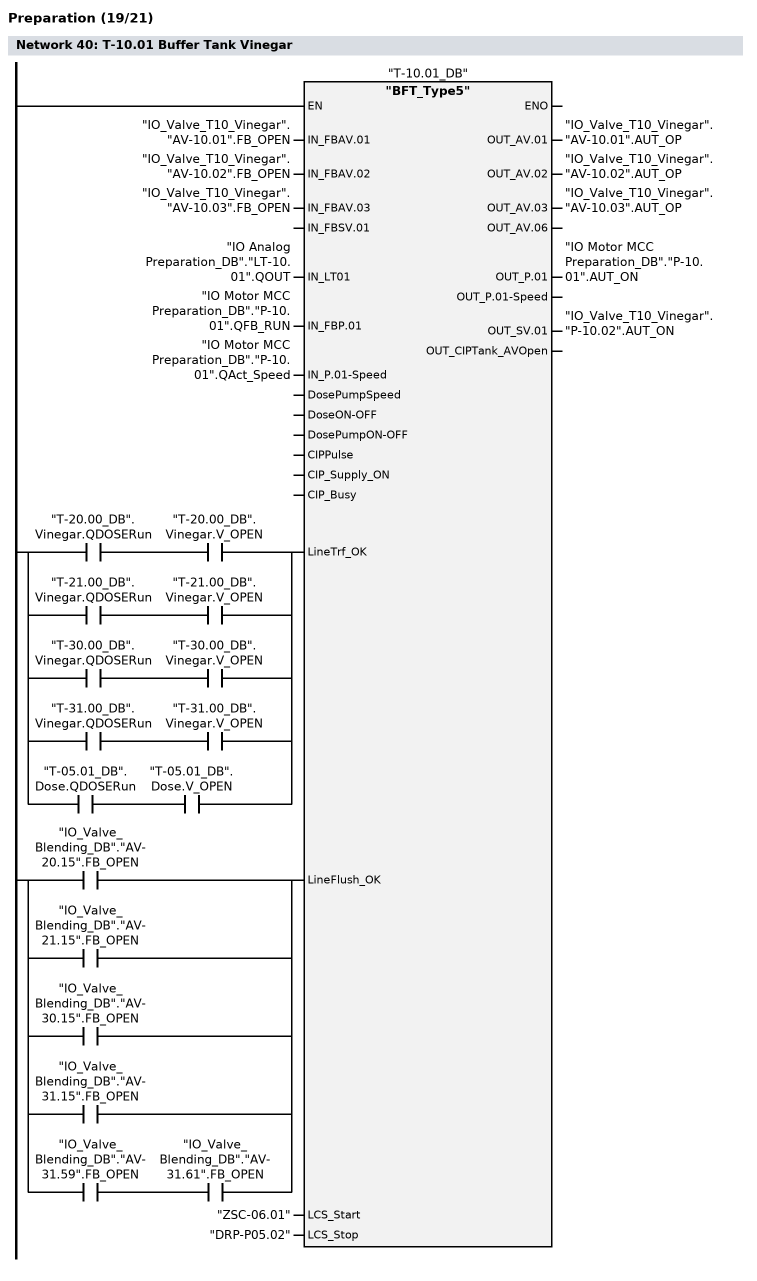
   RUNG wire#powerrail
      "T-10.01_DB"(LineTrf_OK := wire#w1, LineFlush_OK := wire#w2, "IN_FBAV.01" := "IO_Valve_T10_Vinegar"."AV-10.01".FB_OPEN, "IN_FBAV.02" := "IO_Valve_T10_Vinegar"."AV-10.02".FB_OPEN, "IN_FBAV.03" := "IO_Valve_T10_Vinegar"."AV-10.03".FB_OPEN, "IN_FBSV.01" :=, IN_LT01 := "IO Analog Preparation_DB"."LT-10.01".QOUT, "IN_FBP.01" := "IO Motor MCC Preparation_DB"."P-10.01".QFB_RUN, "IN_P.01-Speed" := "IO Motor MCC Preparation_DB"."P-10.01".QAct_Speed, DosePumpSpeed :=, "DoseON-OFF" :=, "DosePumpON-OFF" :=, CIPPulse :=, CIP_Supply_ON :=, CIP_Busy :=, LCS_Start := "ZSC-06.01", LCS_Stop := "DRP-P05.02", "OUT_AV.01" => "IO_Valve_T10_Vinegar"."AV-10.01".AUT_OP, "OUT_AV.02" => "IO_Valve_T10_Vinegar"."AV-10.02".AUT_OP, "OUT_AV.03" => "IO_Valve_T10_Vinegar"."AV-10.03".AUT_OP, "OUT_AV.06" =>, "OUT_P.01" => "IO Motor MCC Preparation_DB"."P-10.01".AUT_ON, "OUT_P.01-Speed" =>, "OUT_SV.01" => "IO_Valve_T10_Vinegar"."P-10.02".AUT_ON, OUT_CIPTank_AVOpen =>)
   END_RUNG
   RUNG wire#powerrail
      Contact( "T-20.00_DB".Vinegar.QDOSERun )
      Contact( "T-20.00_DB".Vinegar.V_OPEN )
   END_RUNG wire#w1
   RUNG wire#powerrail
      Contact( "T-21.00_DB".Vinegar.QDOSERun )
      Contact( "T-21.00_DB".Vinegar.V_OPEN )
   END_RUNG wire#w1
   RUNG wire#powerrail
      Contact( "T-30.00_DB".Vinegar.QDOSERun )
      Contact( "T-30.00_DB".Vinegar.V_OPEN )
   END_RUNG wire#w1
   RUNG wire#powerrail
      Contact( "T-31.00_DB".Vinegar.QDOSERun )
      Contact( "T-31.00_DB".Vinegar.V_OPEN )
   END_RUNG wire#w1
   RUNG wire#powerrail
      Contact( "T-05.01_DB".Dose.QDOSERun )
      Contact( "T-05.01_DB".Dose.V_OPEN )
   END_RUNG wire#w1
   RUNG wire#powerrail
      Contact( "IO_Valve_Blending_DB"."AV-20.15".FB_OPEN )
   END_RUNG wire#w2
   RUNG wire#powerrail
      Contact( "IO_Valve_Blending_DB"."AV-21.15".FB_OPEN )
   END_RUNG wire#w2
   RUNG wire#powerrail
      Contact( "IO_Valve_Blending_DB"."AV-30.15".FB_OPEN )
   END_RUNG wire#w2
   RUNG wire#powerrail
      Contact( "IO_Valve_Blending_DB"."AV-31.15".FB_OPEN )
   END_RUNG wire#w2
   RUNG wire#powerrail
      Contact( "IO_Valve_Blending_DB"."AV-31.59".FB_OPEN )
      Contact( "IO_Valve_Blending_DB"."AV-31.61".FB_OPEN )
   END_RUNG wire#w2
   // the same network as SCL:
   "T-10.01_DB"("IN_FBAV.01" := "IO_Valve_T10_Vinegar"."AV-10.01".FB_OPEN,   // "BFT_Type5"
                "IN_FBAV.02" := "IO_Valve_T10_Vinegar"."AV-10.02".FB_OPEN,
                "IN_FBAV.03" := "IO_Valve_T10_Vinegar"."AV-10.03".FB_OPEN,
                IN_LT01 := "IO Analog Preparation_DB"."LT-10.01".QOUT,
                "IN_FBP.01" := "IO Motor MCC Preparation_DB"."P-10.01".QFB_RUN,
                "IN_P.01-Speed" := "IO Motor MCC Preparation_DB"."P-10.01".QAct_Speed,
                LineTrf_OK := ("T-20.00_DB".Vinegar.QDOSERun AND "T-20.00_DB".Vinegar.V_OPEN) OR ("T-21.00_DB".Vinegar.QDOSERun AND "T-21.00_DB".Vinegar.V_OPEN) OR ("T-30.00_DB".Vinegar.QDOSERun AND "T-30.00_DB".Vinegar.V_OPEN) OR ("T-31.00_DB".Vinegar.QDOSERun AND "T-31.00_DB".Vinegar.V_OPEN) OR ("T-05.01_DB".Dose.QDOSERun AND "T-05.01_DB".Dose.V_OPEN),
                LineFlush_OK := "IO_Valve_Blending_DB"."AV-20.15".FB_OPEN OR "IO_Valve_Blending_DB"."AV-21.15".FB_OPEN OR "IO_Valve_Blending_DB"."AV-30.15".FB_OPEN OR "IO_Valve_Blending_DB"."AV-31.15".FB_OPEN OR ("IO_Valve_Blending_DB"."AV-31.59".FB_OPEN AND "IO_Valve_Blending_DB"."AV-31.61".FB_OPEN),
                LCS_Start := "ZSC-06.01",
                LCS_Stop := "DRP-P05.02",
                "OUT_AV.01" => "IO_Valve_T10_Vinegar"."AV-10.01".AUT_OP,
                "OUT_AV.02" => "IO_Valve_T10_Vinegar"."AV-10.02".AUT_OP,
                "OUT_AV.03" => "IO_Valve_T10_Vinegar"."AV-10.03".AUT_OP,
                "OUT_P.01" => "IO Motor MCC Preparation_DB"."P-10.01".AUT_ON,
                "OUT_SV.01" => "IO_Valve_T10_Vinegar"."P-10.02".AUT_ON);
END_REGION

REGION Network 41: Line CIP Valve AV-02.06
   // CIP Supply Line 1 for CIP Line T-02, T03, T04, T09 to Blending
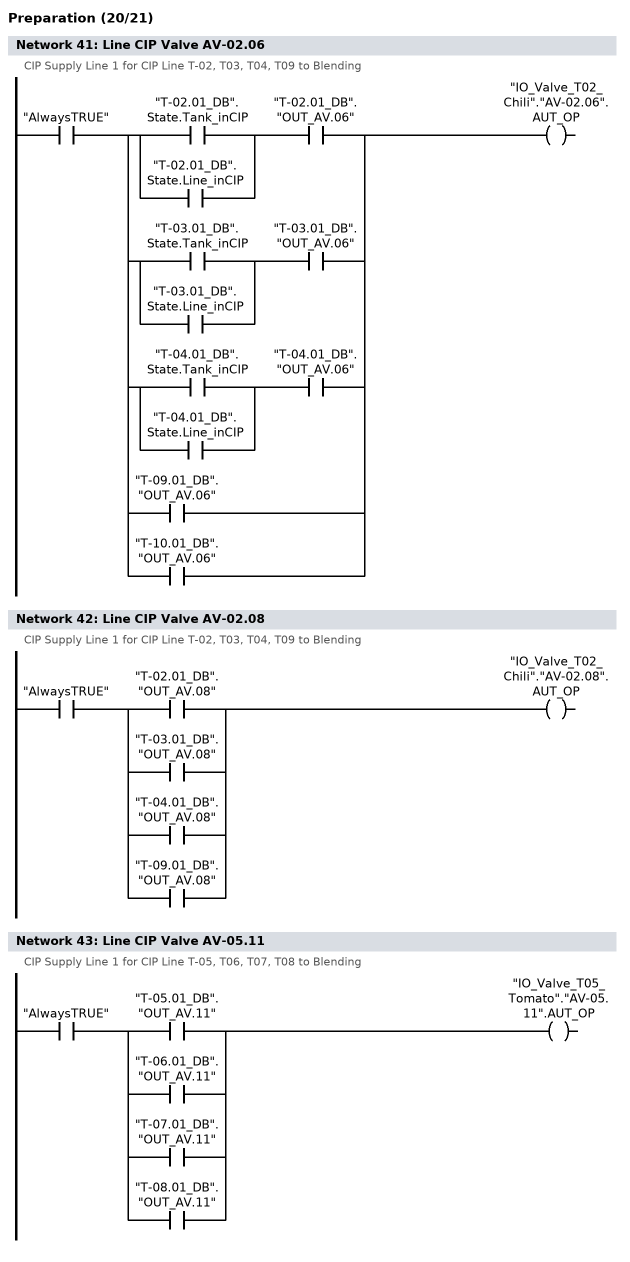
   RUNG wire#powerrail
      Contact( "AlwaysTRUE" )
      wire#w1
      Contact( "T-02.01_DB".State.Tank_inCIP )
      wire#w2
      Contact( "T-02.01_DB"."OUT_AV.06" )
      wire#w3
      Coil( "IO_Valve_T02_Chili"."AV-02.06".AUT_OP )
   END_RUNG
   RUNG wire#w1
      Contact( "T-02.01_DB".State.Line_inCIP )
   END_RUNG wire#w2
   RUNG wire#w1
      Contact( "T-03.01_DB".State.Tank_inCIP )
      wire#w4
      Contact( "T-03.01_DB"."OUT_AV.06" )
   END_RUNG wire#w3
   RUNG wire#w1
      Contact( "T-03.01_DB".State.Line_inCIP )
   END_RUNG wire#w4
   RUNG wire#w1
      Contact( "T-04.01_DB".State.Tank_inCIP )
      wire#w5
      Contact( "T-04.01_DB"."OUT_AV.06" )
   END_RUNG wire#w3
   RUNG wire#w1
      Contact( "T-04.01_DB".State.Line_inCIP )
   END_RUNG wire#w5
   RUNG wire#w1
      Contact( "T-09.01_DB"."OUT_AV.06" )
   END_RUNG wire#w3
   RUNG wire#w1
      Contact( "T-10.01_DB"."OUT_AV.06" )
   END_RUNG wire#w3
   // the same network as SCL:
   "IO_Valve_T02_Chili"."AV-02.06".AUT_OP := "AlwaysTRUE" AND ((("T-02.01_DB".State.Tank_inCIP OR "T-02.01_DB".State.Line_inCIP) AND "T-02.01_DB"."OUT_AV.06") OR (("T-03.01_DB".State.Tank_inCIP OR "T-03.01_DB".State.Line_inCIP) AND "T-03.01_DB"."OUT_AV.06") OR (("T-04.01_DB".State.Tank_inCIP OR "T-04.01_DB".State.Line_inCIP) AND "T-04.01_DB"."OUT_AV.06") OR "T-09.01_DB"."OUT_AV.06" OR "T-10.01_DB"."OUT_AV.06");
END_REGION

